// TIA Portal V17 export
// export: Created 2025-03-12T15:33:37.1839538Z, ExportSetting WithDefaults, DisplayName Totally Integrated Automation Portal, DisplayVersion V17 Update 8, DisplayName TIA Portal Openness, DisplayVersion V17 Update 8, DisplayName TIA Portal Version Control Interface, DisplayVersion V17, DisplayName SINAMICS Startdrive Advanced, DisplayVersion V17 SP2, DisplayName SINAMICS Startdrive G110M, G120, G120C, G120D, G120P, G115D, DisplayVersion V17 SP2, DisplayName SINAMICS Startdrive G130, G150, S120, S150, SINAMICS MV, S210, DisplayVersion V17 SP2, DisplayName STEP 7 Professional, DisplayVersion V17 Update 8, DisplayName SINUMERIK ONE STEP 7 Toolbox, DisplayVersion V17 Update 12, DisplayName SINUMERIK 840D sl STEP 7 Toolbox, DisplayVersion V17 Update 12, DisplayName STEP 7 Safety, DisplayVersion V17 Update 6, DisplayName WinCC Advanced, DisplayVersion V17 Update 8
FUNCTION "FC440_MACHINE_ALARM_DECODING" : Void   // FC440, LAD
{ S7_Optimized_Access := 'FALSE' }
AUTHOR : ETXETAR
VERSION : 1.0
// stored: AutoNumber false, IsIECCheckEnabled false, SetENOAutomatically false, UDAEnableTagReadback false
   VAR_TEMP
      RST_ALARMS_1 : Bool;   // RESET ALARMS 1
      RST_ALARMS_2 : Bool;   // RESET ALARMS 2
      ZERO : Int;   // ZERO
      RET_VAL_1 : Int;   // RET VALUE
   END_VAR
   VAR CONSTANT
      FC_CONSTANT : Int := 440;
   END_VAR
   VAR_TEMP   // added for the SCL form of the ladder/FBD networks
      _w1 : Bool;
      _w2 : Bool;
      _w3 : Bool;
      _w4 : Bool;
      _w5 : Bool;
      _w6 : Bool;
      _w7 : Bool;
      _w8 : Bool;
      _w9 : Bool;
      _w10 : Bool;
      _w11 : Bool;
   END_VAR
BEGIN

REGION Network 1: ZERO
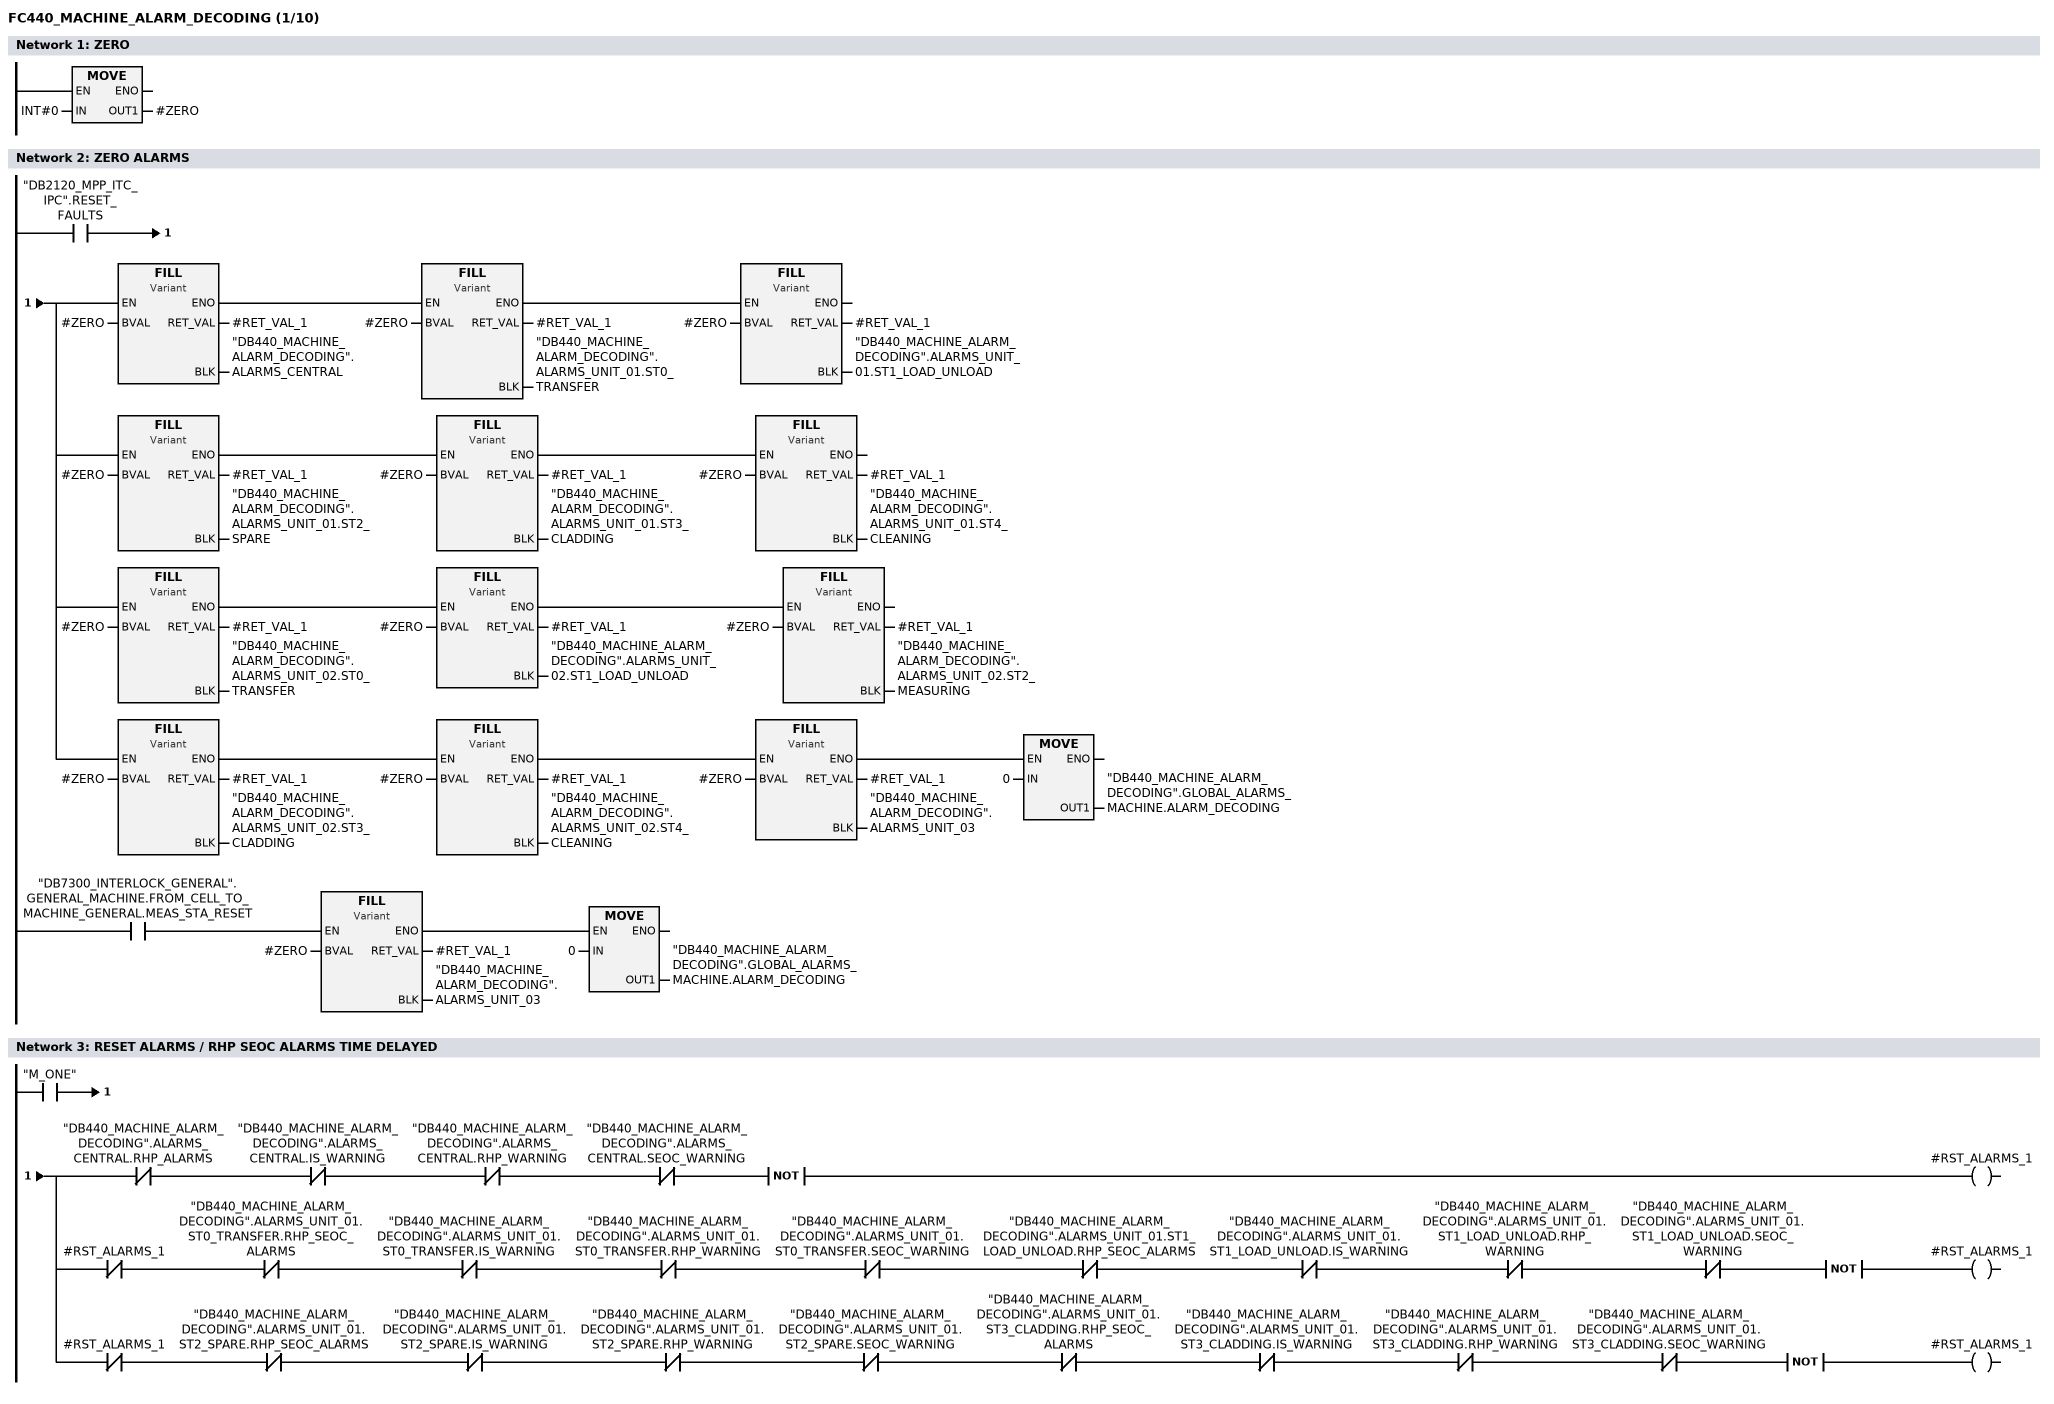
   RUNG wire#powerrail
      { S7_GenerateENO := "TRUE" } Move(in := INT#0, out1 => #ZERO)
   END_RUNG
   // the same network as SCL:
   #ZERO := INT#0;
END_REGION

REGION Network 2: ZERO ALARMS
   RUNG wire#powerrail
      Contact( "DB2120_MPP_ITC_IPC".RESET_FAULTS )
      wire#w1
      { S7_Templates := "ptr_type := Variant" } FILL(BVAL := #ZERO, RET_VAL => #RET_VAL_1, BLK => "DB440_MACHINE_ALARM_DECODING".ALARMS_CENTRAL)
      { S7_Templates := "ptr_type := Variant" } FILL(BVAL := #ZERO, RET_VAL => #RET_VAL_1, BLK => "DB440_MACHINE_ALARM_DECODING".ALARMS_UNIT_01.ST0_TRANSFER)
      { S7_Templates := "ptr_type := Variant" } FILL(BVAL := #ZERO, RET_VAL => #RET_VAL_1, BLK => "DB440_MACHINE_ALARM_DECODING".ALARMS_UNIT_01.ST1_LOAD_UNLOAD)
   END_RUNG
   RUNG wire#w1
      { S7_Templates := "ptr_type := Variant" } FILL(BVAL := #ZERO, RET_VAL => #RET_VAL_1, BLK => "DB440_MACHINE_ALARM_DECODING".ALARMS_UNIT_01.ST2_SPARE)
      { S7_Templates := "ptr_type := Variant" } FILL(BVAL := #ZERO, RET_VAL => #RET_VAL_1, BLK => "DB440_MACHINE_ALARM_DECODING".ALARMS_UNIT_01.ST3_CLADDING)
      { S7_Templates := "ptr_type := Variant" } FILL(BVAL := #ZERO, RET_VAL => #RET_VAL_1, BLK => "DB440_MACHINE_ALARM_DECODING".ALARMS_UNIT_01.ST4_CLEANING)
   END_RUNG
   RUNG wire#w1
      { S7_Templates := "ptr_type := Variant" } FILL(BVAL := #ZERO, RET_VAL => #RET_VAL_1, BLK => "DB440_MACHINE_ALARM_DECODING".ALARMS_UNIT_02.ST0_TRANSFER)
      { S7_Templates := "ptr_type := Variant" } FILL(BVAL := #ZERO, RET_VAL => #RET_VAL_1, BLK => "DB440_MACHINE_ALARM_DECODING".ALARMS_UNIT_02.ST1_LOAD_UNLOAD)
      { S7_Templates := "ptr_type := Variant" } FILL(BVAL := #ZERO, RET_VAL => #RET_VAL_1, BLK => "DB440_MACHINE_ALARM_DECODING".ALARMS_UNIT_02.ST2_MEASURING)
   END_RUNG
   RUNG wire#w1
      { S7_Templates := "ptr_type := Variant" } FILL(BVAL := #ZERO, RET_VAL => #RET_VAL_1, BLK => "DB440_MACHINE_ALARM_DECODING".ALARMS_UNIT_02.ST3_CLADDING)
      { S7_Templates := "ptr_type := Variant" } FILL(BVAL := #ZERO, RET_VAL => #RET_VAL_1, BLK => "DB440_MACHINE_ALARM_DECODING".ALARMS_UNIT_02.ST4_CLEANING)
      { S7_Templates := "ptr_type := Variant" } FILL(BVAL := #ZERO, RET_VAL => #RET_VAL_1, BLK => "DB440_MACHINE_ALARM_DECODING".ALARMS_UNIT_03)
      { S7_GenerateENO := "TRUE" } Move(in := 0, out1 => "DB440_MACHINE_ALARM_DECODING".GLOBAL_ALARMS_MACHINE.ALARM_DECODING)
   END_RUNG
   RUNG wire#powerrail
      Contact( "DB7300_INTERLOCK_GENERAL".GENERAL_MACHINE.FROM_CELL_TO_MACHINE_GENERAL.MEAS_STA_RESET )
      { S7_Templates := "ptr_type := Variant" } FILL(BVAL := #ZERO, RET_VAL => #RET_VAL_1, BLK => "DB440_MACHINE_ALARM_DECODING".ALARMS_UNIT_03)
      { S7_GenerateENO := "TRUE" } Move(in := 0, out1 => "DB440_MACHINE_ALARM_DECODING".GLOBAL_ALARMS_MACHINE.ALARM_DECODING)
   END_RUNG
   // the same network as SCL:
   #_w2 := "DB2120_MPP_ITC_IPC".RESET_FAULTS;
   #RET_VAL_1 := FILL(EN := "DB2120_MPP_ITC_IPC".RESET_FAULTS,
                      BVAL := #ZERO,
                      BLK => "DB440_MACHINE_ALARM_DECODING".ALARMS_CENTRAL,
                      ENO => #_w1);
   #RET_VAL_1 := FILL(EN := #_w1,
                      BVAL := #ZERO,
                      BLK => "DB440_MACHINE_ALARM_DECODING".ALARMS_UNIT_01.ST0_TRANSFER,
                      ENO => #_w3);
   IF #_w3 THEN
       #RET_VAL_1 := FILL(BVAL := #ZERO, BLK => "DB440_MACHINE_ALARM_DECODING".ALARMS_UNIT_01.ST1_LOAD_UNLOAD);
   END_IF;
   #RET_VAL_1 := FILL(EN := #_w2,
                      BVAL := #ZERO,
                      BLK => "DB440_MACHINE_ALARM_DECODING".ALARMS_UNIT_01.ST2_SPARE,
                      ENO => #_w4);
   #RET_VAL_1 := FILL(EN := #_w4,
                      BVAL := #ZERO,
                      BLK => "DB440_MACHINE_ALARM_DECODING".ALARMS_UNIT_01.ST3_CLADDING,
                      ENO => #_w5);
   IF #_w5 THEN
       #RET_VAL_1 := FILL(BVAL := #ZERO, BLK => "DB440_MACHINE_ALARM_DECODING".ALARMS_UNIT_01.ST4_CLEANING);
   END_IF;
   #RET_VAL_1 := FILL(EN := #_w2,
                      BVAL := #ZERO,
                      BLK => "DB440_MACHINE_ALARM_DECODING".ALARMS_UNIT_02.ST0_TRANSFER,
                      ENO => #_w6);
   #RET_VAL_1 := FILL(EN := #_w6,
                      BVAL := #ZERO,
                      BLK => "DB440_MACHINE_ALARM_DECODING".ALARMS_UNIT_02.ST1_LOAD_UNLOAD,
                      ENO => #_w7);
   IF #_w7 THEN
       #RET_VAL_1 := FILL(BVAL := #ZERO, BLK => "DB440_MACHINE_ALARM_DECODING".ALARMS_UNIT_02.ST2_MEASURING);
   END_IF;
   #RET_VAL_1 := FILL(EN := #_w2,
                      BVAL := #ZERO,
                      BLK => "DB440_MACHINE_ALARM_DECODING".ALARMS_UNIT_02.ST3_CLADDING,
                      ENO => #_w8);
   #RET_VAL_1 := FILL(EN := #_w8,
                      BVAL := #ZERO,
                      BLK => "DB440_MACHINE_ALARM_DECODING".ALARMS_UNIT_02.ST4_CLEANING,
                      ENO => #_w9);
   #RET_VAL_1 := FILL(EN := #_w9,
                      BVAL := #ZERO,
                      BLK => "DB440_MACHINE_ALARM_DECODING".ALARMS_UNIT_03,
                      ENO => #_w10);
   IF #_w10 THEN "DB440_MACHINE_ALARM_DECODING".GLOBAL_ALARMS_MACHINE.ALARM_DECODING := 0; END_IF;
   #RET_VAL_1 := FILL(EN := "DB7300_INTERLOCK_GENERAL".GENERAL_MACHINE.FROM_CELL_TO_MACHINE_GENERAL.MEAS_STA_RESET,
                      BVAL := #ZERO,
                      BLK => "DB440_MACHINE_ALARM_DECODING".ALARMS_UNIT_03,
                      ENO => #_w11);
   IF #_w11 THEN "DB440_MACHINE_ALARM_DECODING".GLOBAL_ALARMS_MACHINE.ALARM_DECODING := 0; END_IF;
END_REGION

REGION Network 3: RESET ALARMS / RHP SEOC ALARMS TIME DELAYED
   RUNG wire#powerrail
      Contact( "M_ONE" )
      wire#w1
      I_Contact( "DB440_MACHINE_ALARM_DECODING".ALARMS_CENTRAL.RHP_ALARMS )
      I_Contact( "DB440_MACHINE_ALARM_DECODING".ALARMS_CENTRAL.IS_WARNING )
      I_Contact( "DB440_MACHINE_ALARM_DECODING".ALARMS_CENTRAL.RHP_WARNING )
      I_Contact( "DB440_MACHINE_ALARM_DECODING".ALARMS_CENTRAL.SEOC_WARNING )
      Not()
      Coil( #RST_ALARMS_1 )
   END_RUNG
   RUNG wire#w1
      I_Contact( #RST_ALARMS_1 )
      I_Contact( "DB440_MACHINE_ALARM_DECODING".ALARMS_UNIT_01.ST0_TRANSFER.RHP_SEOC_ALARMS )
      I_Contact( "DB440_MACHINE_ALARM_DECODING".ALARMS_UNIT_01.ST0_TRANSFER.IS_WARNING )
      I_Contact( "DB440_MACHINE_ALARM_DECODING".ALARMS_UNIT_01.ST0_TRANSFER.RHP_WARNING )
      I_Contact( "DB440_MACHINE_ALARM_DECODING".ALARMS_UNIT_01.ST0_TRANSFER.SEOC_WARNING )
      I_Contact( "DB440_MACHINE_ALARM_DECODING".ALARMS_UNIT_01.ST1_LOAD_UNLOAD.RHP_SEOC_ALARMS )
      I_Contact( "DB440_MACHINE_ALARM_DECODING".ALARMS_UNIT_01.ST1_LOAD_UNLOAD.IS_WARNING )
      I_Contact( "DB440_MACHINE_ALARM_DECODING".ALARMS_UNIT_01.ST1_LOAD_UNLOAD.RHP_WARNING )
      I_Contact( "DB440_MACHINE_ALARM_DECODING".ALARMS_UNIT_01.ST1_LOAD_UNLOAD.SEOC_WARNING )
      Not()
      Coil( #RST_ALARMS_1 )
   END_RUNG
   RUNG wire#w1
      I_Contact( #RST_ALARMS_1 )
      I_Contact( "DB440_MACHINE_ALARM_DECODING".ALARMS_UNIT_01.ST2_SPARE.RHP_SEOC_ALARMS )
      I_Contact( "DB440_MACHINE_ALARM_DECODING".ALARMS_UNIT_01.ST2_SPARE.IS_WARNING )
      I_Contact( "DB440_MACHINE_ALARM_DECODING".ALARMS_UNIT_01.ST2_SPARE.RHP_WARNING )
      I_Contact( "DB440_MACHINE_ALARM_DECODING".ALARMS_UNIT_01.ST2_SPARE.SEOC_WARNING )
      I_Contact( "DB440_MACHINE_ALARM_DECODING".ALARMS_UNIT_01.ST3_CLADDING.RHP_SEOC_ALARMS )
      I_Contact( "DB440_MACHINE_ALARM_DECODING".ALARMS_UNIT_01.ST3_CLADDING.IS_WARNING )
      I_Contact( "DB440_MACHINE_ALARM_DECODING".ALARMS_UNIT_01.ST3_CLADDING.RHP_WARNING )
      I_Contact( "DB440_MACHINE_ALARM_DECODING".ALARMS_UNIT_01.ST3_CLADDING.SEOC_WARNING )
      Not()
      Coil( #RST_ALARMS_1 )
   END_RUNG
   // the same network as SCL:
   #RST_ALARMS_1 := NOT ("M_ONE" AND NOT "DB440_MACHINE_ALARM_DECODING".ALARMS_CENTRAL.RHP_ALARMS AND NOT "DB440_MACHINE_ALARM_DECODING".ALARMS_CENTRAL.IS_WARNING AND NOT "DB440_MACHINE_ALARM_DECODING".ALARMS_CENTRAL.RHP_WARNING AND NOT "DB440_MACHINE_ALARM_DECODING".ALARMS_CENTRAL.SEOC_WARNING);
   #RST_ALARMS_1 := NOT ("M_ONE" AND NOT #RST_ALARMS_1 AND NOT "DB440_MACHINE_ALARM_DECODING".ALARMS_UNIT_01.ST0_TRANSFER.RHP_SEOC_ALARMS AND NOT "DB440_MACHINE_ALARM_DECODING".ALARMS_UNIT_01.ST0_TRANSFER.IS_WARNING AND NOT "DB440_MACHINE_ALARM_DECODING".ALARMS_UNIT_01.ST0_TRANSFER.RHP_WARNING AND NOT "DB440_MACHINE_ALARM_DECODING".ALARMS_UNIT_01.ST0_TRANSFER.SEOC_WARNING AND NOT "DB440_MACHINE_ALARM_DECODING".ALARMS_UNIT_01.ST1_LOAD_UNLOAD.RHP_SEOC_ALARMS AND NOT "DB440_MACHINE_ALARM_DECODING".ALARMS_UNIT_01.ST1_LOAD_UNLOAD.IS_WARNING AND NOT "DB440_MACHINE_ALARM_DECODING".ALARMS_UNIT_01.ST1_LOAD_UNLOAD.RHP_WARNING AND NOT "DB440_MACHINE_ALARM_DECODING".ALARMS_UNIT_01.ST1_LOAD_UNLOAD.SEOC_WARNING);
   #RST_ALARMS_1 := NOT ("M_ONE" AND NOT #RST_ALARMS_1 AND NOT "DB440_MACHINE_ALARM_DECODING".ALARMS_UNIT_01.ST2_SPARE.RHP_SEOC_ALARMS AND NOT "DB440_MACHINE_ALARM_DECODING".ALARMS_UNIT_01.ST2_SPARE.IS_WARNING AND NOT "DB440_MACHINE_ALARM_DECODING".ALARMS_UNIT_01.ST2_SPARE.RHP_WARNING AND NOT "DB440_MACHINE_ALARM_DECODING".ALARMS_UNIT_01.ST2_SPARE.SEOC_WARNING AND NOT "DB440_MACHINE_ALARM_DECODING".ALARMS_UNIT_01.ST3_CLADDING.RHP_SEOC_ALARMS AND NOT "DB440_MACHINE_ALARM_DECODING".ALARMS_UNIT_01.ST3_CLADDING.IS_WARNING AND NOT "DB440_MACHINE_ALARM_DECODING".ALARMS_UNIT_01.ST3_CLADDING.RHP_WARNING AND NOT "DB440_MACHINE_ALARM_DECODING".ALARMS_UNIT_01.ST3_CLADDING.SEOC_WARNING);
END_REGION

REGION Network 4: RESET ALARMS / RHP SEOC ALARMS TIME DELAYED
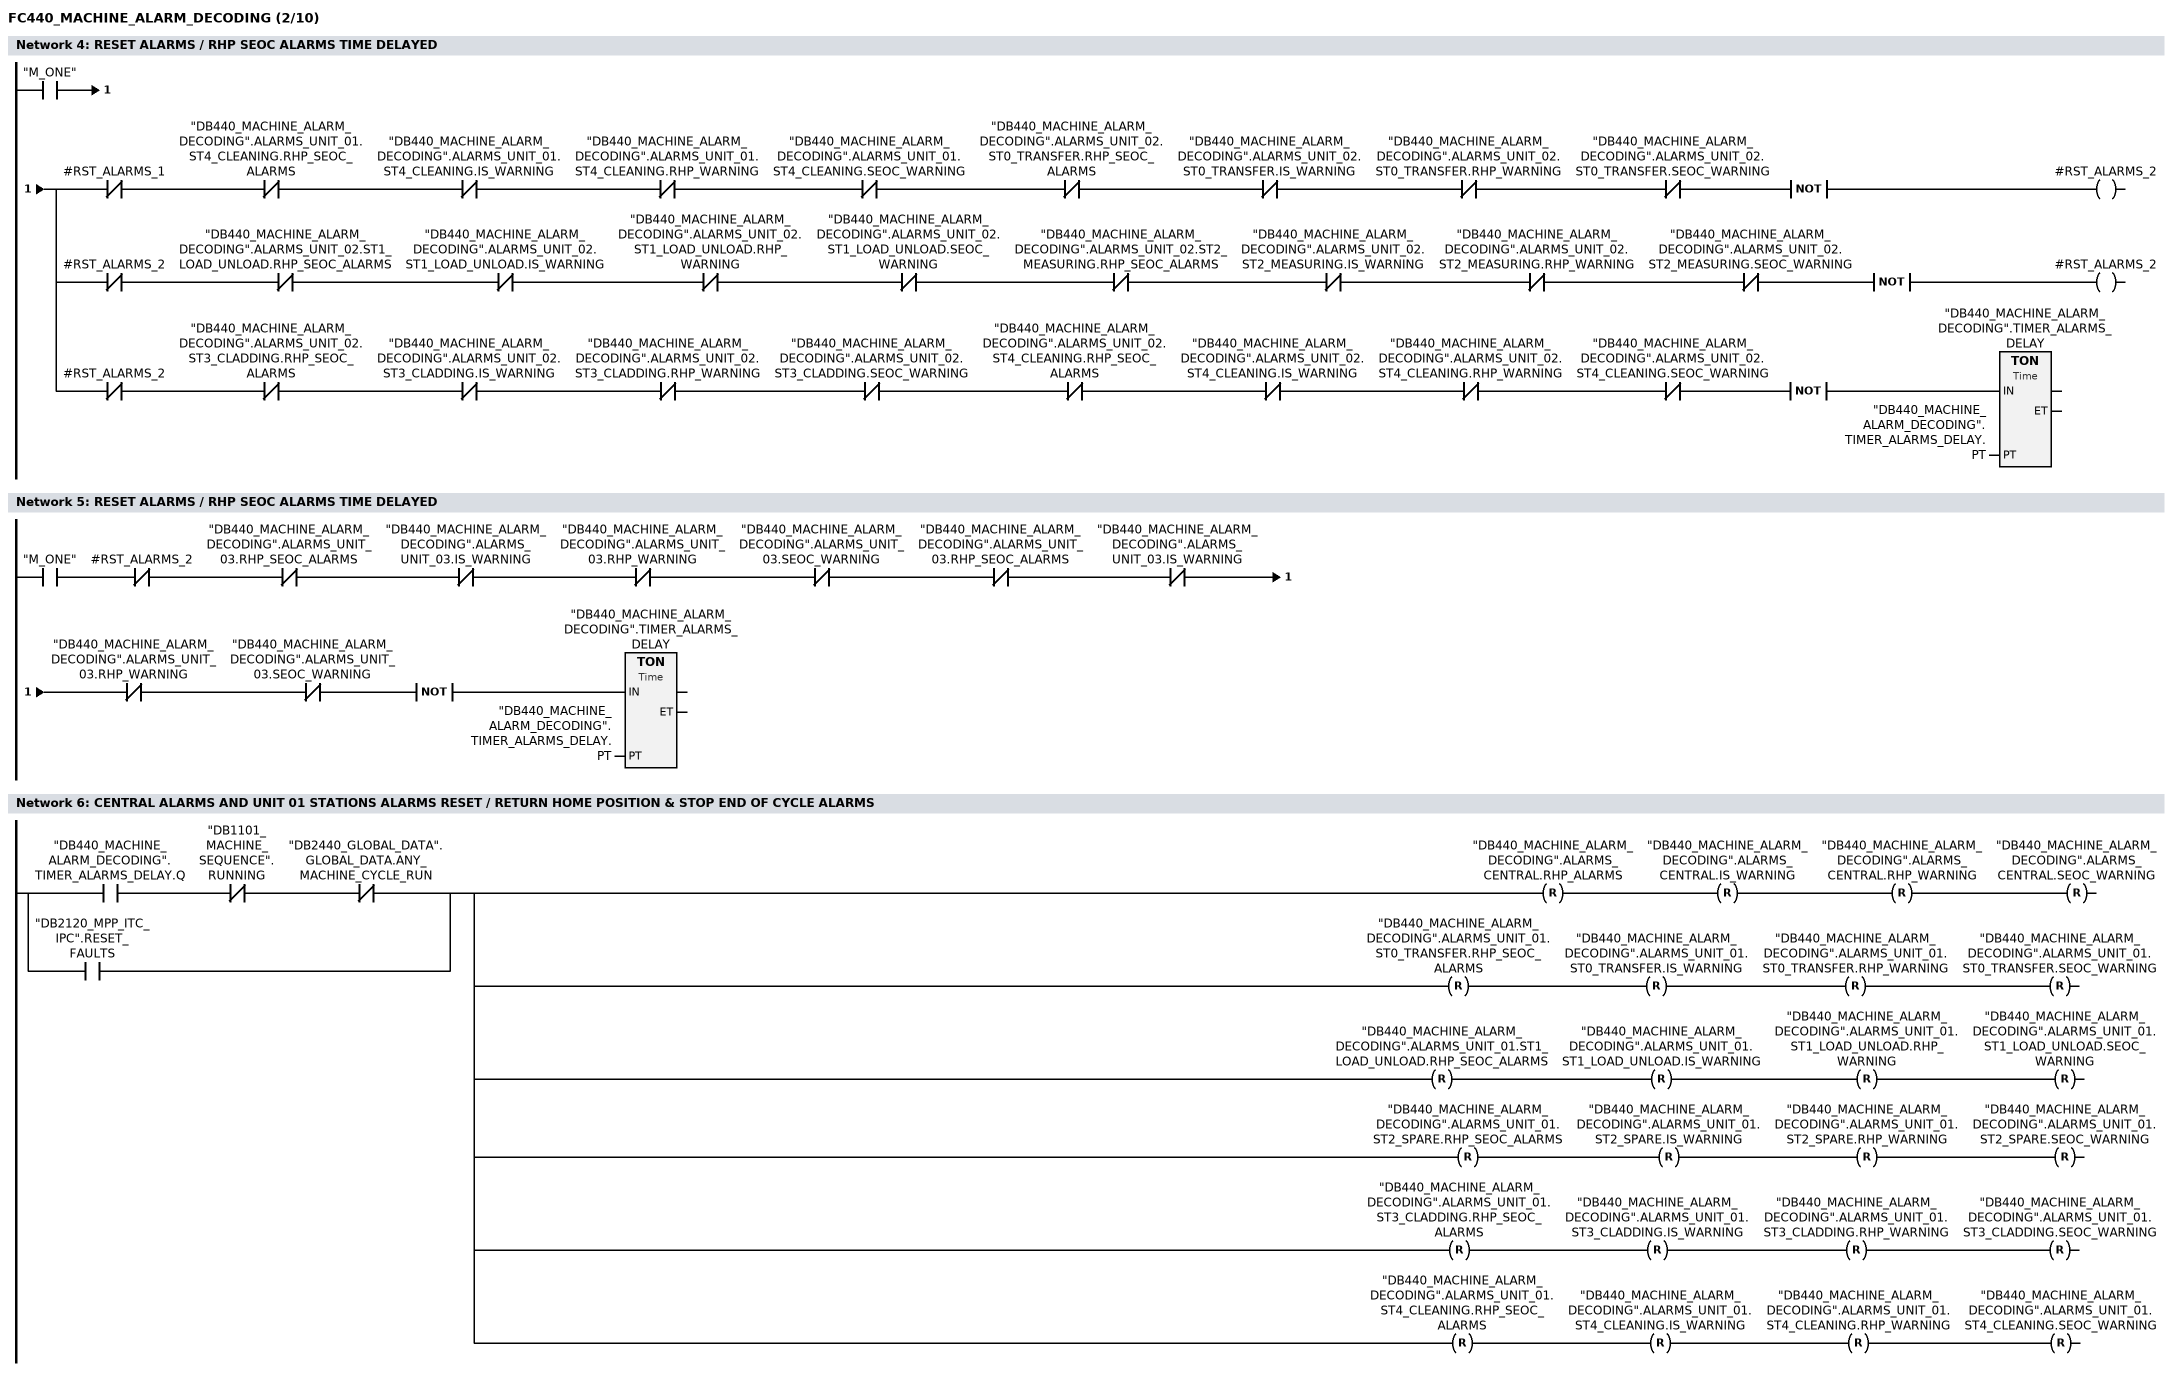
   RUNG wire#powerrail
      Contact( "M_ONE" )
      wire#w1
      I_Contact( #RST_ALARMS_1 )
      I_Contact( "DB440_MACHINE_ALARM_DECODING".ALARMS_UNIT_01.ST4_CLEANING.RHP_SEOC_ALARMS )
      I_Contact( "DB440_MACHINE_ALARM_DECODING".ALARMS_UNIT_01.ST4_CLEANING.IS_WARNING )
      I_Contact( "DB440_MACHINE_ALARM_DECODING".ALARMS_UNIT_01.ST4_CLEANING.RHP_WARNING )
      I_Contact( "DB440_MACHINE_ALARM_DECODING".ALARMS_UNIT_01.ST4_CLEANING.SEOC_WARNING )
      I_Contact( "DB440_MACHINE_ALARM_DECODING".ALARMS_UNIT_02.ST0_TRANSFER.RHP_SEOC_ALARMS )
      I_Contact( "DB440_MACHINE_ALARM_DECODING".ALARMS_UNIT_02.ST0_TRANSFER.IS_WARNING )
      I_Contact( "DB440_MACHINE_ALARM_DECODING".ALARMS_UNIT_02.ST0_TRANSFER.RHP_WARNING )
      I_Contact( "DB440_MACHINE_ALARM_DECODING".ALARMS_UNIT_02.ST0_TRANSFER.SEOC_WARNING )
      Not()
      Coil( #RST_ALARMS_2 )
   END_RUNG
   RUNG wire#w1
      I_Contact( #RST_ALARMS_2 )
      I_Contact( "DB440_MACHINE_ALARM_DECODING".ALARMS_UNIT_02.ST1_LOAD_UNLOAD.RHP_SEOC_ALARMS )
      I_Contact( "DB440_MACHINE_ALARM_DECODING".ALARMS_UNIT_02.ST1_LOAD_UNLOAD.IS_WARNING )
      I_Contact( "DB440_MACHINE_ALARM_DECODING".ALARMS_UNIT_02.ST1_LOAD_UNLOAD.RHP_WARNING )
      I_Contact( "DB440_MACHINE_ALARM_DECODING".ALARMS_UNIT_02.ST1_LOAD_UNLOAD.SEOC_WARNING )
      I_Contact( "DB440_MACHINE_ALARM_DECODING".ALARMS_UNIT_02.ST2_MEASURING.RHP_SEOC_ALARMS )
      I_Contact( "DB440_MACHINE_ALARM_DECODING".ALARMS_UNIT_02.ST2_MEASURING.IS_WARNING )
      I_Contact( "DB440_MACHINE_ALARM_DECODING".ALARMS_UNIT_02.ST2_MEASURING.RHP_WARNING )
      I_Contact( "DB440_MACHINE_ALARM_DECODING".ALARMS_UNIT_02.ST2_MEASURING.SEOC_WARNING )
      Not()
      Coil( #RST_ALARMS_2 )
   END_RUNG
   RUNG wire#w1
      I_Contact( #RST_ALARMS_2 )
      I_Contact( "DB440_MACHINE_ALARM_DECODING".ALARMS_UNIT_02.ST3_CLADDING.RHP_SEOC_ALARMS )
      I_Contact( "DB440_MACHINE_ALARM_DECODING".ALARMS_UNIT_02.ST3_CLADDING.IS_WARNING )
      I_Contact( "DB440_MACHINE_ALARM_DECODING".ALARMS_UNIT_02.ST3_CLADDING.RHP_WARNING )
      I_Contact( "DB440_MACHINE_ALARM_DECODING".ALARMS_UNIT_02.ST3_CLADDING.SEOC_WARNING )
      I_Contact( "DB440_MACHINE_ALARM_DECODING".ALARMS_UNIT_02.ST4_CLEANING.RHP_SEOC_ALARMS )
      I_Contact( "DB440_MACHINE_ALARM_DECODING".ALARMS_UNIT_02.ST4_CLEANING.IS_WARNING )
      I_Contact( "DB440_MACHINE_ALARM_DECODING".ALARMS_UNIT_02.ST4_CLEANING.RHP_WARNING )
      I_Contact( "DB440_MACHINE_ALARM_DECODING".ALARMS_UNIT_02.ST4_CLEANING.SEOC_WARNING )
      Not()
      { S7_Templates := "time_type := Time" } "DB440_MACHINE_ALARM_DECODING".TIMER_ALARMS_DELAY.TON(pt := "DB440_MACHINE_ALARM_DECODING".TIMER_ALARMS_DELAY.PT, et =>)
   END_RUNG
   // the same network as SCL:
   #RST_ALARMS_2 := NOT ("M_ONE" AND NOT #RST_ALARMS_1 AND NOT "DB440_MACHINE_ALARM_DECODING".ALARMS_UNIT_01.ST4_CLEANING.RHP_SEOC_ALARMS AND NOT "DB440_MACHINE_ALARM_DECODING".ALARMS_UNIT_01.ST4_CLEANING.IS_WARNING AND NOT "DB440_MACHINE_ALARM_DECODING".ALARMS_UNIT_01.ST4_CLEANING.RHP_WARNING AND NOT "DB440_MACHINE_ALARM_DECODING".ALARMS_UNIT_01.ST4_CLEANING.SEOC_WARNING AND NOT "DB440_MACHINE_ALARM_DECODING".ALARMS_UNIT_02.ST0_TRANSFER.RHP_SEOC_ALARMS AND NOT "DB440_MACHINE_ALARM_DECODING".ALARMS_UNIT_02.ST0_TRANSFER.IS_WARNING AND NOT "DB440_MACHINE_ALARM_DECODING".ALARMS_UNIT_02.ST0_TRANSFER.RHP_WARNING AND NOT "DB440_MACHINE_ALARM_DECODING".ALARMS_UNIT_02.ST0_TRANSFER.SEOC_WARNING);
   #RST_ALARMS_2 := NOT ("M_ONE" AND NOT #RST_ALARMS_2 AND NOT "DB440_MACHINE_ALARM_DECODING".ALARMS_UNIT_02.ST1_LOAD_UNLOAD.RHP_SEOC_ALARMS AND NOT "DB440_MACHINE_ALARM_DECODING".ALARMS_UNIT_02.ST1_LOAD_UNLOAD.IS_WARNING AND NOT "DB440_MACHINE_ALARM_DECODING".ALARMS_UNIT_02.ST1_LOAD_UNLOAD.RHP_WARNING AND NOT "DB440_MACHINE_ALARM_DECODING".ALARMS_UNIT_02.ST1_LOAD_UNLOAD.SEOC_WARNING AND NOT "DB440_MACHINE_ALARM_DECODING".ALARMS_UNIT_02.ST2_MEASURING.RHP_SEOC_ALARMS AND NOT "DB440_MACHINE_ALARM_DECODING".ALARMS_UNIT_02.ST2_MEASURING.IS_WARNING AND NOT "DB440_MACHINE_ALARM_DECODING".ALARMS_UNIT_02.ST2_MEASURING.RHP_WARNING AND NOT "DB440_MACHINE_ALARM_DECODING".ALARMS_UNIT_02.ST2_MEASURING.SEOC_WARNING);
   "DB440_MACHINE_ALARM_DECODING".TIMER_ALARMS_DELAY.TON(IN := NOT ("M_ONE" AND NOT #RST_ALARMS_2 AND NOT "DB440_MACHINE_ALARM_DECODING".ALARMS_UNIT_02.ST3_CLADDING.RHP_SEOC_ALARMS AND NOT "DB440_MACHINE_ALARM_DECODING".ALARMS_UNIT_02.ST3_CLADDING.IS_WARNING AND NOT "DB440_MACHINE_ALARM_DECODING".ALARMS_UNIT_02.ST3_CLADDING.RHP_WARNING AND NOT "DB440_MACHINE_ALARM_DECODING".ALARMS_UNIT_02.ST3_CLADDING.SEOC_WARNING AND NOT "DB440_MACHINE_ALARM_DECODING".ALARMS_UNIT_02.ST4_CLEANING.RHP_SEOC_ALARMS AND NOT "DB440_MACHINE_ALARM_DECODING".ALARMS_UNIT_02.ST4_CLEANING.IS_WARNING AND NOT "DB440_MACHINE_ALARM_DECODING".ALARMS_UNIT_02.ST4_CLEANING.RHP_WARNING AND NOT "DB440_MACHINE_ALARM_DECODING".ALARMS_UNIT_02.ST4_CLEANING.SEOC_WARNING),
                           PT := "DB440_MACHINE_ALARM_DECODING".TIMER_ALARMS_DELAY.PT);
END_REGION

REGION Network 5: RESET ALARMS / RHP SEOC ALARMS TIME DELAYED
   RUNG wire#powerrail
      Contact( "M_ONE" )
      I_Contact( #RST_ALARMS_2 )
      I_Contact( "DB440_MACHINE_ALARM_DECODING".ALARMS_UNIT_03.RHP_SEOC_ALARMS )
      I_Contact( "DB440_MACHINE_ALARM_DECODING".ALARMS_UNIT_03.IS_WARNING )
      I_Contact( "DB440_MACHINE_ALARM_DECODING".ALARMS_UNIT_03.RHP_WARNING )
      I_Contact( "DB440_MACHINE_ALARM_DECODING".ALARMS_UNIT_03.SEOC_WARNING )
      I_Contact( "DB440_MACHINE_ALARM_DECODING".ALARMS_UNIT_03.RHP_SEOC_ALARMS )
      I_Contact( "DB440_MACHINE_ALARM_DECODING".ALARMS_UNIT_03.IS_WARNING )
      I_Contact( "DB440_MACHINE_ALARM_DECODING".ALARMS_UNIT_03.RHP_WARNING )
      I_Contact( "DB440_MACHINE_ALARM_DECODING".ALARMS_UNIT_03.SEOC_WARNING )
      Not()
      { S7_Templates := "time_type := Time" } "DB440_MACHINE_ALARM_DECODING".TIMER_ALARMS_DELAY.TON(pt := "DB440_MACHINE_ALARM_DECODING".TIMER_ALARMS_DELAY.PT, et =>)
   END_RUNG
   // the same network as SCL:
   "DB440_MACHINE_ALARM_DECODING".TIMER_ALARMS_DELAY.TON(IN := NOT ("M_ONE" AND NOT #RST_ALARMS_2 AND NOT "DB440_MACHINE_ALARM_DECODING".ALARMS_UNIT_03.RHP_SEOC_ALARMS AND NOT "DB440_MACHINE_ALARM_DECODING".ALARMS_UNIT_03.IS_WARNING AND NOT "DB440_MACHINE_ALARM_DECODING".ALARMS_UNIT_03.RHP_WARNING AND NOT "DB440_MACHINE_ALARM_DECODING".ALARMS_UNIT_03.SEOC_WARNING AND NOT "DB440_MACHINE_ALARM_DECODING".ALARMS_UNIT_03.RHP_SEOC_ALARMS AND NOT "DB440_MACHINE_ALARM_DECODING".ALARMS_UNIT_03.IS_WARNING AND NOT "DB440_MACHINE_ALARM_DECODING".ALARMS_UNIT_03.RHP_WARNING AND NOT "DB440_MACHINE_ALARM_DECODING".ALARMS_UNIT_03.SEOC_WARNING),
                           PT := "DB440_MACHINE_ALARM_DECODING".TIMER_ALARMS_DELAY.PT);
END_REGION

REGION Network 6: CENTRAL ALARMS AND UNIT 01 STATIONS ALARMS RESET / RETURN HOME POSITION & STOP END OF CYCLE ALARMS
   RUNG wire#powerrail
      Contact( "DB440_MACHINE_ALARM_DECODING".TIMER_ALARMS_DELAY.Q )
      I_Contact( "DB1101_MACHINE_SEQUENCE".RUNNING )
      I_Contact( "DB2440_GLOBAL_DATA".GLOBAL_DATA.ANY_MACHINE_CYCLE_RUN )
      wire#w1
      R_Coil( "DB440_MACHINE_ALARM_DECODING".ALARMS_CENTRAL.RHP_ALARMS )
      R_Coil( "DB440_MACHINE_ALARM_DECODING".ALARMS_CENTRAL.IS_WARNING )
      R_Coil( "DB440_MACHINE_ALARM_DECODING".ALARMS_CENTRAL.RHP_WARNING )
      R_Coil( "DB440_MACHINE_ALARM_DECODING".ALARMS_CENTRAL.SEOC_WARNING )
   END_RUNG
   RUNG wire#powerrail
      Contact( "DB2120_MPP_ITC_IPC".RESET_FAULTS )
   END_RUNG wire#w1
   RUNG wire#w1
      R_Coil( "DB440_MACHINE_ALARM_DECODING".ALARMS_UNIT_01.ST0_TRANSFER.RHP_SEOC_ALARMS )
      R_Coil( "DB440_MACHINE_ALARM_DECODING".ALARMS_UNIT_01.ST0_TRANSFER.IS_WARNING )
      R_Coil( "DB440_MACHINE_ALARM_DECODING".ALARMS_UNIT_01.ST0_TRANSFER.RHP_WARNING )
      R_Coil( "DB440_MACHINE_ALARM_DECODING".ALARMS_UNIT_01.ST0_TRANSFER.SEOC_WARNING )
   END_RUNG
   RUNG wire#w1
      R_Coil( "DB440_MACHINE_ALARM_DECODING".ALARMS_UNIT_01.ST1_LOAD_UNLOAD.RHP_SEOC_ALARMS )
      R_Coil( "DB440_MACHINE_ALARM_DECODING".ALARMS_UNIT_01.ST1_LOAD_UNLOAD.IS_WARNING )
      R_Coil( "DB440_MACHINE_ALARM_DECODING".ALARMS_UNIT_01.ST1_LOAD_UNLOAD.RHP_WARNING )
      R_Coil( "DB440_MACHINE_ALARM_DECODING".ALARMS_UNIT_01.ST1_LOAD_UNLOAD.SEOC_WARNING )
   END_RUNG
   RUNG wire#w1
      R_Coil( "DB440_MACHINE_ALARM_DECODING".ALARMS_UNIT_01.ST2_SPARE.RHP_SEOC_ALARMS )
      R_Coil( "DB440_MACHINE_ALARM_DECODING".ALARMS_UNIT_01.ST2_SPARE.IS_WARNING )
      R_Coil( "DB440_MACHINE_ALARM_DECODING".ALARMS_UNIT_01.ST2_SPARE.RHP_WARNING )
      R_Coil( "DB440_MACHINE_ALARM_DECODING".ALARMS_UNIT_01.ST2_SPARE.SEOC_WARNING )
   END_RUNG
   RUNG wire#w1
      R_Coil( "DB440_MACHINE_ALARM_DECODING".ALARMS_UNIT_01.ST3_CLADDING.RHP_SEOC_ALARMS )
      R_Coil( "DB440_MACHINE_ALARM_DECODING".ALARMS_UNIT_01.ST3_CLADDING.IS_WARNING )
      R_Coil( "DB440_MACHINE_ALARM_DECODING".ALARMS_UNIT_01.ST3_CLADDING.RHP_WARNING )
      R_Coil( "DB440_MACHINE_ALARM_DECODING".ALARMS_UNIT_01.ST3_CLADDING.SEOC_WARNING )
   END_RUNG
   RUNG wire#w1
      R_Coil( "DB440_MACHINE_ALARM_DECODING".ALARMS_UNIT_01.ST4_CLEANING.RHP_SEOC_ALARMS )
      R_Coil( "DB440_MACHINE_ALARM_DECODING".ALARMS_UNIT_01.ST4_CLEANING.IS_WARNING )
      R_Coil( "DB440_MACHINE_ALARM_DECODING".ALARMS_UNIT_01.ST4_CLEANING.RHP_WARNING )
      R_Coil( "DB440_MACHINE_ALARM_DECODING".ALARMS_UNIT_01.ST4_CLEANING.SEOC_WARNING )
   END_RUNG
   // the same network as SCL:
   IF ("DB440_MACHINE_ALARM_DECODING".TIMER_ALARMS_DELAY.Q AND NOT "DB1101_MACHINE_SEQUENCE".RUNNING AND NOT "DB2440_GLOBAL_DATA".GLOBAL_DATA.ANY_MACHINE_CYCLE_RUN) OR "DB2120_MPP_ITC_IPC".RESET_FAULTS THEN
       "DB440_MACHINE_ALARM_DECODING".ALARMS_CENTRAL.RHP_ALARMS := FALSE;
       "DB440_MACHINE_ALARM_DECODING".ALARMS_CENTRAL.IS_WARNING := FALSE;
       "DB440_MACHINE_ALARM_DECODING".ALARMS_CENTRAL.RHP_WARNING := FALSE;
       "DB440_MACHINE_ALARM_DECODING".ALARMS_CENTRAL.SEOC_WARNING := FALSE;
       "DB440_MACHINE_ALARM_DECODING".ALARMS_UNIT_01.ST0_TRANSFER.RHP_SEOC_ALARMS := FALSE;
       "DB440_MACHINE_ALARM_DECODING".ALARMS_UNIT_01.ST0_TRANSFER.IS_WARNING := FALSE;
       "DB440_MACHINE_ALARM_DECODING".ALARMS_UNIT_01.ST0_TRANSFER.RHP_WARNING := FALSE;
       "DB440_MACHINE_ALARM_DECODING".ALARMS_UNIT_01.ST0_TRANSFER.SEOC_WARNING := FALSE;
       "DB440_MACHINE_ALARM_DECODING".ALARMS_UNIT_01.ST1_LOAD_UNLOAD.RHP_SEOC_ALARMS := FALSE;
       "DB440_MACHINE_ALARM_DECODING".ALARMS_UNIT_01.ST1_LOAD_UNLOAD.IS_WARNING := FALSE;
       "DB440_MACHINE_ALARM_DECODING".ALARMS_UNIT_01.ST1_LOAD_UNLOAD.RHP_WARNING := FALSE;
       "DB440_MACHINE_ALARM_DECODING".ALARMS_UNIT_01.ST1_LOAD_UNLOAD.SEOC_WARNING := FALSE;
       "DB440_MACHINE_ALARM_DECODING".ALARMS_UNIT_01.ST2_SPARE.RHP_SEOC_ALARMS := FALSE;
       "DB440_MACHINE_ALARM_DECODING".ALARMS_UNIT_01.ST2_SPARE.IS_WARNING := FALSE;
       "DB440_MACHINE_ALARM_DECODING".ALARMS_UNIT_01.ST2_SPARE.RHP_WARNING := FALSE;
       "DB440_MACHINE_ALARM_DECODING".ALARMS_UNIT_01.ST2_SPARE.SEOC_WARNING := FALSE;
       "DB440_MACHINE_ALARM_DECODING".ALARMS_UNIT_01.ST3_CLADDING.RHP_SEOC_ALARMS := FALSE;
       "DB440_MACHINE_ALARM_DECODING".ALARMS_UNIT_01.ST3_CLADDING.IS_WARNING := FALSE;
       "DB440_MACHINE_ALARM_DECODING".ALARMS_UNIT_01.ST3_CLADDING.RHP_WARNING := FALSE;
       "DB440_MACHINE_ALARM_DECODING".ALARMS_UNIT_01.ST3_CLADDING.SEOC_WARNING := FALSE;
       "DB440_MACHINE_ALARM_DECODING".ALARMS_UNIT_01.ST4_CLEANING.RHP_SEOC_ALARMS := FALSE;
       "DB440_MACHINE_ALARM_DECODING".ALARMS_UNIT_01.ST4_CLEANING.IS_WARNING := FALSE;
       "DB440_MACHINE_ALARM_DECODING".ALARMS_UNIT_01.ST4_CLEANING.RHP_WARNING := FALSE;
       "DB440_MACHINE_ALARM_DECODING".ALARMS_UNIT_01.ST4_CLEANING.SEOC_WARNING := FALSE;
   END_IF;
END_REGION

REGION Network 7: UNIT 02 STATIONS ALARMS AND UNIT 03 ALARMS RESET / RHP SEOC ALARMS TIME DELAYED
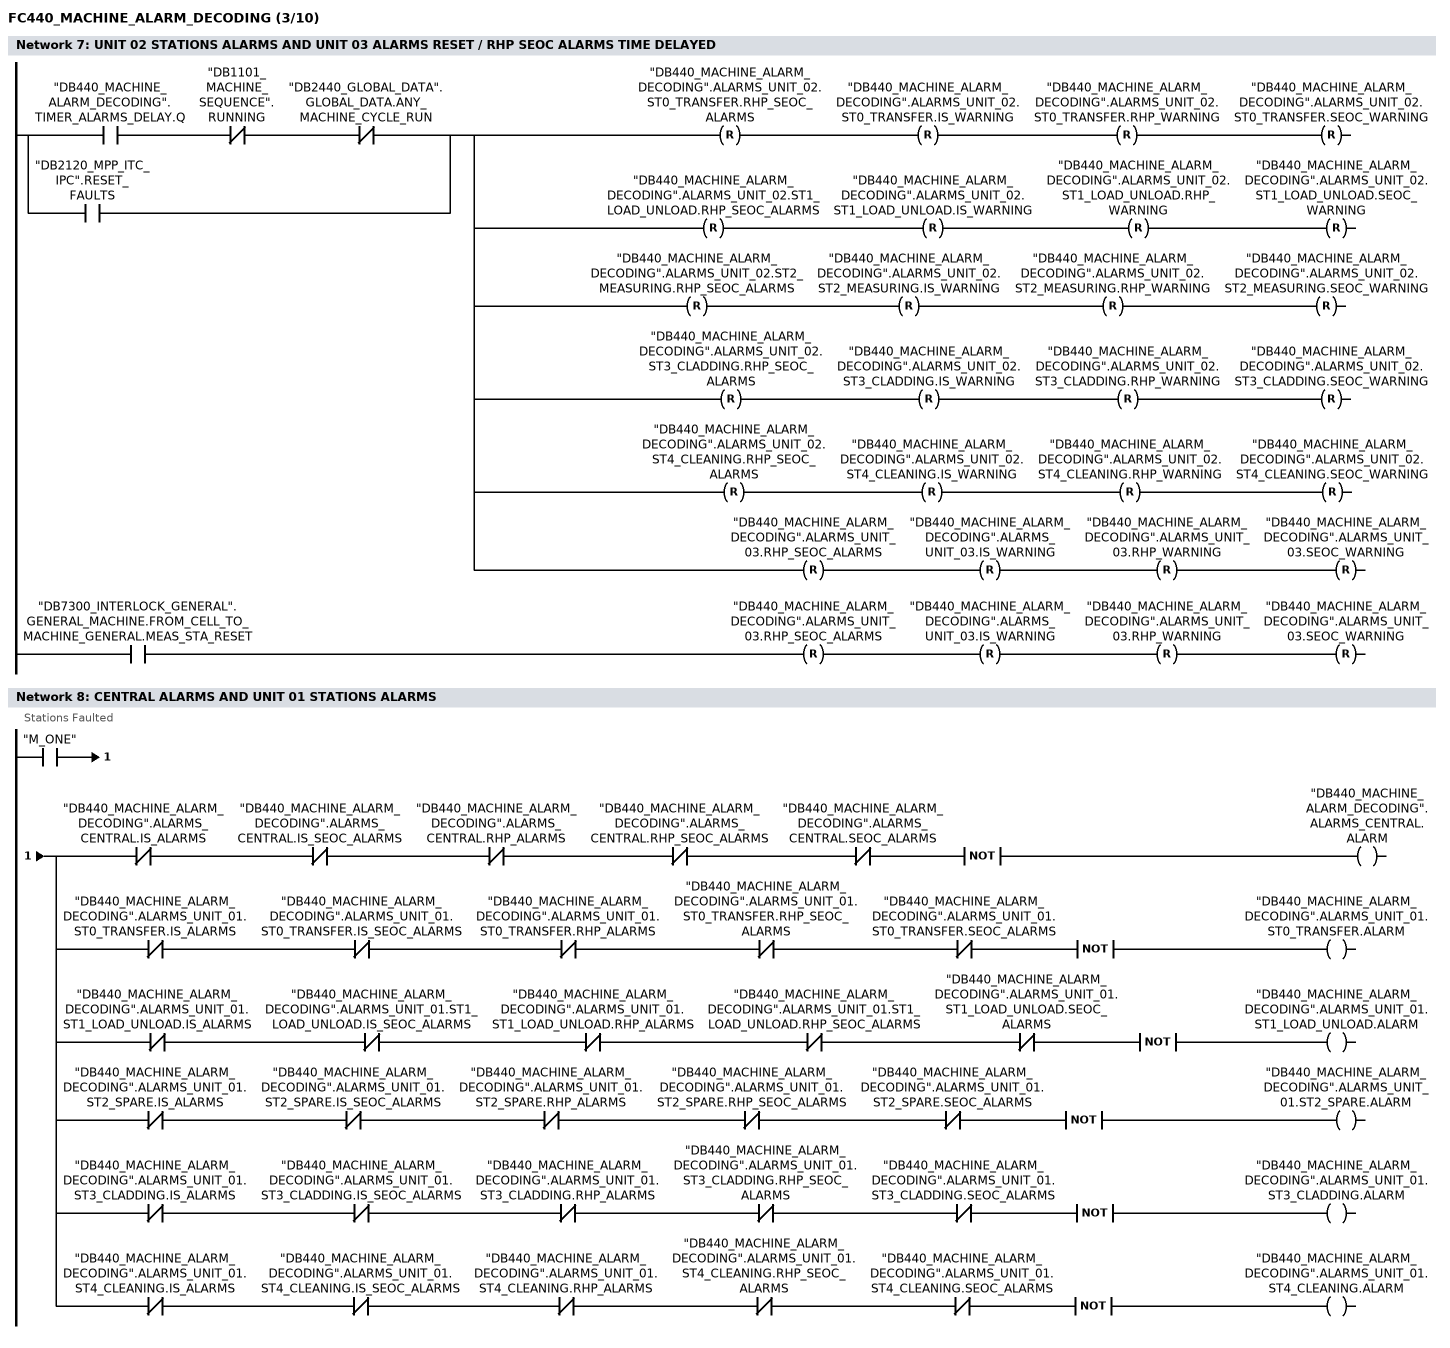
   RUNG wire#powerrail
      Contact( "DB440_MACHINE_ALARM_DECODING".TIMER_ALARMS_DELAY.Q )
      I_Contact( "DB1101_MACHINE_SEQUENCE".RUNNING )
      I_Contact( "DB2440_GLOBAL_DATA".GLOBAL_DATA.ANY_MACHINE_CYCLE_RUN )
      wire#w1
      R_Coil( "DB440_MACHINE_ALARM_DECODING".ALARMS_UNIT_02.ST0_TRANSFER.RHP_SEOC_ALARMS )
      R_Coil( "DB440_MACHINE_ALARM_DECODING".ALARMS_UNIT_02.ST0_TRANSFER.IS_WARNING )
      R_Coil( "DB440_MACHINE_ALARM_DECODING".ALARMS_UNIT_02.ST0_TRANSFER.RHP_WARNING )
      R_Coil( "DB440_MACHINE_ALARM_DECODING".ALARMS_UNIT_02.ST0_TRANSFER.SEOC_WARNING )
   END_RUNG
   RUNG wire#powerrail
      Contact( "DB2120_MPP_ITC_IPC".RESET_FAULTS )
   END_RUNG wire#w1
   RUNG wire#w1
      R_Coil( "DB440_MACHINE_ALARM_DECODING".ALARMS_UNIT_02.ST1_LOAD_UNLOAD.RHP_SEOC_ALARMS )
      R_Coil( "DB440_MACHINE_ALARM_DECODING".ALARMS_UNIT_02.ST1_LOAD_UNLOAD.IS_WARNING )
      R_Coil( "DB440_MACHINE_ALARM_DECODING".ALARMS_UNIT_02.ST1_LOAD_UNLOAD.RHP_WARNING )
      R_Coil( "DB440_MACHINE_ALARM_DECODING".ALARMS_UNIT_02.ST1_LOAD_UNLOAD.SEOC_WARNING )
   END_RUNG
   RUNG wire#w1
      R_Coil( "DB440_MACHINE_ALARM_DECODING".ALARMS_UNIT_02.ST2_MEASURING.RHP_SEOC_ALARMS )
      R_Coil( "DB440_MACHINE_ALARM_DECODING".ALARMS_UNIT_02.ST2_MEASURING.IS_WARNING )
      R_Coil( "DB440_MACHINE_ALARM_DECODING".ALARMS_UNIT_02.ST2_MEASURING.RHP_WARNING )
      R_Coil( "DB440_MACHINE_ALARM_DECODING".ALARMS_UNIT_02.ST2_MEASURING.SEOC_WARNING )
   END_RUNG
   RUNG wire#w1
      R_Coil( "DB440_MACHINE_ALARM_DECODING".ALARMS_UNIT_02.ST3_CLADDING.RHP_SEOC_ALARMS )
      R_Coil( "DB440_MACHINE_ALARM_DECODING".ALARMS_UNIT_02.ST3_CLADDING.IS_WARNING )
      R_Coil( "DB440_MACHINE_ALARM_DECODING".ALARMS_UNIT_02.ST3_CLADDING.RHP_WARNING )
      R_Coil( "DB440_MACHINE_ALARM_DECODING".ALARMS_UNIT_02.ST3_CLADDING.SEOC_WARNING )
   END_RUNG
   RUNG wire#w1
      R_Coil( "DB440_MACHINE_ALARM_DECODING".ALARMS_UNIT_02.ST4_CLEANING.RHP_SEOC_ALARMS )
      R_Coil( "DB440_MACHINE_ALARM_DECODING".ALARMS_UNIT_02.ST4_CLEANING.IS_WARNING )
      R_Coil( "DB440_MACHINE_ALARM_DECODING".ALARMS_UNIT_02.ST4_CLEANING.RHP_WARNING )
      R_Coil( "DB440_MACHINE_ALARM_DECODING".ALARMS_UNIT_02.ST4_CLEANING.SEOC_WARNING )
   END_RUNG
   RUNG wire#w1
      R_Coil( "DB440_MACHINE_ALARM_DECODING".ALARMS_UNIT_03.RHP_SEOC_ALARMS )
      R_Coil( "DB440_MACHINE_ALARM_DECODING".ALARMS_UNIT_03.IS_WARNING )
      R_Coil( "DB440_MACHINE_ALARM_DECODING".ALARMS_UNIT_03.RHP_WARNING )
      R_Coil( "DB440_MACHINE_ALARM_DECODING".ALARMS_UNIT_03.SEOC_WARNING )
   END_RUNG
   RUNG wire#powerrail
      Contact( "DB7300_INTERLOCK_GENERAL".GENERAL_MACHINE.FROM_CELL_TO_MACHINE_GENERAL.MEAS_STA_RESET )
      R_Coil( "DB440_MACHINE_ALARM_DECODING".ALARMS_UNIT_03.RHP_SEOC_ALARMS )
      R_Coil( "DB440_MACHINE_ALARM_DECODING".ALARMS_UNIT_03.IS_WARNING )
      R_Coil( "DB440_MACHINE_ALARM_DECODING".ALARMS_UNIT_03.RHP_WARNING )
      R_Coil( "DB440_MACHINE_ALARM_DECODING".ALARMS_UNIT_03.SEOC_WARNING )
   END_RUNG
   // the same network as SCL:
   IF ("DB440_MACHINE_ALARM_DECODING".TIMER_ALARMS_DELAY.Q AND NOT "DB1101_MACHINE_SEQUENCE".RUNNING AND NOT "DB2440_GLOBAL_DATA".GLOBAL_DATA.ANY_MACHINE_CYCLE_RUN) OR "DB2120_MPP_ITC_IPC".RESET_FAULTS THEN
       "DB440_MACHINE_ALARM_DECODING".ALARMS_UNIT_02.ST0_TRANSFER.RHP_SEOC_ALARMS := FALSE;
       "DB440_MACHINE_ALARM_DECODING".ALARMS_UNIT_02.ST0_TRANSFER.IS_WARNING := FALSE;
       "DB440_MACHINE_ALARM_DECODING".ALARMS_UNIT_02.ST0_TRANSFER.RHP_WARNING := FALSE;
       "DB440_MACHINE_ALARM_DECODING".ALARMS_UNIT_02.ST0_TRANSFER.SEOC_WARNING := FALSE;
       "DB440_MACHINE_ALARM_DECODING".ALARMS_UNIT_02.ST1_LOAD_UNLOAD.RHP_SEOC_ALARMS := FALSE;
       "DB440_MACHINE_ALARM_DECODING".ALARMS_UNIT_02.ST1_LOAD_UNLOAD.IS_WARNING := FALSE;
       "DB440_MACHINE_ALARM_DECODING".ALARMS_UNIT_02.ST1_LOAD_UNLOAD.RHP_WARNING := FALSE;
       "DB440_MACHINE_ALARM_DECODING".ALARMS_UNIT_02.ST1_LOAD_UNLOAD.SEOC_WARNING := FALSE;
       "DB440_MACHINE_ALARM_DECODING".ALARMS_UNIT_02.ST2_MEASURING.RHP_SEOC_ALARMS := FALSE;
       "DB440_MACHINE_ALARM_DECODING".ALARMS_UNIT_02.ST2_MEASURING.IS_WARNING := FALSE;
       "DB440_MACHINE_ALARM_DECODING".ALARMS_UNIT_02.ST2_MEASURING.RHP_WARNING := FALSE;
       "DB440_MACHINE_ALARM_DECODING".ALARMS_UNIT_02.ST2_MEASURING.SEOC_WARNING := FALSE;
       "DB440_MACHINE_ALARM_DECODING".ALARMS_UNIT_02.ST3_CLADDING.RHP_SEOC_ALARMS := FALSE;
       "DB440_MACHINE_ALARM_DECODING".ALARMS_UNIT_02.ST3_CLADDING.IS_WARNING := FALSE;
       "DB440_MACHINE_ALARM_DECODING".ALARMS_UNIT_02.ST3_CLADDING.RHP_WARNING := FALSE;
       "DB440_MACHINE_ALARM_DECODING".ALARMS_UNIT_02.ST3_CLADDING.SEOC_WARNING := FALSE;
       "DB440_MACHINE_ALARM_DECODING".ALARMS_UNIT_02.ST4_CLEANING.RHP_SEOC_ALARMS := FALSE;
       "DB440_MACHINE_ALARM_DECODING".ALARMS_UNIT_02.ST4_CLEANING.IS_WARNING := FALSE;
       "DB440_MACHINE_ALARM_DECODING".ALARMS_UNIT_02.ST4_CLEANING.RHP_WARNING := FALSE;
       "DB440_MACHINE_ALARM_DECODING".ALARMS_UNIT_02.ST4_CLEANING.SEOC_WARNING := FALSE;
       "DB440_MACHINE_ALARM_DECODING".ALARMS_UNIT_03.RHP_SEOC_ALARMS := FALSE;
       "DB440_MACHINE_ALARM_DECODING".ALARMS_UNIT_03.IS_WARNING := FALSE;
       "DB440_MACHINE_ALARM_DECODING".ALARMS_UNIT_03.RHP_WARNING := FALSE;
       "DB440_MACHINE_ALARM_DECODING".ALARMS_UNIT_03.SEOC_WARNING := FALSE;
   END_IF;
   IF "DB7300_INTERLOCK_GENERAL".GENERAL_MACHINE.FROM_CELL_TO_MACHINE_GENERAL.MEAS_STA_RESET THEN
       "DB440_MACHINE_ALARM_DECODING".ALARMS_UNIT_03.RHP_SEOC_ALARMS := FALSE;
       "DB440_MACHINE_ALARM_DECODING".ALARMS_UNIT_03.IS_WARNING := FALSE;
       "DB440_MACHINE_ALARM_DECODING".ALARMS_UNIT_03.RHP_WARNING := FALSE;
       "DB440_MACHINE_ALARM_DECODING".ALARMS_UNIT_03.SEOC_WARNING := FALSE;
   END_IF;
END_REGION

REGION Network 8: CENTRAL ALARMS AND UNIT 01 STATIONS ALARMS
   // Stations Faulted
   RUNG wire#powerrail
      Contact( "M_ONE" )
      wire#w1
      I_Contact( "DB440_MACHINE_ALARM_DECODING".ALARMS_CENTRAL.IS_ALARMS )
      I_Contact( "DB440_MACHINE_ALARM_DECODING".ALARMS_CENTRAL.IS_SEOC_ALARMS )
      I_Contact( "DB440_MACHINE_ALARM_DECODING".ALARMS_CENTRAL.RHP_ALARMS )
      I_Contact( "DB440_MACHINE_ALARM_DECODING".ALARMS_CENTRAL.RHP_SEOC_ALARMS )
      I_Contact( "DB440_MACHINE_ALARM_DECODING".ALARMS_CENTRAL.SEOC_ALARMS )
      Not()
      Coil( "DB440_MACHINE_ALARM_DECODING".ALARMS_CENTRAL.ALARM )
   END_RUNG
   RUNG wire#w1
      I_Contact( "DB440_MACHINE_ALARM_DECODING".ALARMS_UNIT_01.ST0_TRANSFER.IS_ALARMS )
      I_Contact( "DB440_MACHINE_ALARM_DECODING".ALARMS_UNIT_01.ST0_TRANSFER.IS_SEOC_ALARMS )
      I_Contact( "DB440_MACHINE_ALARM_DECODING".ALARMS_UNIT_01.ST0_TRANSFER.RHP_ALARMS )
      I_Contact( "DB440_MACHINE_ALARM_DECODING".ALARMS_UNIT_01.ST0_TRANSFER.RHP_SEOC_ALARMS )
      I_Contact( "DB440_MACHINE_ALARM_DECODING".ALARMS_UNIT_01.ST0_TRANSFER.SEOC_ALARMS )
      Not()
      Coil( "DB440_MACHINE_ALARM_DECODING".ALARMS_UNIT_01.ST0_TRANSFER.ALARM )
   END_RUNG
   RUNG wire#w1
      I_Contact( "DB440_MACHINE_ALARM_DECODING".ALARMS_UNIT_01.ST1_LOAD_UNLOAD.IS_ALARMS )
      I_Contact( "DB440_MACHINE_ALARM_DECODING".ALARMS_UNIT_01.ST1_LOAD_UNLOAD.IS_SEOC_ALARMS )
      I_Contact( "DB440_MACHINE_ALARM_DECODING".ALARMS_UNIT_01.ST1_LOAD_UNLOAD.RHP_ALARMS )
      I_Contact( "DB440_MACHINE_ALARM_DECODING".ALARMS_UNIT_01.ST1_LOAD_UNLOAD.RHP_SEOC_ALARMS )
      I_Contact( "DB440_MACHINE_ALARM_DECODING".ALARMS_UNIT_01.ST1_LOAD_UNLOAD.SEOC_ALARMS )
      Not()
      Coil( "DB440_MACHINE_ALARM_DECODING".ALARMS_UNIT_01.ST1_LOAD_UNLOAD.ALARM )
   END_RUNG
   RUNG wire#w1
      I_Contact( "DB440_MACHINE_ALARM_DECODING".ALARMS_UNIT_01.ST2_SPARE.IS_ALARMS )
      I_Contact( "DB440_MACHINE_ALARM_DECODING".ALARMS_UNIT_01.ST2_SPARE.IS_SEOC_ALARMS )
      I_Contact( "DB440_MACHINE_ALARM_DECODING".ALARMS_UNIT_01.ST2_SPARE.RHP_ALARMS )
      I_Contact( "DB440_MACHINE_ALARM_DECODING".ALARMS_UNIT_01.ST2_SPARE.RHP_SEOC_ALARMS )
      I_Contact( "DB440_MACHINE_ALARM_DECODING".ALARMS_UNIT_01.ST2_SPARE.SEOC_ALARMS )
      Not()
      Coil( "DB440_MACHINE_ALARM_DECODING".ALARMS_UNIT_01.ST2_SPARE.ALARM )
   END_RUNG
   RUNG wire#w1
      I_Contact( "DB440_MACHINE_ALARM_DECODING".ALARMS_UNIT_01.ST3_CLADDING.IS_ALARMS )
      I_Contact( "DB440_MACHINE_ALARM_DECODING".ALARMS_UNIT_01.ST3_CLADDING.IS_SEOC_ALARMS )
      I_Contact( "DB440_MACHINE_ALARM_DECODING".ALARMS_UNIT_01.ST3_CLADDING.RHP_ALARMS )
      I_Contact( "DB440_MACHINE_ALARM_DECODING".ALARMS_UNIT_01.ST3_CLADDING.RHP_SEOC_ALARMS )
      I_Contact( "DB440_MACHINE_ALARM_DECODING".ALARMS_UNIT_01.ST3_CLADDING.SEOC_ALARMS )
      Not()
      Coil( "DB440_MACHINE_ALARM_DECODING".ALARMS_UNIT_01.ST3_CLADDING.ALARM )
   END_RUNG
   RUNG wire#w1
      I_Contact( "DB440_MACHINE_ALARM_DECODING".ALARMS_UNIT_01.ST4_CLEANING.IS_ALARMS )
      I_Contact( "DB440_MACHINE_ALARM_DECODING".ALARMS_UNIT_01.ST4_CLEANING.IS_SEOC_ALARMS )
      I_Contact( "DB440_MACHINE_ALARM_DECODING".ALARMS_UNIT_01.ST4_CLEANING.RHP_ALARMS )
      I_Contact( "DB440_MACHINE_ALARM_DECODING".ALARMS_UNIT_01.ST4_CLEANING.RHP_SEOC_ALARMS )
      I_Contact( "DB440_MACHINE_ALARM_DECODING".ALARMS_UNIT_01.ST4_CLEANING.SEOC_ALARMS )
      Not()
      Coil( "DB440_MACHINE_ALARM_DECODING".ALARMS_UNIT_01.ST4_CLEANING.ALARM )
   END_RUNG
   // the same network as SCL:
   "DB440_MACHINE_ALARM_DECODING".ALARMS_CENTRAL.ALARM := NOT ("M_ONE" AND NOT "DB440_MACHINE_ALARM_DECODING".ALARMS_CENTRAL.IS_ALARMS AND NOT "DB440_MACHINE_ALARM_DECODING".ALARMS_CENTRAL.IS_SEOC_ALARMS AND NOT "DB440_MACHINE_ALARM_DECODING".ALARMS_CENTRAL.RHP_ALARMS AND NOT "DB440_MACHINE_ALARM_DECODING".ALARMS_CENTRAL.RHP_SEOC_ALARMS AND NOT "DB440_MACHINE_ALARM_DECODING".ALARMS_CENTRAL.SEOC_ALARMS);
   "DB440_MACHINE_ALARM_DECODING".ALARMS_UNIT_01.ST0_TRANSFER.ALARM := NOT ("M_ONE" AND NOT "DB440_MACHINE_ALARM_DECODING".ALARMS_UNIT_01.ST0_TRANSFER.IS_ALARMS AND NOT "DB440_MACHINE_ALARM_DECODING".ALARMS_UNIT_01.ST0_TRANSFER.IS_SEOC_ALARMS AND NOT "DB440_MACHINE_ALARM_DECODING".ALARMS_UNIT_01.ST0_TRANSFER.RHP_ALARMS AND NOT "DB440_MACHINE_ALARM_DECODING".ALARMS_UNIT_01.ST0_TRANSFER.RHP_SEOC_ALARMS AND NOT "DB440_MACHINE_ALARM_DECODING".ALARMS_UNIT_01.ST0_TRANSFER.SEOC_ALARMS);
   "DB440_MACHINE_ALARM_DECODING".ALARMS_UNIT_01.ST1_LOAD_UNLOAD.ALARM := NOT ("M_ONE" AND NOT "DB440_MACHINE_ALARM_DECODING".ALARMS_UNIT_01.ST1_LOAD_UNLOAD.IS_ALARMS AND NOT "DB440_MACHINE_ALARM_DECODING".ALARMS_UNIT_01.ST1_LOAD_UNLOAD.IS_SEOC_ALARMS AND NOT "DB440_MACHINE_ALARM_DECODING".ALARMS_UNIT_01.ST1_LOAD_UNLOAD.RHP_ALARMS AND NOT "DB440_MACHINE_ALARM_DECODING".ALARMS_UNIT_01.ST1_LOAD_UNLOAD.RHP_SEOC_ALARMS AND NOT "DB440_MACHINE_ALARM_DECODING".ALARMS_UNIT_01.ST1_LOAD_UNLOAD.SEOC_ALARMS);
   "DB440_MACHINE_ALARM_DECODING".ALARMS_UNIT_01.ST2_SPARE.ALARM := NOT ("M_ONE" AND NOT "DB440_MACHINE_ALARM_DECODING".ALARMS_UNIT_01.ST2_SPARE.IS_ALARMS AND NOT "DB440_MACHINE_ALARM_DECODING".ALARMS_UNIT_01.ST2_SPARE.IS_SEOC_ALARMS AND NOT "DB440_MACHINE_ALARM_DECODING".ALARMS_UNIT_01.ST2_SPARE.RHP_ALARMS AND NOT "DB440_MACHINE_ALARM_DECODING".ALARMS_UNIT_01.ST2_SPARE.RHP_SEOC_ALARMS AND NOT "DB440_MACHINE_ALARM_DECODING".ALARMS_UNIT_01.ST2_SPARE.SEOC_ALARMS);
   "DB440_MACHINE_ALARM_DECODING".ALARMS_UNIT_01.ST3_CLADDING.ALARM := NOT ("M_ONE" AND NOT "DB440_MACHINE_ALARM_DECODING".ALARMS_UNIT_01.ST3_CLADDING.IS_ALARMS AND NOT "DB440_MACHINE_ALARM_DECODING".ALARMS_UNIT_01.ST3_CLADDING.IS_SEOC_ALARMS AND NOT "DB440_MACHINE_ALARM_DECODING".ALARMS_UNIT_01.ST3_CLADDING.RHP_ALARMS AND NOT "DB440_MACHINE_ALARM_DECODING".ALARMS_UNIT_01.ST3_CLADDING.RHP_SEOC_ALARMS AND NOT "DB440_MACHINE_ALARM_DECODING".ALARMS_UNIT_01.ST3_CLADDING.SEOC_ALARMS);
   "DB440_MACHINE_ALARM_DECODING".ALARMS_UNIT_01.ST4_CLEANING.ALARM := NOT ("M_ONE" AND NOT "DB440_MACHINE_ALARM_DECODING".ALARMS_UNIT_01.ST4_CLEANING.IS_ALARMS AND NOT "DB440_MACHINE_ALARM_DECODING".ALARMS_UNIT_01.ST4_CLEANING.IS_SEOC_ALARMS AND NOT "DB440_MACHINE_ALARM_DECODING".ALARMS_UNIT_01.ST4_CLEANING.RHP_ALARMS AND NOT "DB440_MACHINE_ALARM_DECODING".ALARMS_UNIT_01.ST4_CLEANING.RHP_SEOC_ALARMS AND NOT "DB440_MACHINE_ALARM_DECODING".ALARMS_UNIT_01.ST4_CLEANING.SEOC_ALARMS);
END_REGION

REGION Network 9: UNIT 02 STATIONS ALARMS AND UNIT 03 ALARMS
   // Stations Faulted
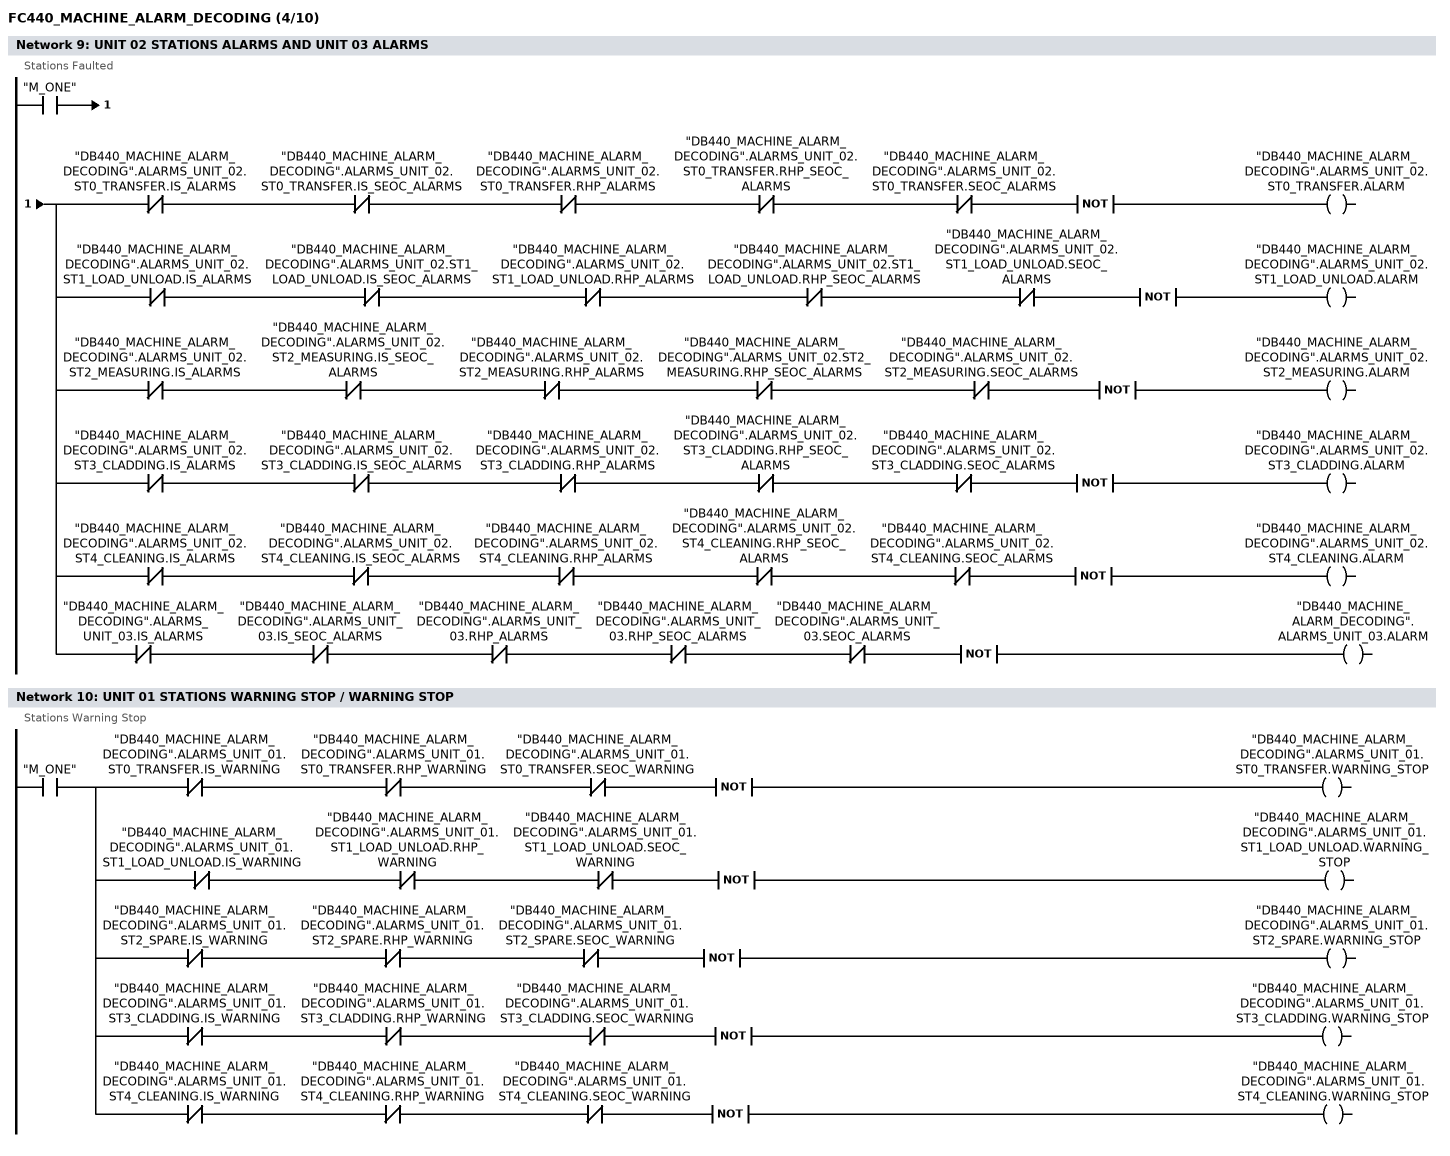
   RUNG wire#powerrail
      Contact( "M_ONE" )
      wire#w1
      I_Contact( "DB440_MACHINE_ALARM_DECODING".ALARMS_UNIT_02.ST0_TRANSFER.IS_ALARMS )
      I_Contact( "DB440_MACHINE_ALARM_DECODING".ALARMS_UNIT_02.ST0_TRANSFER.IS_SEOC_ALARMS )
      I_Contact( "DB440_MACHINE_ALARM_DECODING".ALARMS_UNIT_02.ST0_TRANSFER.RHP_ALARMS )
      I_Contact( "DB440_MACHINE_ALARM_DECODING".ALARMS_UNIT_02.ST0_TRANSFER.RHP_SEOC_ALARMS )
      I_Contact( "DB440_MACHINE_ALARM_DECODING".ALARMS_UNIT_02.ST0_TRANSFER.SEOC_ALARMS )
      Not()
      Coil( "DB440_MACHINE_ALARM_DECODING".ALARMS_UNIT_02.ST0_TRANSFER.ALARM )
   END_RUNG
   RUNG wire#w1
      I_Contact( "DB440_MACHINE_ALARM_DECODING".ALARMS_UNIT_02.ST1_LOAD_UNLOAD.IS_ALARMS )
      I_Contact( "DB440_MACHINE_ALARM_DECODING".ALARMS_UNIT_02.ST1_LOAD_UNLOAD.IS_SEOC_ALARMS )
      I_Contact( "DB440_MACHINE_ALARM_DECODING".ALARMS_UNIT_02.ST1_LOAD_UNLOAD.RHP_ALARMS )
      I_Contact( "DB440_MACHINE_ALARM_DECODING".ALARMS_UNIT_02.ST1_LOAD_UNLOAD.RHP_SEOC_ALARMS )
      I_Contact( "DB440_MACHINE_ALARM_DECODING".ALARMS_UNIT_02.ST1_LOAD_UNLOAD.SEOC_ALARMS )
      Not()
      Coil( "DB440_MACHINE_ALARM_DECODING".ALARMS_UNIT_02.ST1_LOAD_UNLOAD.ALARM )
   END_RUNG
   RUNG wire#w1
      I_Contact( "DB440_MACHINE_ALARM_DECODING".ALARMS_UNIT_02.ST2_MEASURING.IS_ALARMS )
      I_Contact( "DB440_MACHINE_ALARM_DECODING".ALARMS_UNIT_02.ST2_MEASURING.IS_SEOC_ALARMS )
      I_Contact( "DB440_MACHINE_ALARM_DECODING".ALARMS_UNIT_02.ST2_MEASURING.RHP_ALARMS )
      I_Contact( "DB440_MACHINE_ALARM_DECODING".ALARMS_UNIT_02.ST2_MEASURING.RHP_SEOC_ALARMS )
      I_Contact( "DB440_MACHINE_ALARM_DECODING".ALARMS_UNIT_02.ST2_MEASURING.SEOC_ALARMS )
      Not()
      Coil( "DB440_MACHINE_ALARM_DECODING".ALARMS_UNIT_02.ST2_MEASURING.ALARM )
   END_RUNG
   RUNG wire#w1
      I_Contact( "DB440_MACHINE_ALARM_DECODING".ALARMS_UNIT_02.ST3_CLADDING.IS_ALARMS )
      I_Contact( "DB440_MACHINE_ALARM_DECODING".ALARMS_UNIT_02.ST3_CLADDING.IS_SEOC_ALARMS )
      I_Contact( "DB440_MACHINE_ALARM_DECODING".ALARMS_UNIT_02.ST3_CLADDING.RHP_ALARMS )
      I_Contact( "DB440_MACHINE_ALARM_DECODING".ALARMS_UNIT_02.ST3_CLADDING.RHP_SEOC_ALARMS )
      I_Contact( "DB440_MACHINE_ALARM_DECODING".ALARMS_UNIT_02.ST3_CLADDING.SEOC_ALARMS )
      Not()
      Coil( "DB440_MACHINE_ALARM_DECODING".ALARMS_UNIT_02.ST3_CLADDING.ALARM )
   END_RUNG
   RUNG wire#w1
      I_Contact( "DB440_MACHINE_ALARM_DECODING".ALARMS_UNIT_02.ST4_CLEANING.IS_ALARMS )
      I_Contact( "DB440_MACHINE_ALARM_DECODING".ALARMS_UNIT_02.ST4_CLEANING.IS_SEOC_ALARMS )
      I_Contact( "DB440_MACHINE_ALARM_DECODING".ALARMS_UNIT_02.ST4_CLEANING.RHP_ALARMS )
      I_Contact( "DB440_MACHINE_ALARM_DECODING".ALARMS_UNIT_02.ST4_CLEANING.RHP_SEOC_ALARMS )
      I_Contact( "DB440_MACHINE_ALARM_DECODING".ALARMS_UNIT_02.ST4_CLEANING.SEOC_ALARMS )
      Not()
      Coil( "DB440_MACHINE_ALARM_DECODING".ALARMS_UNIT_02.ST4_CLEANING.ALARM )
   END_RUNG
   RUNG wire#w1
      I_Contact( "DB440_MACHINE_ALARM_DECODING".ALARMS_UNIT_03.IS_ALARMS )
      I_Contact( "DB440_MACHINE_ALARM_DECODING".ALARMS_UNIT_03.IS_SEOC_ALARMS )
      I_Contact( "DB440_MACHINE_ALARM_DECODING".ALARMS_UNIT_03.RHP_ALARMS )
      I_Contact( "DB440_MACHINE_ALARM_DECODING".ALARMS_UNIT_03.RHP_SEOC_ALARMS )
      I_Contact( "DB440_MACHINE_ALARM_DECODING".ALARMS_UNIT_03.SEOC_ALARMS )
      Not()
      Coil( "DB440_MACHINE_ALARM_DECODING".ALARMS_UNIT_03.ALARM )
   END_RUNG
   // the same network as SCL:
   "DB440_MACHINE_ALARM_DECODING".ALARMS_UNIT_02.ST0_TRANSFER.ALARM := NOT ("M_ONE" AND NOT "DB440_MACHINE_ALARM_DECODING".ALARMS_UNIT_02.ST0_TRANSFER.IS_ALARMS AND NOT "DB440_MACHINE_ALARM_DECODING".ALARMS_UNIT_02.ST0_TRANSFER.IS_SEOC_ALARMS AND NOT "DB440_MACHINE_ALARM_DECODING".ALARMS_UNIT_02.ST0_TRANSFER.RHP_ALARMS AND NOT "DB440_MACHINE_ALARM_DECODING".ALARMS_UNIT_02.ST0_TRANSFER.RHP_SEOC_ALARMS AND NOT "DB440_MACHINE_ALARM_DECODING".ALARMS_UNIT_02.ST0_TRANSFER.SEOC_ALARMS);
   "DB440_MACHINE_ALARM_DECODING".ALARMS_UNIT_02.ST1_LOAD_UNLOAD.ALARM := NOT ("M_ONE" AND NOT "DB440_MACHINE_ALARM_DECODING".ALARMS_UNIT_02.ST1_LOAD_UNLOAD.IS_ALARMS AND NOT "DB440_MACHINE_ALARM_DECODING".ALARMS_UNIT_02.ST1_LOAD_UNLOAD.IS_SEOC_ALARMS AND NOT "DB440_MACHINE_ALARM_DECODING".ALARMS_UNIT_02.ST1_LOAD_UNLOAD.RHP_ALARMS AND NOT "DB440_MACHINE_ALARM_DECODING".ALARMS_UNIT_02.ST1_LOAD_UNLOAD.RHP_SEOC_ALARMS AND NOT "DB440_MACHINE_ALARM_DECODING".ALARMS_UNIT_02.ST1_LOAD_UNLOAD.SEOC_ALARMS);
   "DB440_MACHINE_ALARM_DECODING".ALARMS_UNIT_02.ST2_MEASURING.ALARM := NOT ("M_ONE" AND NOT "DB440_MACHINE_ALARM_DECODING".ALARMS_UNIT_02.ST2_MEASURING.IS_ALARMS AND NOT "DB440_MACHINE_ALARM_DECODING".ALARMS_UNIT_02.ST2_MEASURING.IS_SEOC_ALARMS AND NOT "DB440_MACHINE_ALARM_DECODING".ALARMS_UNIT_02.ST2_MEASURING.RHP_ALARMS AND NOT "DB440_MACHINE_ALARM_DECODING".ALARMS_UNIT_02.ST2_MEASURING.RHP_SEOC_ALARMS AND NOT "DB440_MACHINE_ALARM_DECODING".ALARMS_UNIT_02.ST2_MEASURING.SEOC_ALARMS);
   "DB440_MACHINE_ALARM_DECODING".ALARMS_UNIT_02.ST3_CLADDING.ALARM := NOT ("M_ONE" AND NOT "DB440_MACHINE_ALARM_DECODING".ALARMS_UNIT_02.ST3_CLADDING.IS_ALARMS AND NOT "DB440_MACHINE_ALARM_DECODING".ALARMS_UNIT_02.ST3_CLADDING.IS_SEOC_ALARMS AND NOT "DB440_MACHINE_ALARM_DECODING".ALARMS_UNIT_02.ST3_CLADDING.RHP_ALARMS AND NOT "DB440_MACHINE_ALARM_DECODING".ALARMS_UNIT_02.ST3_CLADDING.RHP_SEOC_ALARMS AND NOT "DB440_MACHINE_ALARM_DECODING".ALARMS_UNIT_02.ST3_CLADDING.SEOC_ALARMS);
   "DB440_MACHINE_ALARM_DECODING".ALARMS_UNIT_02.ST4_CLEANING.ALARM := NOT ("M_ONE" AND NOT "DB440_MACHINE_ALARM_DECODING".ALARMS_UNIT_02.ST4_CLEANING.IS_ALARMS AND NOT "DB440_MACHINE_ALARM_DECODING".ALARMS_UNIT_02.ST4_CLEANING.IS_SEOC_ALARMS AND NOT "DB440_MACHINE_ALARM_DECODING".ALARMS_UNIT_02.ST4_CLEANING.RHP_ALARMS AND NOT "DB440_MACHINE_ALARM_DECODING".ALARMS_UNIT_02.ST4_CLEANING.RHP_SEOC_ALARMS AND NOT "DB440_MACHINE_ALARM_DECODING".ALARMS_UNIT_02.ST4_CLEANING.SEOC_ALARMS);
   "DB440_MACHINE_ALARM_DECODING".ALARMS_UNIT_03.ALARM := NOT ("M_ONE" AND NOT "DB440_MACHINE_ALARM_DECODING".ALARMS_UNIT_03.IS_ALARMS AND NOT "DB440_MACHINE_ALARM_DECODING".ALARMS_UNIT_03.IS_SEOC_ALARMS AND NOT "DB440_MACHINE_ALARM_DECODING".ALARMS_UNIT_03.RHP_ALARMS AND NOT "DB440_MACHINE_ALARM_DECODING".ALARMS_UNIT_03.RHP_SEOC_ALARMS AND NOT "DB440_MACHINE_ALARM_DECODING".ALARMS_UNIT_03.SEOC_ALARMS);
END_REGION

REGION Network 10: UNIT 01 STATIONS WARNING STOP / WARNING STOP
   // Stations Warning Stop
   RUNG wire#powerrail
      Contact( "M_ONE" )
      wire#w1
      I_Contact( "DB440_MACHINE_ALARM_DECODING".ALARMS_UNIT_01.ST0_TRANSFER.IS_WARNING )
      I_Contact( "DB440_MACHINE_ALARM_DECODING".ALARMS_UNIT_01.ST0_TRANSFER.RHP_WARNING )
      I_Contact( "DB440_MACHINE_ALARM_DECODING".ALARMS_UNIT_01.ST0_TRANSFER.SEOC_WARNING )
      Not()
      Coil( "DB440_MACHINE_ALARM_DECODING".ALARMS_UNIT_01.ST0_TRANSFER.WARNING_STOP )
   END_RUNG
   RUNG wire#w1
      I_Contact( "DB440_MACHINE_ALARM_DECODING".ALARMS_UNIT_01.ST1_LOAD_UNLOAD.IS_WARNING )
      I_Contact( "DB440_MACHINE_ALARM_DECODING".ALARMS_UNIT_01.ST1_LOAD_UNLOAD.RHP_WARNING )
      I_Contact( "DB440_MACHINE_ALARM_DECODING".ALARMS_UNIT_01.ST1_LOAD_UNLOAD.SEOC_WARNING )
      Not()
      Coil( "DB440_MACHINE_ALARM_DECODING".ALARMS_UNIT_01.ST1_LOAD_UNLOAD.WARNING_STOP )
   END_RUNG
   RUNG wire#w1
      I_Contact( "DB440_MACHINE_ALARM_DECODING".ALARMS_UNIT_01.ST2_SPARE.IS_WARNING )
      I_Contact( "DB440_MACHINE_ALARM_DECODING".ALARMS_UNIT_01.ST2_SPARE.RHP_WARNING )
      I_Contact( "DB440_MACHINE_ALARM_DECODING".ALARMS_UNIT_01.ST2_SPARE.SEOC_WARNING )
      Not()
      Coil( "DB440_MACHINE_ALARM_DECODING".ALARMS_UNIT_01.ST2_SPARE.WARNING_STOP )
   END_RUNG
   RUNG wire#w1
      I_Contact( "DB440_MACHINE_ALARM_DECODING".ALARMS_UNIT_01.ST3_CLADDING.IS_WARNING )
      I_Contact( "DB440_MACHINE_ALARM_DECODING".ALARMS_UNIT_01.ST3_CLADDING.RHP_WARNING )
      I_Contact( "DB440_MACHINE_ALARM_DECODING".ALARMS_UNIT_01.ST3_CLADDING.SEOC_WARNING )
      Not()
      Coil( "DB440_MACHINE_ALARM_DECODING".ALARMS_UNIT_01.ST3_CLADDING.WARNING_STOP )
   END_RUNG
   RUNG wire#w1
      I_Contact( "DB440_MACHINE_ALARM_DECODING".ALARMS_UNIT_01.ST4_CLEANING.IS_WARNING )
      I_Contact( "DB440_MACHINE_ALARM_DECODING".ALARMS_UNIT_01.ST4_CLEANING.RHP_WARNING )
      I_Contact( "DB440_MACHINE_ALARM_DECODING".ALARMS_UNIT_01.ST4_CLEANING.SEOC_WARNING )
      Not()
      Coil( "DB440_MACHINE_ALARM_DECODING".ALARMS_UNIT_01.ST4_CLEANING.WARNING_STOP )
   END_RUNG
   // the same network as SCL:
   "DB440_MACHINE_ALARM_DECODING".ALARMS_UNIT_01.ST0_TRANSFER.WARNING_STOP := NOT ("M_ONE" AND NOT "DB440_MACHINE_ALARM_DECODING".ALARMS_UNIT_01.ST0_TRANSFER.IS_WARNING AND NOT "DB440_MACHINE_ALARM_DECODING".ALARMS_UNIT_01.ST0_TRANSFER.RHP_WARNING AND NOT "DB440_MACHINE_ALARM_DECODING".ALARMS_UNIT_01.ST0_TRANSFER.SEOC_WARNING);
   "DB440_MACHINE_ALARM_DECODING".ALARMS_UNIT_01.ST1_LOAD_UNLOAD.WARNING_STOP := NOT ("M_ONE" AND NOT "DB440_MACHINE_ALARM_DECODING".ALARMS_UNIT_01.ST1_LOAD_UNLOAD.IS_WARNING AND NOT "DB440_MACHINE_ALARM_DECODING".ALARMS_UNIT_01.ST1_LOAD_UNLOAD.RHP_WARNING AND NOT "DB440_MACHINE_ALARM_DECODING".ALARMS_UNIT_01.ST1_LOAD_UNLOAD.SEOC_WARNING);
   "DB440_MACHINE_ALARM_DECODING".ALARMS_UNIT_01.ST2_SPARE.WARNING_STOP := NOT ("M_ONE" AND NOT "DB440_MACHINE_ALARM_DECODING".ALARMS_UNIT_01.ST2_SPARE.IS_WARNING AND NOT "DB440_MACHINE_ALARM_DECODING".ALARMS_UNIT_01.ST2_SPARE.RHP_WARNING AND NOT "DB440_MACHINE_ALARM_DECODING".ALARMS_UNIT_01.ST2_SPARE.SEOC_WARNING);
   "DB440_MACHINE_ALARM_DECODING".ALARMS_UNIT_01.ST3_CLADDING.WARNING_STOP := NOT ("M_ONE" AND NOT "DB440_MACHINE_ALARM_DECODING".ALARMS_UNIT_01.ST3_CLADDING.IS_WARNING AND NOT "DB440_MACHINE_ALARM_DECODING".ALARMS_UNIT_01.ST3_CLADDING.RHP_WARNING AND NOT "DB440_MACHINE_ALARM_DECODING".ALARMS_UNIT_01.ST3_CLADDING.SEOC_WARNING);
   "DB440_MACHINE_ALARM_DECODING".ALARMS_UNIT_01.ST4_CLEANING.WARNING_STOP := NOT ("M_ONE" AND NOT "DB440_MACHINE_ALARM_DECODING".ALARMS_UNIT_01.ST4_CLEANING.IS_WARNING AND NOT "DB440_MACHINE_ALARM_DECODING".ALARMS_UNIT_01.ST4_CLEANING.RHP_WARNING AND NOT "DB440_MACHINE_ALARM_DECODING".ALARMS_UNIT_01.ST4_CLEANING.SEOC_WARNING);
END_REGION

REGION Network 11: UNIT 02 STATIONS WARNING AND UNIT 03 WARNINGS STOP / WARNING STOP
   // Stations Warning Stop
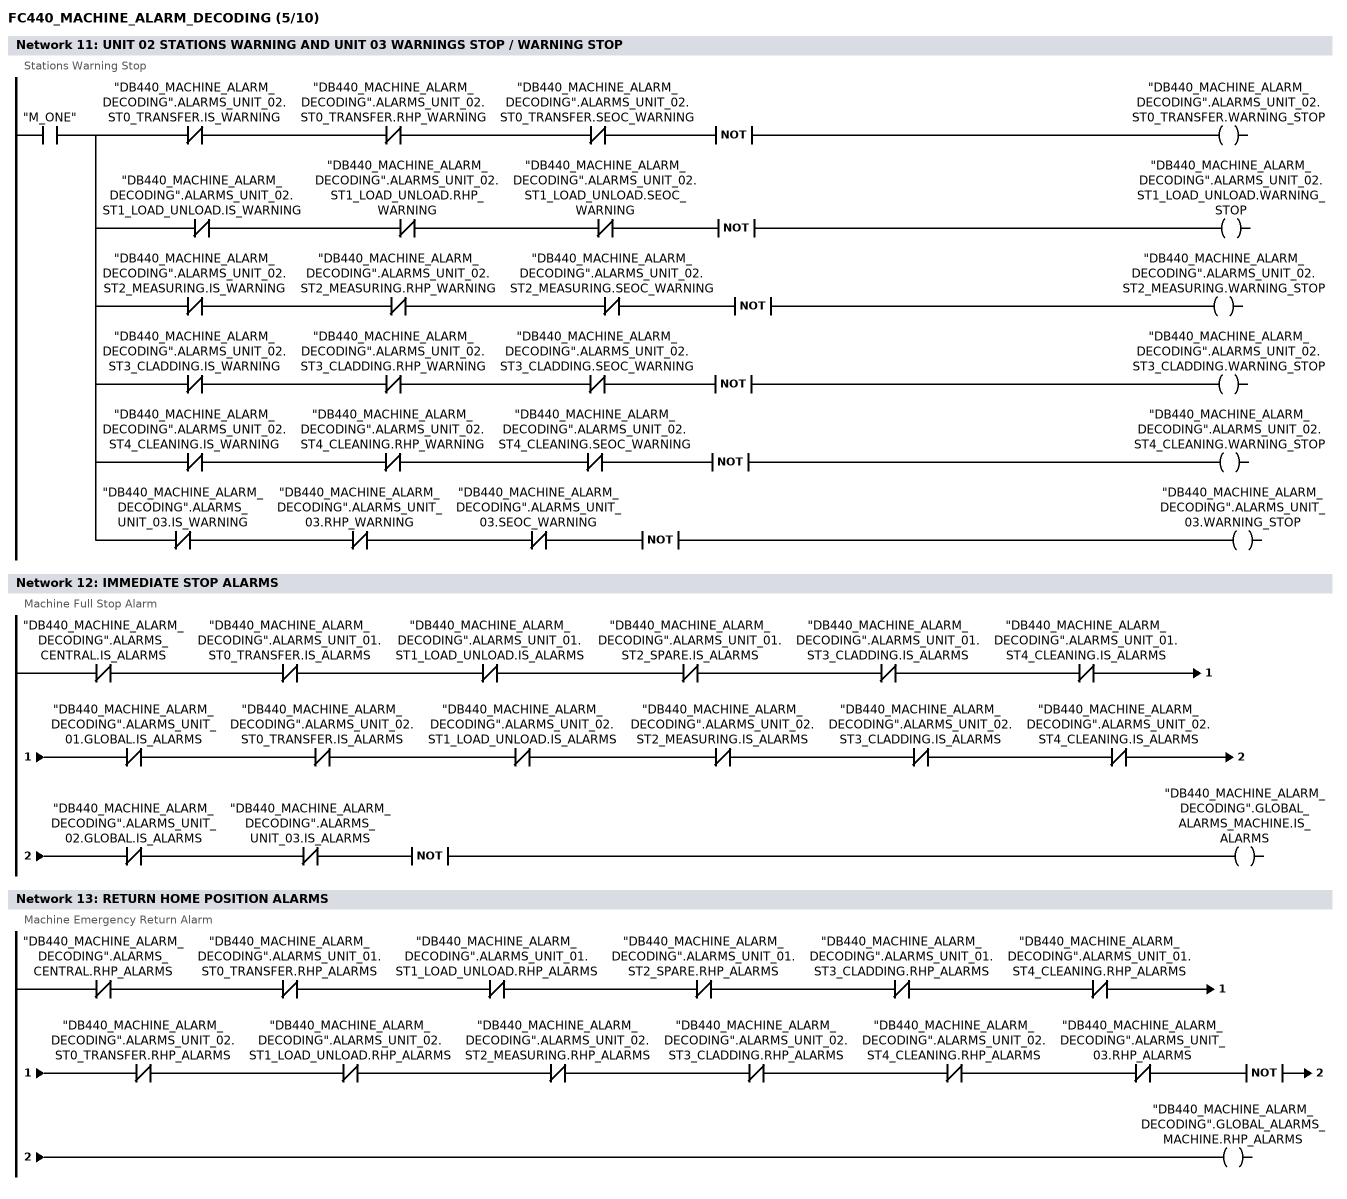
   RUNG wire#powerrail
      Contact( "M_ONE" )
      wire#w1
      I_Contact( "DB440_MACHINE_ALARM_DECODING".ALARMS_UNIT_02.ST0_TRANSFER.IS_WARNING )
      I_Contact( "DB440_MACHINE_ALARM_DECODING".ALARMS_UNIT_02.ST0_TRANSFER.RHP_WARNING )
      I_Contact( "DB440_MACHINE_ALARM_DECODING".ALARMS_UNIT_02.ST0_TRANSFER.SEOC_WARNING )
      Not()
      Coil( "DB440_MACHINE_ALARM_DECODING".ALARMS_UNIT_02.ST0_TRANSFER.WARNING_STOP )
   END_RUNG
   RUNG wire#w1
      I_Contact( "DB440_MACHINE_ALARM_DECODING".ALARMS_UNIT_02.ST1_LOAD_UNLOAD.IS_WARNING )
      I_Contact( "DB440_MACHINE_ALARM_DECODING".ALARMS_UNIT_02.ST1_LOAD_UNLOAD.RHP_WARNING )
      I_Contact( "DB440_MACHINE_ALARM_DECODING".ALARMS_UNIT_02.ST1_LOAD_UNLOAD.SEOC_WARNING )
      Not()
      Coil( "DB440_MACHINE_ALARM_DECODING".ALARMS_UNIT_02.ST1_LOAD_UNLOAD.WARNING_STOP )
   END_RUNG
   RUNG wire#w1
      I_Contact( "DB440_MACHINE_ALARM_DECODING".ALARMS_UNIT_02.ST2_MEASURING.IS_WARNING )
      I_Contact( "DB440_MACHINE_ALARM_DECODING".ALARMS_UNIT_02.ST2_MEASURING.RHP_WARNING )
      I_Contact( "DB440_MACHINE_ALARM_DECODING".ALARMS_UNIT_02.ST2_MEASURING.SEOC_WARNING )
      Not()
      Coil( "DB440_MACHINE_ALARM_DECODING".ALARMS_UNIT_02.ST2_MEASURING.WARNING_STOP )
   END_RUNG
   RUNG wire#w1
      I_Contact( "DB440_MACHINE_ALARM_DECODING".ALARMS_UNIT_02.ST3_CLADDING.IS_WARNING )
      I_Contact( "DB440_MACHINE_ALARM_DECODING".ALARMS_UNIT_02.ST3_CLADDING.RHP_WARNING )
      I_Contact( "DB440_MACHINE_ALARM_DECODING".ALARMS_UNIT_02.ST3_CLADDING.SEOC_WARNING )
      Not()
      Coil( "DB440_MACHINE_ALARM_DECODING".ALARMS_UNIT_02.ST3_CLADDING.WARNING_STOP )
   END_RUNG
   RUNG wire#w1
      I_Contact( "DB440_MACHINE_ALARM_DECODING".ALARMS_UNIT_02.ST4_CLEANING.IS_WARNING )
      I_Contact( "DB440_MACHINE_ALARM_DECODING".ALARMS_UNIT_02.ST4_CLEANING.RHP_WARNING )
      I_Contact( "DB440_MACHINE_ALARM_DECODING".ALARMS_UNIT_02.ST4_CLEANING.SEOC_WARNING )
      Not()
      Coil( "DB440_MACHINE_ALARM_DECODING".ALARMS_UNIT_02.ST4_CLEANING.WARNING_STOP )
   END_RUNG
   RUNG wire#w1
      I_Contact( "DB440_MACHINE_ALARM_DECODING".ALARMS_UNIT_03.IS_WARNING )
      I_Contact( "DB440_MACHINE_ALARM_DECODING".ALARMS_UNIT_03.RHP_WARNING )
      I_Contact( "DB440_MACHINE_ALARM_DECODING".ALARMS_UNIT_03.SEOC_WARNING )
      Not()
      Coil( "DB440_MACHINE_ALARM_DECODING".ALARMS_UNIT_03.WARNING_STOP )
   END_RUNG
   // the same network as SCL:
   "DB440_MACHINE_ALARM_DECODING".ALARMS_UNIT_02.ST0_TRANSFER.WARNING_STOP := NOT ("M_ONE" AND NOT "DB440_MACHINE_ALARM_DECODING".ALARMS_UNIT_02.ST0_TRANSFER.IS_WARNING AND NOT "DB440_MACHINE_ALARM_DECODING".ALARMS_UNIT_02.ST0_TRANSFER.RHP_WARNING AND NOT "DB440_MACHINE_ALARM_DECODING".ALARMS_UNIT_02.ST0_TRANSFER.SEOC_WARNING);
   "DB440_MACHINE_ALARM_DECODING".ALARMS_UNIT_02.ST1_LOAD_UNLOAD.WARNING_STOP := NOT ("M_ONE" AND NOT "DB440_MACHINE_ALARM_DECODING".ALARMS_UNIT_02.ST1_LOAD_UNLOAD.IS_WARNING AND NOT "DB440_MACHINE_ALARM_DECODING".ALARMS_UNIT_02.ST1_LOAD_UNLOAD.RHP_WARNING AND NOT "DB440_MACHINE_ALARM_DECODING".ALARMS_UNIT_02.ST1_LOAD_UNLOAD.SEOC_WARNING);
   "DB440_MACHINE_ALARM_DECODING".ALARMS_UNIT_02.ST2_MEASURING.WARNING_STOP := NOT ("M_ONE" AND NOT "DB440_MACHINE_ALARM_DECODING".ALARMS_UNIT_02.ST2_MEASURING.IS_WARNING AND NOT "DB440_MACHINE_ALARM_DECODING".ALARMS_UNIT_02.ST2_MEASURING.RHP_WARNING AND NOT "DB440_MACHINE_ALARM_DECODING".ALARMS_UNIT_02.ST2_MEASURING.SEOC_WARNING);
   "DB440_MACHINE_ALARM_DECODING".ALARMS_UNIT_02.ST3_CLADDING.WARNING_STOP := NOT ("M_ONE" AND NOT "DB440_MACHINE_ALARM_DECODING".ALARMS_UNIT_02.ST3_CLADDING.IS_WARNING AND NOT "DB440_MACHINE_ALARM_DECODING".ALARMS_UNIT_02.ST3_CLADDING.RHP_WARNING AND NOT "DB440_MACHINE_ALARM_DECODING".ALARMS_UNIT_02.ST3_CLADDING.SEOC_WARNING);
   "DB440_MACHINE_ALARM_DECODING".ALARMS_UNIT_02.ST4_CLEANING.WARNING_STOP := NOT ("M_ONE" AND NOT "DB440_MACHINE_ALARM_DECODING".ALARMS_UNIT_02.ST4_CLEANING.IS_WARNING AND NOT "DB440_MACHINE_ALARM_DECODING".ALARMS_UNIT_02.ST4_CLEANING.RHP_WARNING AND NOT "DB440_MACHINE_ALARM_DECODING".ALARMS_UNIT_02.ST4_CLEANING.SEOC_WARNING);
   "DB440_MACHINE_ALARM_DECODING".ALARMS_UNIT_03.WARNING_STOP := NOT ("M_ONE" AND NOT "DB440_MACHINE_ALARM_DECODING".ALARMS_UNIT_03.IS_WARNING AND NOT "DB440_MACHINE_ALARM_DECODING".ALARMS_UNIT_03.RHP_WARNING AND NOT "DB440_MACHINE_ALARM_DECODING".ALARMS_UNIT_03.SEOC_WARNING);
END_REGION

REGION Network 12: IMMEDIATE STOP ALARMS
   // Machine Full Stop Alarm
   RUNG wire#powerrail
      I_Contact( "DB440_MACHINE_ALARM_DECODING".ALARMS_CENTRAL.IS_ALARMS )
      I_Contact( "DB440_MACHINE_ALARM_DECODING".ALARMS_UNIT_01.ST0_TRANSFER.IS_ALARMS )
      I_Contact( "DB440_MACHINE_ALARM_DECODING".ALARMS_UNIT_01.ST1_LOAD_UNLOAD.IS_ALARMS )
      I_Contact( "DB440_MACHINE_ALARM_DECODING".ALARMS_UNIT_01.ST2_SPARE.IS_ALARMS )
      I_Contact( "DB440_MACHINE_ALARM_DECODING".ALARMS_UNIT_01.ST3_CLADDING.IS_ALARMS )
      I_Contact( "DB440_MACHINE_ALARM_DECODING".ALARMS_UNIT_01.ST4_CLEANING.IS_ALARMS )
      I_Contact( "DB440_MACHINE_ALARM_DECODING".ALARMS_UNIT_01.GLOBAL.IS_ALARMS )
      I_Contact( "DB440_MACHINE_ALARM_DECODING".ALARMS_UNIT_02.ST0_TRANSFER.IS_ALARMS )
      I_Contact( "DB440_MACHINE_ALARM_DECODING".ALARMS_UNIT_02.ST1_LOAD_UNLOAD.IS_ALARMS )
      I_Contact( "DB440_MACHINE_ALARM_DECODING".ALARMS_UNIT_02.ST2_MEASURING.IS_ALARMS )
      I_Contact( "DB440_MACHINE_ALARM_DECODING".ALARMS_UNIT_02.ST3_CLADDING.IS_ALARMS )
      I_Contact( "DB440_MACHINE_ALARM_DECODING".ALARMS_UNIT_02.ST4_CLEANING.IS_ALARMS )
      I_Contact( "DB440_MACHINE_ALARM_DECODING".ALARMS_UNIT_02.GLOBAL.IS_ALARMS )
      I_Contact( "DB440_MACHINE_ALARM_DECODING".ALARMS_UNIT_03.IS_ALARMS )
      Not()
      Coil( "DB440_MACHINE_ALARM_DECODING".GLOBAL_ALARMS_MACHINE.IS_ALARMS )
   END_RUNG
   // the same network as SCL:
   "DB440_MACHINE_ALARM_DECODING".GLOBAL_ALARMS_MACHINE.IS_ALARMS := NOT (NOT "DB440_MACHINE_ALARM_DECODING".ALARMS_CENTRAL.IS_ALARMS AND NOT "DB440_MACHINE_ALARM_DECODING".ALARMS_UNIT_01.ST0_TRANSFER.IS_ALARMS AND NOT "DB440_MACHINE_ALARM_DECODING".ALARMS_UNIT_01.ST1_LOAD_UNLOAD.IS_ALARMS AND NOT "DB440_MACHINE_ALARM_DECODING".ALARMS_UNIT_01.ST2_SPARE.IS_ALARMS AND NOT "DB440_MACHINE_ALARM_DECODING".ALARMS_UNIT_01.ST3_CLADDING.IS_ALARMS AND NOT "DB440_MACHINE_ALARM_DECODING".ALARMS_UNIT_01.ST4_CLEANING.IS_ALARMS AND NOT "DB440_MACHINE_ALARM_DECODING".ALARMS_UNIT_01.GLOBAL.IS_ALARMS AND NOT "DB440_MACHINE_ALARM_DECODING".ALARMS_UNIT_02.ST0_TRANSFER.IS_ALARMS AND NOT "DB440_MACHINE_ALARM_DECODING".ALARMS_UNIT_02.ST1_LOAD_UNLOAD.IS_ALARMS AND NOT "DB440_MACHINE_ALARM_DECODING".ALARMS_UNIT_02.ST2_MEASURING.IS_ALARMS AND NOT "DB440_MACHINE_ALARM_DECODING".ALARMS_UNIT_02.ST3_CLADDING.IS_ALARMS AND NOT "DB440_MACHINE_ALARM_DECODING".ALARMS_UNIT_02.ST4_CLEANING.IS_ALARMS AND NOT "DB440_MACHINE_ALARM_DECODING".ALARMS_UNIT_02.GLOBAL.IS_ALARMS AND NOT "DB440_MACHINE_ALARM_DECODING".ALARMS_UNIT_03.IS_ALARMS);
END_REGION

REGION Network 13: RETURN HOME POSITION ALARMS
   // Machine Emergency Return Alarm
   RUNG wire#powerrail
      I_Contact( "DB440_MACHINE_ALARM_DECODING".ALARMS_CENTRAL.RHP_ALARMS )
      I_Contact( "DB440_MACHINE_ALARM_DECODING".ALARMS_UNIT_01.ST0_TRANSFER.RHP_ALARMS )
      I_Contact( "DB440_MACHINE_ALARM_DECODING".ALARMS_UNIT_01.ST1_LOAD_UNLOAD.RHP_ALARMS )
      I_Contact( "DB440_MACHINE_ALARM_DECODING".ALARMS_UNIT_01.ST2_SPARE.RHP_ALARMS )
      I_Contact( "DB440_MACHINE_ALARM_DECODING".ALARMS_UNIT_01.ST3_CLADDING.RHP_ALARMS )
      I_Contact( "DB440_MACHINE_ALARM_DECODING".ALARMS_UNIT_01.ST4_CLEANING.RHP_ALARMS )
      I_Contact( "DB440_MACHINE_ALARM_DECODING".ALARMS_UNIT_02.ST0_TRANSFER.RHP_ALARMS )
      I_Contact( "DB440_MACHINE_ALARM_DECODING".ALARMS_UNIT_02.ST1_LOAD_UNLOAD.RHP_ALARMS )
      I_Contact( "DB440_MACHINE_ALARM_DECODING".ALARMS_UNIT_02.ST2_MEASURING.RHP_ALARMS )
      I_Contact( "DB440_MACHINE_ALARM_DECODING".ALARMS_UNIT_02.ST3_CLADDING.RHP_ALARMS )
      I_Contact( "DB440_MACHINE_ALARM_DECODING".ALARMS_UNIT_02.ST4_CLEANING.RHP_ALARMS )
      I_Contact( "DB440_MACHINE_ALARM_DECODING".ALARMS_UNIT_03.RHP_ALARMS )
      Not()
      Coil( "DB440_MACHINE_ALARM_DECODING".GLOBAL_ALARMS_MACHINE.RHP_ALARMS )
   END_RUNG
   // the same network as SCL:
   "DB440_MACHINE_ALARM_DECODING".GLOBAL_ALARMS_MACHINE.RHP_ALARMS := NOT (NOT "DB440_MACHINE_ALARM_DECODING".ALARMS_CENTRAL.RHP_ALARMS AND NOT "DB440_MACHINE_ALARM_DECODING".ALARMS_UNIT_01.ST0_TRANSFER.RHP_ALARMS AND NOT "DB440_MACHINE_ALARM_DECODING".ALARMS_UNIT_01.ST1_LOAD_UNLOAD.RHP_ALARMS AND NOT "DB440_MACHINE_ALARM_DECODING".ALARMS_UNIT_01.ST2_SPARE.RHP_ALARMS AND NOT "DB440_MACHINE_ALARM_DECODING".ALARMS_UNIT_01.ST3_CLADDING.RHP_ALARMS AND NOT "DB440_MACHINE_ALARM_DECODING".ALARMS_UNIT_01.ST4_CLEANING.RHP_ALARMS AND NOT "DB440_MACHINE_ALARM_DECODING".ALARMS_UNIT_02.ST0_TRANSFER.RHP_ALARMS AND NOT "DB440_MACHINE_ALARM_DECODING".ALARMS_UNIT_02.ST1_LOAD_UNLOAD.RHP_ALARMS AND NOT "DB440_MACHINE_ALARM_DECODING".ALARMS_UNIT_02.ST2_MEASURING.RHP_ALARMS AND NOT "DB440_MACHINE_ALARM_DECODING".ALARMS_UNIT_02.ST3_CLADDING.RHP_ALARMS AND NOT "DB440_MACHINE_ALARM_DECODING".ALARMS_UNIT_02.ST4_CLEANING.RHP_ALARMS AND NOT "DB440_MACHINE_ALARM_DECODING".ALARMS_UNIT_03.RHP_ALARMS);
END_REGION

REGION Network 14: STOP END OF CYCLE ALARMS
   // Machine End Of Cycle Alarm
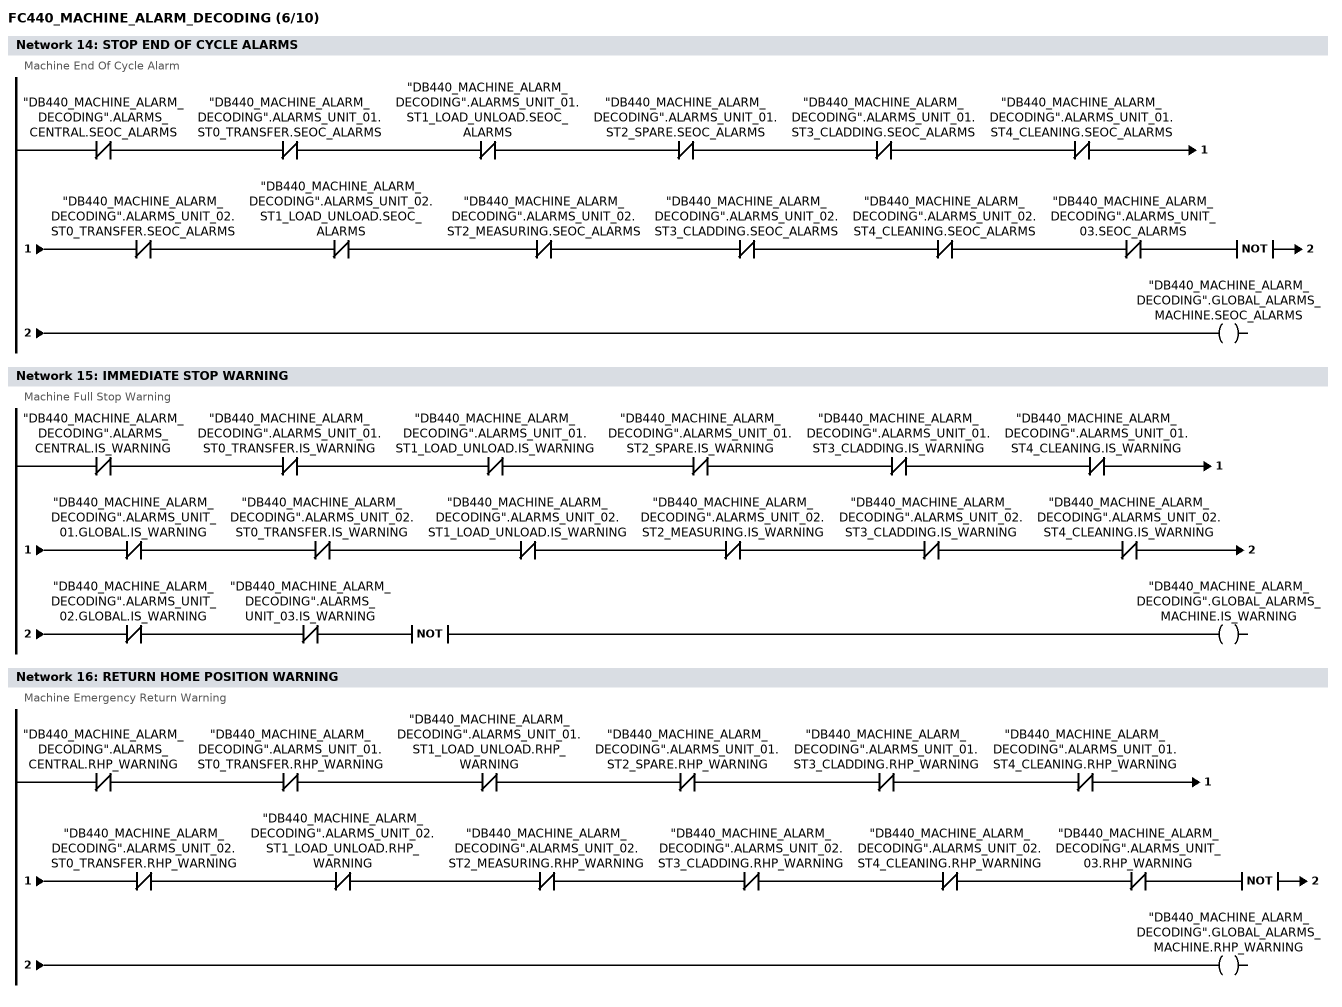
   RUNG wire#powerrail
      I_Contact( "DB440_MACHINE_ALARM_DECODING".ALARMS_CENTRAL.SEOC_ALARMS )
      I_Contact( "DB440_MACHINE_ALARM_DECODING".ALARMS_UNIT_01.ST0_TRANSFER.SEOC_ALARMS )
      I_Contact( "DB440_MACHINE_ALARM_DECODING".ALARMS_UNIT_01.ST1_LOAD_UNLOAD.SEOC_ALARMS )
      I_Contact( "DB440_MACHINE_ALARM_DECODING".ALARMS_UNIT_01.ST2_SPARE.SEOC_ALARMS )
      I_Contact( "DB440_MACHINE_ALARM_DECODING".ALARMS_UNIT_01.ST3_CLADDING.SEOC_ALARMS )
      I_Contact( "DB440_MACHINE_ALARM_DECODING".ALARMS_UNIT_01.ST4_CLEANING.SEOC_ALARMS )
      I_Contact( "DB440_MACHINE_ALARM_DECODING".ALARMS_UNIT_02.ST0_TRANSFER.SEOC_ALARMS )
      I_Contact( "DB440_MACHINE_ALARM_DECODING".ALARMS_UNIT_02.ST1_LOAD_UNLOAD.SEOC_ALARMS )
      I_Contact( "DB440_MACHINE_ALARM_DECODING".ALARMS_UNIT_02.ST2_MEASURING.SEOC_ALARMS )
      I_Contact( "DB440_MACHINE_ALARM_DECODING".ALARMS_UNIT_02.ST3_CLADDING.SEOC_ALARMS )
      I_Contact( "DB440_MACHINE_ALARM_DECODING".ALARMS_UNIT_02.ST4_CLEANING.SEOC_ALARMS )
      I_Contact( "DB440_MACHINE_ALARM_DECODING".ALARMS_UNIT_03.SEOC_ALARMS )
      Not()
      Coil( "DB440_MACHINE_ALARM_DECODING".GLOBAL_ALARMS_MACHINE.SEOC_ALARMS )
   END_RUNG
   // the same network as SCL:
   "DB440_MACHINE_ALARM_DECODING".GLOBAL_ALARMS_MACHINE.SEOC_ALARMS := NOT (NOT "DB440_MACHINE_ALARM_DECODING".ALARMS_CENTRAL.SEOC_ALARMS AND NOT "DB440_MACHINE_ALARM_DECODING".ALARMS_UNIT_01.ST0_TRANSFER.SEOC_ALARMS AND NOT "DB440_MACHINE_ALARM_DECODING".ALARMS_UNIT_01.ST1_LOAD_UNLOAD.SEOC_ALARMS AND NOT "DB440_MACHINE_ALARM_DECODING".ALARMS_UNIT_01.ST2_SPARE.SEOC_ALARMS AND NOT "DB440_MACHINE_ALARM_DECODING".ALARMS_UNIT_01.ST3_CLADDING.SEOC_ALARMS AND NOT "DB440_MACHINE_ALARM_DECODING".ALARMS_UNIT_01.ST4_CLEANING.SEOC_ALARMS AND NOT "DB440_MACHINE_ALARM_DECODING".ALARMS_UNIT_02.ST0_TRANSFER.SEOC_ALARMS AND NOT "DB440_MACHINE_ALARM_DECODING".ALARMS_UNIT_02.ST1_LOAD_UNLOAD.SEOC_ALARMS AND NOT "DB440_MACHINE_ALARM_DECODING".ALARMS_UNIT_02.ST2_MEASURING.SEOC_ALARMS AND NOT "DB440_MACHINE_ALARM_DECODING".ALARMS_UNIT_02.ST3_CLADDING.SEOC_ALARMS AND NOT "DB440_MACHINE_ALARM_DECODING".ALARMS_UNIT_02.ST4_CLEANING.SEOC_ALARMS AND NOT "DB440_MACHINE_ALARM_DECODING".ALARMS_UNIT_03.SEOC_ALARMS);
END_REGION

REGION Network 15: IMMEDIATE STOP WARNING
   // Machine Full Stop Warning
   RUNG wire#powerrail
      I_Contact( "DB440_MACHINE_ALARM_DECODING".ALARMS_CENTRAL.IS_WARNING )
      I_Contact( "DB440_MACHINE_ALARM_DECODING".ALARMS_UNIT_01.ST0_TRANSFER.IS_WARNING )
      I_Contact( "DB440_MACHINE_ALARM_DECODING".ALARMS_UNIT_01.ST1_LOAD_UNLOAD.IS_WARNING )
      I_Contact( "DB440_MACHINE_ALARM_DECODING".ALARMS_UNIT_01.ST2_SPARE.IS_WARNING )
      I_Contact( "DB440_MACHINE_ALARM_DECODING".ALARMS_UNIT_01.ST3_CLADDING.IS_WARNING )
      I_Contact( "DB440_MACHINE_ALARM_DECODING".ALARMS_UNIT_01.ST4_CLEANING.IS_WARNING )
      I_Contact( "DB440_MACHINE_ALARM_DECODING".ALARMS_UNIT_01.GLOBAL.IS_WARNING )
      I_Contact( "DB440_MACHINE_ALARM_DECODING".ALARMS_UNIT_02.ST0_TRANSFER.IS_WARNING )
      I_Contact( "DB440_MACHINE_ALARM_DECODING".ALARMS_UNIT_02.ST1_LOAD_UNLOAD.IS_WARNING )
      I_Contact( "DB440_MACHINE_ALARM_DECODING".ALARMS_UNIT_02.ST2_MEASURING.IS_WARNING )
      I_Contact( "DB440_MACHINE_ALARM_DECODING".ALARMS_UNIT_02.ST3_CLADDING.IS_WARNING )
      I_Contact( "DB440_MACHINE_ALARM_DECODING".ALARMS_UNIT_02.ST4_CLEANING.IS_WARNING )
      I_Contact( "DB440_MACHINE_ALARM_DECODING".ALARMS_UNIT_02.GLOBAL.IS_WARNING )
      I_Contact( "DB440_MACHINE_ALARM_DECODING".ALARMS_UNIT_03.IS_WARNING )
      Not()
      Coil( "DB440_MACHINE_ALARM_DECODING".GLOBAL_ALARMS_MACHINE.IS_WARNING )
   END_RUNG
   // the same network as SCL:
   "DB440_MACHINE_ALARM_DECODING".GLOBAL_ALARMS_MACHINE.IS_WARNING := NOT (NOT "DB440_MACHINE_ALARM_DECODING".ALARMS_CENTRAL.IS_WARNING AND NOT "DB440_MACHINE_ALARM_DECODING".ALARMS_UNIT_01.ST0_TRANSFER.IS_WARNING AND NOT "DB440_MACHINE_ALARM_DECODING".ALARMS_UNIT_01.ST1_LOAD_UNLOAD.IS_WARNING AND NOT "DB440_MACHINE_ALARM_DECODING".ALARMS_UNIT_01.ST2_SPARE.IS_WARNING AND NOT "DB440_MACHINE_ALARM_DECODING".ALARMS_UNIT_01.ST3_CLADDING.IS_WARNING AND NOT "DB440_MACHINE_ALARM_DECODING".ALARMS_UNIT_01.ST4_CLEANING.IS_WARNING AND NOT "DB440_MACHINE_ALARM_DECODING".ALARMS_UNIT_01.GLOBAL.IS_WARNING AND NOT "DB440_MACHINE_ALARM_DECODING".ALARMS_UNIT_02.ST0_TRANSFER.IS_WARNING AND NOT "DB440_MACHINE_ALARM_DECODING".ALARMS_UNIT_02.ST1_LOAD_UNLOAD.IS_WARNING AND NOT "DB440_MACHINE_ALARM_DECODING".ALARMS_UNIT_02.ST2_MEASURING.IS_WARNING AND NOT "DB440_MACHINE_ALARM_DECODING".ALARMS_UNIT_02.ST3_CLADDING.IS_WARNING AND NOT "DB440_MACHINE_ALARM_DECODING".ALARMS_UNIT_02.ST4_CLEANING.IS_WARNING AND NOT "DB440_MACHINE_ALARM_DECODING".ALARMS_UNIT_02.GLOBAL.IS_WARNING AND NOT "DB440_MACHINE_ALARM_DECODING".ALARMS_UNIT_03.IS_WARNING);
END_REGION

REGION Network 16: RETURN HOME POSITION WARNING
   // Machine Emergency Return Warning
   RUNG wire#powerrail
      I_Contact( "DB440_MACHINE_ALARM_DECODING".ALARMS_CENTRAL.RHP_WARNING )
      I_Contact( "DB440_MACHINE_ALARM_DECODING".ALARMS_UNIT_01.ST0_TRANSFER.RHP_WARNING )
      I_Contact( "DB440_MACHINE_ALARM_DECODING".ALARMS_UNIT_01.ST1_LOAD_UNLOAD.RHP_WARNING )
      I_Contact( "DB440_MACHINE_ALARM_DECODING".ALARMS_UNIT_01.ST2_SPARE.RHP_WARNING )
      I_Contact( "DB440_MACHINE_ALARM_DECODING".ALARMS_UNIT_01.ST3_CLADDING.RHP_WARNING )
      I_Contact( "DB440_MACHINE_ALARM_DECODING".ALARMS_UNIT_01.ST4_CLEANING.RHP_WARNING )
      I_Contact( "DB440_MACHINE_ALARM_DECODING".ALARMS_UNIT_02.ST0_TRANSFER.RHP_WARNING )
      I_Contact( "DB440_MACHINE_ALARM_DECODING".ALARMS_UNIT_02.ST1_LOAD_UNLOAD.RHP_WARNING )
      I_Contact( "DB440_MACHINE_ALARM_DECODING".ALARMS_UNIT_02.ST2_MEASURING.RHP_WARNING )
      I_Contact( "DB440_MACHINE_ALARM_DECODING".ALARMS_UNIT_02.ST3_CLADDING.RHP_WARNING )
      I_Contact( "DB440_MACHINE_ALARM_DECODING".ALARMS_UNIT_02.ST4_CLEANING.RHP_WARNING )
      I_Contact( "DB440_MACHINE_ALARM_DECODING".ALARMS_UNIT_03.RHP_WARNING )
      Not()
      Coil( "DB440_MACHINE_ALARM_DECODING".GLOBAL_ALARMS_MACHINE.RHP_WARNING )
   END_RUNG
   // the same network as SCL:
   "DB440_MACHINE_ALARM_DECODING".GLOBAL_ALARMS_MACHINE.RHP_WARNING := NOT (NOT "DB440_MACHINE_ALARM_DECODING".ALARMS_CENTRAL.RHP_WARNING AND NOT "DB440_MACHINE_ALARM_DECODING".ALARMS_UNIT_01.ST0_TRANSFER.RHP_WARNING AND NOT "DB440_MACHINE_ALARM_DECODING".ALARMS_UNIT_01.ST1_LOAD_UNLOAD.RHP_WARNING AND NOT "DB440_MACHINE_ALARM_DECODING".ALARMS_UNIT_01.ST2_SPARE.RHP_WARNING AND NOT "DB440_MACHINE_ALARM_DECODING".ALARMS_UNIT_01.ST3_CLADDING.RHP_WARNING AND NOT "DB440_MACHINE_ALARM_DECODING".ALARMS_UNIT_01.ST4_CLEANING.RHP_WARNING AND NOT "DB440_MACHINE_ALARM_DECODING".ALARMS_UNIT_02.ST0_TRANSFER.RHP_WARNING AND NOT "DB440_MACHINE_ALARM_DECODING".ALARMS_UNIT_02.ST1_LOAD_UNLOAD.RHP_WARNING AND NOT "DB440_MACHINE_ALARM_DECODING".ALARMS_UNIT_02.ST2_MEASURING.RHP_WARNING AND NOT "DB440_MACHINE_ALARM_DECODING".ALARMS_UNIT_02.ST3_CLADDING.RHP_WARNING AND NOT "DB440_MACHINE_ALARM_DECODING".ALARMS_UNIT_02.ST4_CLEANING.RHP_WARNING AND NOT "DB440_MACHINE_ALARM_DECODING".ALARMS_UNIT_03.RHP_WARNING);
END_REGION

REGION Network 17: STOP END OF CYCLE WARNING
   // Machine End of Cycle Warning
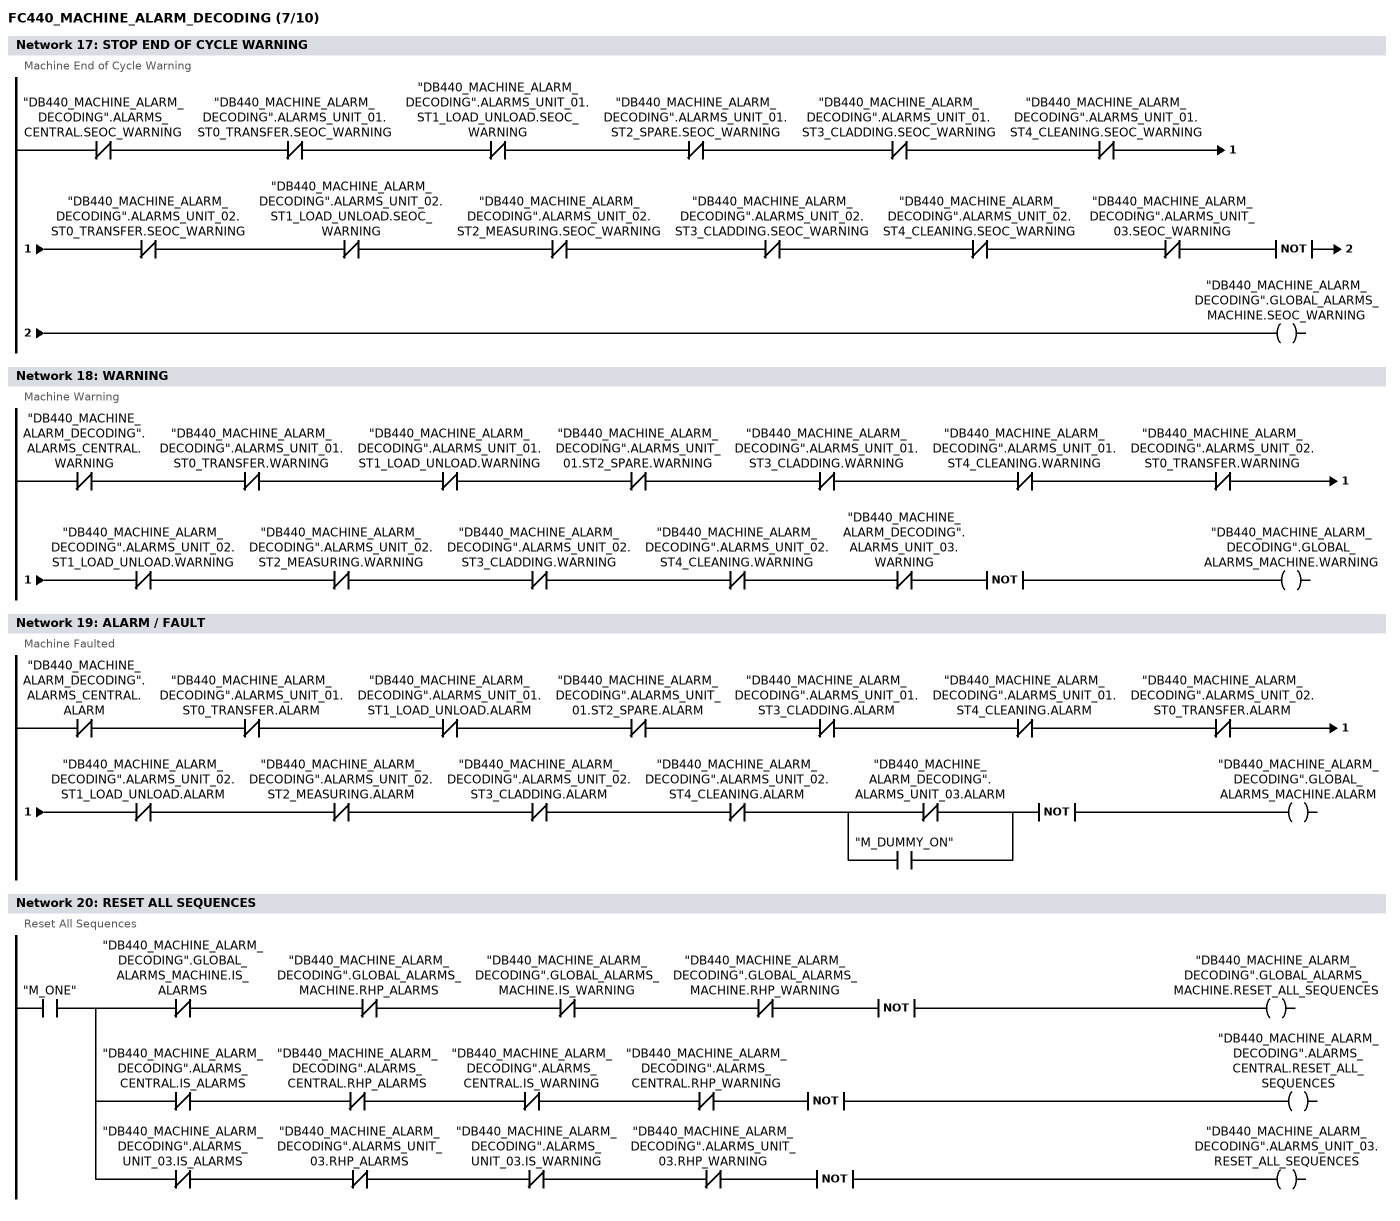
   RUNG wire#powerrail
      I_Contact( "DB440_MACHINE_ALARM_DECODING".ALARMS_CENTRAL.SEOC_WARNING )
      I_Contact( "DB440_MACHINE_ALARM_DECODING".ALARMS_UNIT_01.ST0_TRANSFER.SEOC_WARNING )
      I_Contact( "DB440_MACHINE_ALARM_DECODING".ALARMS_UNIT_01.ST1_LOAD_UNLOAD.SEOC_WARNING )
      I_Contact( "DB440_MACHINE_ALARM_DECODING".ALARMS_UNIT_01.ST2_SPARE.SEOC_WARNING )
      I_Contact( "DB440_MACHINE_ALARM_DECODING".ALARMS_UNIT_01.ST3_CLADDING.SEOC_WARNING )
      I_Contact( "DB440_MACHINE_ALARM_DECODING".ALARMS_UNIT_01.ST4_CLEANING.SEOC_WARNING )
      I_Contact( "DB440_MACHINE_ALARM_DECODING".ALARMS_UNIT_02.ST0_TRANSFER.SEOC_WARNING )
      I_Contact( "DB440_MACHINE_ALARM_DECODING".ALARMS_UNIT_02.ST1_LOAD_UNLOAD.SEOC_WARNING )
      I_Contact( "DB440_MACHINE_ALARM_DECODING".ALARMS_UNIT_02.ST2_MEASURING.SEOC_WARNING )
      I_Contact( "DB440_MACHINE_ALARM_DECODING".ALARMS_UNIT_02.ST3_CLADDING.SEOC_WARNING )
      I_Contact( "DB440_MACHINE_ALARM_DECODING".ALARMS_UNIT_02.ST4_CLEANING.SEOC_WARNING )
      I_Contact( "DB440_MACHINE_ALARM_DECODING".ALARMS_UNIT_03.SEOC_WARNING )
      Not()
      Coil( "DB440_MACHINE_ALARM_DECODING".GLOBAL_ALARMS_MACHINE.SEOC_WARNING )
   END_RUNG
   // the same network as SCL:
   "DB440_MACHINE_ALARM_DECODING".GLOBAL_ALARMS_MACHINE.SEOC_WARNING := NOT (NOT "DB440_MACHINE_ALARM_DECODING".ALARMS_CENTRAL.SEOC_WARNING AND NOT "DB440_MACHINE_ALARM_DECODING".ALARMS_UNIT_01.ST0_TRANSFER.SEOC_WARNING AND NOT "DB440_MACHINE_ALARM_DECODING".ALARMS_UNIT_01.ST1_LOAD_UNLOAD.SEOC_WARNING AND NOT "DB440_MACHINE_ALARM_DECODING".ALARMS_UNIT_01.ST2_SPARE.SEOC_WARNING AND NOT "DB440_MACHINE_ALARM_DECODING".ALARMS_UNIT_01.ST3_CLADDING.SEOC_WARNING AND NOT "DB440_MACHINE_ALARM_DECODING".ALARMS_UNIT_01.ST4_CLEANING.SEOC_WARNING AND NOT "DB440_MACHINE_ALARM_DECODING".ALARMS_UNIT_02.ST0_TRANSFER.SEOC_WARNING AND NOT "DB440_MACHINE_ALARM_DECODING".ALARMS_UNIT_02.ST1_LOAD_UNLOAD.SEOC_WARNING AND NOT "DB440_MACHINE_ALARM_DECODING".ALARMS_UNIT_02.ST2_MEASURING.SEOC_WARNING AND NOT "DB440_MACHINE_ALARM_DECODING".ALARMS_UNIT_02.ST3_CLADDING.SEOC_WARNING AND NOT "DB440_MACHINE_ALARM_DECODING".ALARMS_UNIT_02.ST4_CLEANING.SEOC_WARNING AND NOT "DB440_MACHINE_ALARM_DECODING".ALARMS_UNIT_03.SEOC_WARNING);
END_REGION

REGION Network 18: WARNING
   // Machine Warning
   RUNG wire#powerrail
      I_Contact( "DB440_MACHINE_ALARM_DECODING".ALARMS_CENTRAL.WARNING )
      I_Contact( "DB440_MACHINE_ALARM_DECODING".ALARMS_UNIT_01.ST0_TRANSFER.WARNING )
      I_Contact( "DB440_MACHINE_ALARM_DECODING".ALARMS_UNIT_01.ST1_LOAD_UNLOAD.WARNING )
      I_Contact( "DB440_MACHINE_ALARM_DECODING".ALARMS_UNIT_01.ST2_SPARE.WARNING )
      I_Contact( "DB440_MACHINE_ALARM_DECODING".ALARMS_UNIT_01.ST3_CLADDING.WARNING )
      I_Contact( "DB440_MACHINE_ALARM_DECODING".ALARMS_UNIT_01.ST4_CLEANING.WARNING )
      I_Contact( "DB440_MACHINE_ALARM_DECODING".ALARMS_UNIT_02.ST0_TRANSFER.WARNING )
      I_Contact( "DB440_MACHINE_ALARM_DECODING".ALARMS_UNIT_02.ST1_LOAD_UNLOAD.WARNING )
      I_Contact( "DB440_MACHINE_ALARM_DECODING".ALARMS_UNIT_02.ST2_MEASURING.WARNING )
      I_Contact( "DB440_MACHINE_ALARM_DECODING".ALARMS_UNIT_02.ST3_CLADDING.WARNING )
      I_Contact( "DB440_MACHINE_ALARM_DECODING".ALARMS_UNIT_02.ST4_CLEANING.WARNING )
      I_Contact( "DB440_MACHINE_ALARM_DECODING".ALARMS_UNIT_03.WARNING )
      Not()
      Coil( "DB440_MACHINE_ALARM_DECODING".GLOBAL_ALARMS_MACHINE.WARNING )
   END_RUNG
   // the same network as SCL:
   "DB440_MACHINE_ALARM_DECODING".GLOBAL_ALARMS_MACHINE.WARNING := NOT (NOT "DB440_MACHINE_ALARM_DECODING".ALARMS_CENTRAL.WARNING AND NOT "DB440_MACHINE_ALARM_DECODING".ALARMS_UNIT_01.ST0_TRANSFER.WARNING AND NOT "DB440_MACHINE_ALARM_DECODING".ALARMS_UNIT_01.ST1_LOAD_UNLOAD.WARNING AND NOT "DB440_MACHINE_ALARM_DECODING".ALARMS_UNIT_01.ST2_SPARE.WARNING AND NOT "DB440_MACHINE_ALARM_DECODING".ALARMS_UNIT_01.ST3_CLADDING.WARNING AND NOT "DB440_MACHINE_ALARM_DECODING".ALARMS_UNIT_01.ST4_CLEANING.WARNING AND NOT "DB440_MACHINE_ALARM_DECODING".ALARMS_UNIT_02.ST0_TRANSFER.WARNING AND NOT "DB440_MACHINE_ALARM_DECODING".ALARMS_UNIT_02.ST1_LOAD_UNLOAD.WARNING AND NOT "DB440_MACHINE_ALARM_DECODING".ALARMS_UNIT_02.ST2_MEASURING.WARNING AND NOT "DB440_MACHINE_ALARM_DECODING".ALARMS_UNIT_02.ST3_CLADDING.WARNING AND NOT "DB440_MACHINE_ALARM_DECODING".ALARMS_UNIT_02.ST4_CLEANING.WARNING AND NOT "DB440_MACHINE_ALARM_DECODING".ALARMS_UNIT_03.WARNING);
END_REGION

REGION Network 19: ALARM / FAULT
   // Machine Faulted
   RUNG wire#powerrail
      I_Contact( "DB440_MACHINE_ALARM_DECODING".ALARMS_CENTRAL.ALARM )
      I_Contact( "DB440_MACHINE_ALARM_DECODING".ALARMS_UNIT_01.ST0_TRANSFER.ALARM )
      I_Contact( "DB440_MACHINE_ALARM_DECODING".ALARMS_UNIT_01.ST1_LOAD_UNLOAD.ALARM )
      I_Contact( "DB440_MACHINE_ALARM_DECODING".ALARMS_UNIT_01.ST2_SPARE.ALARM )
      I_Contact( "DB440_MACHINE_ALARM_DECODING".ALARMS_UNIT_01.ST3_CLADDING.ALARM )
      I_Contact( "DB440_MACHINE_ALARM_DECODING".ALARMS_UNIT_01.ST4_CLEANING.ALARM )
      I_Contact( "DB440_MACHINE_ALARM_DECODING".ALARMS_UNIT_02.ST0_TRANSFER.ALARM )
      I_Contact( "DB440_MACHINE_ALARM_DECODING".ALARMS_UNIT_02.ST1_LOAD_UNLOAD.ALARM )
      I_Contact( "DB440_MACHINE_ALARM_DECODING".ALARMS_UNIT_02.ST2_MEASURING.ALARM )
      I_Contact( "DB440_MACHINE_ALARM_DECODING".ALARMS_UNIT_02.ST3_CLADDING.ALARM )
      I_Contact( "DB440_MACHINE_ALARM_DECODING".ALARMS_UNIT_02.ST4_CLEANING.ALARM )
      wire#w1
      I_Contact( "DB440_MACHINE_ALARM_DECODING".ALARMS_UNIT_03.ALARM )
      wire#w2
      Not()
      Coil( "DB440_MACHINE_ALARM_DECODING".GLOBAL_ALARMS_MACHINE.ALARM )
   END_RUNG
   RUNG wire#w1
      Contact( "M_DUMMY_ON" )
   END_RUNG wire#w2
   // the same network as SCL:
   "DB440_MACHINE_ALARM_DECODING".GLOBAL_ALARMS_MACHINE.ALARM := NOT (NOT "DB440_MACHINE_ALARM_DECODING".ALARMS_CENTRAL.ALARM AND NOT "DB440_MACHINE_ALARM_DECODING".ALARMS_UNIT_01.ST0_TRANSFER.ALARM AND NOT "DB440_MACHINE_ALARM_DECODING".ALARMS_UNIT_01.ST1_LOAD_UNLOAD.ALARM AND NOT "DB440_MACHINE_ALARM_DECODING".ALARMS_UNIT_01.ST2_SPARE.ALARM AND NOT "DB440_MACHINE_ALARM_DECODING".ALARMS_UNIT_01.ST3_CLADDING.ALARM AND NOT "DB440_MACHINE_ALARM_DECODING".ALARMS_UNIT_01.ST4_CLEANING.ALARM AND NOT "DB440_MACHINE_ALARM_DECODING".ALARMS_UNIT_02.ST0_TRANSFER.ALARM AND NOT "DB440_MACHINE_ALARM_DECODING".ALARMS_UNIT_02.ST1_LOAD_UNLOAD.ALARM AND NOT "DB440_MACHINE_ALARM_DECODING".ALARMS_UNIT_02.ST2_MEASURING.ALARM AND NOT "DB440_MACHINE_ALARM_DECODING".ALARMS_UNIT_02.ST3_CLADDING.ALARM AND NOT "DB440_MACHINE_ALARM_DECODING".ALARMS_UNIT_02.ST4_CLEANING.ALARM AND (NOT "DB440_MACHINE_ALARM_DECODING".ALARMS_UNIT_03.ALARM OR "M_DUMMY_ON"));
END_REGION

REGION Network 20: RESET ALL SEQUENCES
   // Reset All Sequences
   RUNG wire#powerrail
      Contact( "M_ONE" )
      wire#w1
      I_Contact( "DB440_MACHINE_ALARM_DECODING".GLOBAL_ALARMS_MACHINE.IS_ALARMS )
      I_Contact( "DB440_MACHINE_ALARM_DECODING".GLOBAL_ALARMS_MACHINE.RHP_ALARMS )
      I_Contact( "DB440_MACHINE_ALARM_DECODING".GLOBAL_ALARMS_MACHINE.IS_WARNING )
      I_Contact( "DB440_MACHINE_ALARM_DECODING".GLOBAL_ALARMS_MACHINE.RHP_WARNING )
      Not()
      Coil( "DB440_MACHINE_ALARM_DECODING".GLOBAL_ALARMS_MACHINE.RESET_ALL_SEQUENCES )
   END_RUNG
   RUNG wire#w1
      I_Contact( "DB440_MACHINE_ALARM_DECODING".ALARMS_CENTRAL.IS_ALARMS )
      I_Contact( "DB440_MACHINE_ALARM_DECODING".ALARMS_CENTRAL.RHP_ALARMS )
      I_Contact( "DB440_MACHINE_ALARM_DECODING".ALARMS_CENTRAL.IS_WARNING )
      I_Contact( "DB440_MACHINE_ALARM_DECODING".ALARMS_CENTRAL.RHP_WARNING )
      Not()
      Coil( "DB440_MACHINE_ALARM_DECODING".ALARMS_CENTRAL.RESET_ALL_SEQUENCES )
   END_RUNG
   RUNG wire#w1
      I_Contact( "DB440_MACHINE_ALARM_DECODING".ALARMS_UNIT_03.IS_ALARMS )
      I_Contact( "DB440_MACHINE_ALARM_DECODING".ALARMS_UNIT_03.RHP_ALARMS )
      I_Contact( "DB440_MACHINE_ALARM_DECODING".ALARMS_UNIT_03.IS_WARNING )
      I_Contact( "DB440_MACHINE_ALARM_DECODING".ALARMS_UNIT_03.RHP_WARNING )
      Not()
      Coil( "DB440_MACHINE_ALARM_DECODING".ALARMS_UNIT_03.RESET_ALL_SEQUENCES )
   END_RUNG
   // the same network as SCL:
   "DB440_MACHINE_ALARM_DECODING".GLOBAL_ALARMS_MACHINE.RESET_ALL_SEQUENCES := NOT ("M_ONE" AND NOT "DB440_MACHINE_ALARM_DECODING".GLOBAL_ALARMS_MACHINE.IS_ALARMS AND NOT "DB440_MACHINE_ALARM_DECODING".GLOBAL_ALARMS_MACHINE.RHP_ALARMS AND NOT "DB440_MACHINE_ALARM_DECODING".GLOBAL_ALARMS_MACHINE.IS_WARNING AND NOT "DB440_MACHINE_ALARM_DECODING".GLOBAL_ALARMS_MACHINE.RHP_WARNING);
   "DB440_MACHINE_ALARM_DECODING".ALARMS_CENTRAL.RESET_ALL_SEQUENCES := NOT ("M_ONE" AND NOT "DB440_MACHINE_ALARM_DECODING".ALARMS_CENTRAL.IS_ALARMS AND NOT "DB440_MACHINE_ALARM_DECODING".ALARMS_CENTRAL.RHP_ALARMS AND NOT "DB440_MACHINE_ALARM_DECODING".ALARMS_CENTRAL.IS_WARNING AND NOT "DB440_MACHINE_ALARM_DECODING".ALARMS_CENTRAL.RHP_WARNING);
   "DB440_MACHINE_ALARM_DECODING".ALARMS_UNIT_03.RESET_ALL_SEQUENCES := NOT ("M_ONE" AND NOT "DB440_MACHINE_ALARM_DECODING".ALARMS_UNIT_03.IS_ALARMS AND NOT "DB440_MACHINE_ALARM_DECODING".ALARMS_UNIT_03.RHP_ALARMS AND NOT "DB440_MACHINE_ALARM_DECODING".ALARMS_UNIT_03.IS_WARNING AND NOT "DB440_MACHINE_ALARM_DECODING".ALARMS_UNIT_03.RHP_WARNING);
END_REGION

REGION Network 21: CENTRAL ALARMS RESET LOCAL SEQUENCES AND UNIT 01 STATIONS ALARMS RESET LOCAL SEQUENCES / RESET LOCAL SEQUENCES
   // Central Reset Local Sequences
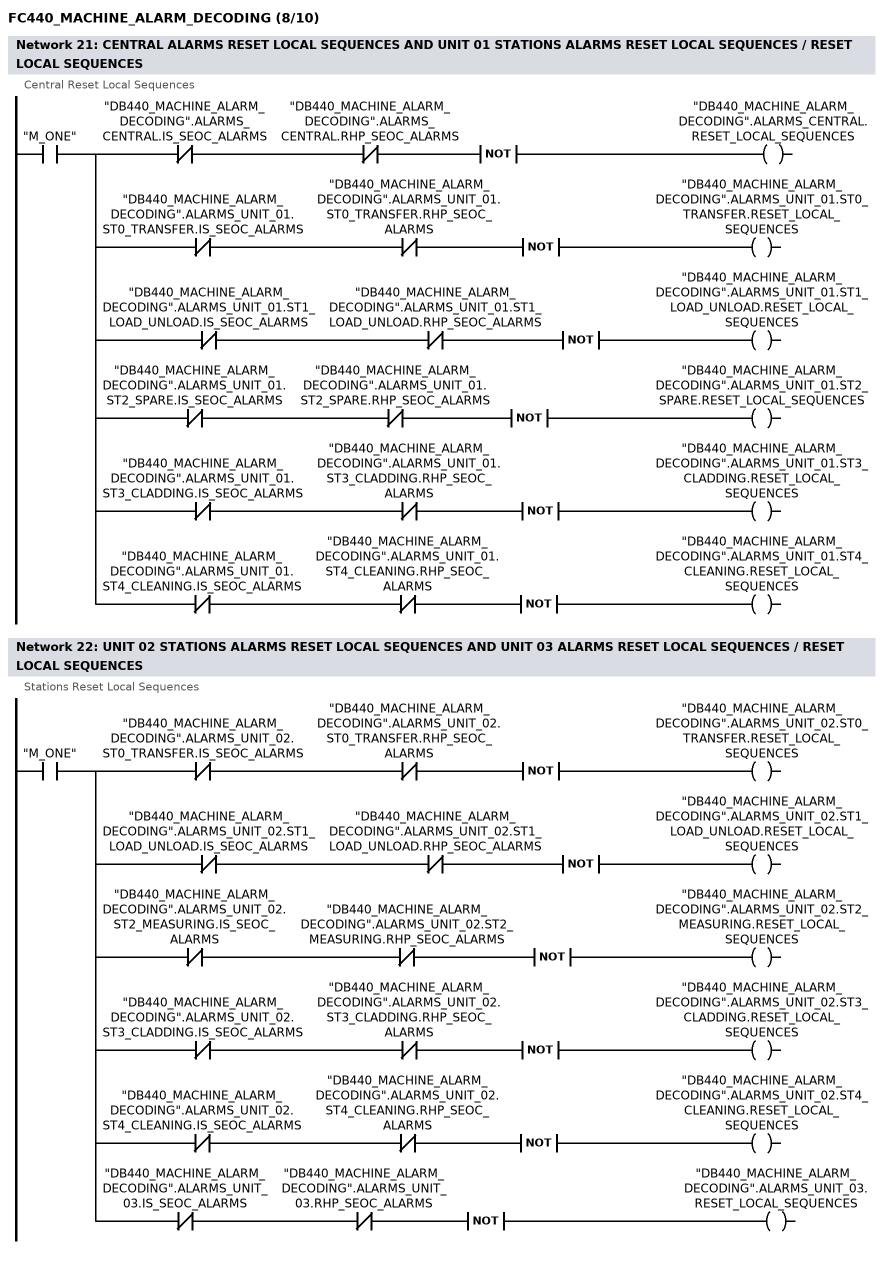
   RUNG wire#powerrail
      Contact( "M_ONE" )
      wire#w1
      I_Contact( "DB440_MACHINE_ALARM_DECODING".ALARMS_CENTRAL.IS_SEOC_ALARMS )
      I_Contact( "DB440_MACHINE_ALARM_DECODING".ALARMS_CENTRAL.RHP_SEOC_ALARMS )
      Not()
      Coil( "DB440_MACHINE_ALARM_DECODING".ALARMS_CENTRAL.RESET_LOCAL_SEQUENCES )
   END_RUNG
   RUNG wire#w1
      I_Contact( "DB440_MACHINE_ALARM_DECODING".ALARMS_UNIT_01.ST0_TRANSFER.IS_SEOC_ALARMS )
      I_Contact( "DB440_MACHINE_ALARM_DECODING".ALARMS_UNIT_01.ST0_TRANSFER.RHP_SEOC_ALARMS )
      Not()
      Coil( "DB440_MACHINE_ALARM_DECODING".ALARMS_UNIT_01.ST0_TRANSFER.RESET_LOCAL_SEQUENCES )
   END_RUNG
   RUNG wire#w1
      I_Contact( "DB440_MACHINE_ALARM_DECODING".ALARMS_UNIT_01.ST1_LOAD_UNLOAD.IS_SEOC_ALARMS )
      I_Contact( "DB440_MACHINE_ALARM_DECODING".ALARMS_UNIT_01.ST1_LOAD_UNLOAD.RHP_SEOC_ALARMS )
      Not()
      Coil( "DB440_MACHINE_ALARM_DECODING".ALARMS_UNIT_01.ST1_LOAD_UNLOAD.RESET_LOCAL_SEQUENCES )
   END_RUNG
   RUNG wire#w1
      I_Contact( "DB440_MACHINE_ALARM_DECODING".ALARMS_UNIT_01.ST2_SPARE.IS_SEOC_ALARMS )
      I_Contact( "DB440_MACHINE_ALARM_DECODING".ALARMS_UNIT_01.ST2_SPARE.RHP_SEOC_ALARMS )
      Not()
      Coil( "DB440_MACHINE_ALARM_DECODING".ALARMS_UNIT_01.ST2_SPARE.RESET_LOCAL_SEQUENCES )
   END_RUNG
   RUNG wire#w1
      I_Contact( "DB440_MACHINE_ALARM_DECODING".ALARMS_UNIT_01.ST3_CLADDING.IS_SEOC_ALARMS )
      I_Contact( "DB440_MACHINE_ALARM_DECODING".ALARMS_UNIT_01.ST3_CLADDING.RHP_SEOC_ALARMS )
      Not()
      Coil( "DB440_MACHINE_ALARM_DECODING".ALARMS_UNIT_01.ST3_CLADDING.RESET_LOCAL_SEQUENCES )
   END_RUNG
   RUNG wire#w1
      I_Contact( "DB440_MACHINE_ALARM_DECODING".ALARMS_UNIT_01.ST4_CLEANING.IS_SEOC_ALARMS )
      I_Contact( "DB440_MACHINE_ALARM_DECODING".ALARMS_UNIT_01.ST4_CLEANING.RHP_SEOC_ALARMS )
      Not()
      Coil( "DB440_MACHINE_ALARM_DECODING".ALARMS_UNIT_01.ST4_CLEANING.RESET_LOCAL_SEQUENCES )
   END_RUNG
   // the same network as SCL:
   "DB440_MACHINE_ALARM_DECODING".ALARMS_CENTRAL.RESET_LOCAL_SEQUENCES := NOT ("M_ONE" AND NOT "DB440_MACHINE_ALARM_DECODING".ALARMS_CENTRAL.IS_SEOC_ALARMS AND NOT "DB440_MACHINE_ALARM_DECODING".ALARMS_CENTRAL.RHP_SEOC_ALARMS);
   "DB440_MACHINE_ALARM_DECODING".ALARMS_UNIT_01.ST0_TRANSFER.RESET_LOCAL_SEQUENCES := NOT ("M_ONE" AND NOT "DB440_MACHINE_ALARM_DECODING".ALARMS_UNIT_01.ST0_TRANSFER.IS_SEOC_ALARMS AND NOT "DB440_MACHINE_ALARM_DECODING".ALARMS_UNIT_01.ST0_TRANSFER.RHP_SEOC_ALARMS);
   "DB440_MACHINE_ALARM_DECODING".ALARMS_UNIT_01.ST1_LOAD_UNLOAD.RESET_LOCAL_SEQUENCES := NOT ("M_ONE" AND NOT "DB440_MACHINE_ALARM_DECODING".ALARMS_UNIT_01.ST1_LOAD_UNLOAD.IS_SEOC_ALARMS AND NOT "DB440_MACHINE_ALARM_DECODING".ALARMS_UNIT_01.ST1_LOAD_UNLOAD.RHP_SEOC_ALARMS);
   "DB440_MACHINE_ALARM_DECODING".ALARMS_UNIT_01.ST2_SPARE.RESET_LOCAL_SEQUENCES := NOT ("M_ONE" AND NOT "DB440_MACHINE_ALARM_DECODING".ALARMS_UNIT_01.ST2_SPARE.IS_SEOC_ALARMS AND NOT "DB440_MACHINE_ALARM_DECODING".ALARMS_UNIT_01.ST2_SPARE.RHP_SEOC_ALARMS);
   "DB440_MACHINE_ALARM_DECODING".ALARMS_UNIT_01.ST3_CLADDING.RESET_LOCAL_SEQUENCES := NOT ("M_ONE" AND NOT "DB440_MACHINE_ALARM_DECODING".ALARMS_UNIT_01.ST3_CLADDING.IS_SEOC_ALARMS AND NOT "DB440_MACHINE_ALARM_DECODING".ALARMS_UNIT_01.ST3_CLADDING.RHP_SEOC_ALARMS);
   "DB440_MACHINE_ALARM_DECODING".ALARMS_UNIT_01.ST4_CLEANING.RESET_LOCAL_SEQUENCES := NOT ("M_ONE" AND NOT "DB440_MACHINE_ALARM_DECODING".ALARMS_UNIT_01.ST4_CLEANING.IS_SEOC_ALARMS AND NOT "DB440_MACHINE_ALARM_DECODING".ALARMS_UNIT_01.ST4_CLEANING.RHP_SEOC_ALARMS);
END_REGION

REGION Network 22: UNIT 02 STATIONS ALARMS RESET LOCAL SEQUENCES AND UNIT 03 ALARMS RESET LOCAL SEQUENCES / RESET LOCAL SEQUENCES
   // Stations Reset Local Sequences
   RUNG wire#powerrail
      Contact( "M_ONE" )
      wire#w1
      I_Contact( "DB440_MACHINE_ALARM_DECODING".ALARMS_UNIT_02.ST0_TRANSFER.IS_SEOC_ALARMS )
      I_Contact( "DB440_MACHINE_ALARM_DECODING".ALARMS_UNIT_02.ST0_TRANSFER.RHP_SEOC_ALARMS )
      Not()
      Coil( "DB440_MACHINE_ALARM_DECODING".ALARMS_UNIT_02.ST0_TRANSFER.RESET_LOCAL_SEQUENCES )
   END_RUNG
   RUNG wire#w1
      I_Contact( "DB440_MACHINE_ALARM_DECODING".ALARMS_UNIT_02.ST1_LOAD_UNLOAD.IS_SEOC_ALARMS )
      I_Contact( "DB440_MACHINE_ALARM_DECODING".ALARMS_UNIT_02.ST1_LOAD_UNLOAD.RHP_SEOC_ALARMS )
      Not()
      Coil( "DB440_MACHINE_ALARM_DECODING".ALARMS_UNIT_02.ST1_LOAD_UNLOAD.RESET_LOCAL_SEQUENCES )
   END_RUNG
   RUNG wire#w1
      I_Contact( "DB440_MACHINE_ALARM_DECODING".ALARMS_UNIT_02.ST2_MEASURING.IS_SEOC_ALARMS )
      I_Contact( "DB440_MACHINE_ALARM_DECODING".ALARMS_UNIT_02.ST2_MEASURING.RHP_SEOC_ALARMS )
      Not()
      Coil( "DB440_MACHINE_ALARM_DECODING".ALARMS_UNIT_02.ST2_MEASURING.RESET_LOCAL_SEQUENCES )
   END_RUNG
   RUNG wire#w1
      I_Contact( "DB440_MACHINE_ALARM_DECODING".ALARMS_UNIT_02.ST3_CLADDING.IS_SEOC_ALARMS )
      I_Contact( "DB440_MACHINE_ALARM_DECODING".ALARMS_UNIT_02.ST3_CLADDING.RHP_SEOC_ALARMS )
      Not()
      Coil( "DB440_MACHINE_ALARM_DECODING".ALARMS_UNIT_02.ST3_CLADDING.RESET_LOCAL_SEQUENCES )
   END_RUNG
   RUNG wire#w1
      I_Contact( "DB440_MACHINE_ALARM_DECODING".ALARMS_UNIT_02.ST4_CLEANING.IS_SEOC_ALARMS )
      I_Contact( "DB440_MACHINE_ALARM_DECODING".ALARMS_UNIT_02.ST4_CLEANING.RHP_SEOC_ALARMS )
      Not()
      Coil( "DB440_MACHINE_ALARM_DECODING".ALARMS_UNIT_02.ST4_CLEANING.RESET_LOCAL_SEQUENCES )
   END_RUNG
   RUNG wire#w1
      I_Contact( "DB440_MACHINE_ALARM_DECODING".ALARMS_UNIT_03.IS_SEOC_ALARMS )
      I_Contact( "DB440_MACHINE_ALARM_DECODING".ALARMS_UNIT_03.RHP_SEOC_ALARMS )
      Not()
      Coil( "DB440_MACHINE_ALARM_DECODING".ALARMS_UNIT_03.RESET_LOCAL_SEQUENCES )
   END_RUNG
   // the same network as SCL:
   "DB440_MACHINE_ALARM_DECODING".ALARMS_UNIT_02.ST0_TRANSFER.RESET_LOCAL_SEQUENCES := NOT ("M_ONE" AND NOT "DB440_MACHINE_ALARM_DECODING".ALARMS_UNIT_02.ST0_TRANSFER.IS_SEOC_ALARMS AND NOT "DB440_MACHINE_ALARM_DECODING".ALARMS_UNIT_02.ST0_TRANSFER.RHP_SEOC_ALARMS);
   "DB440_MACHINE_ALARM_DECODING".ALARMS_UNIT_02.ST1_LOAD_UNLOAD.RESET_LOCAL_SEQUENCES := NOT ("M_ONE" AND NOT "DB440_MACHINE_ALARM_DECODING".ALARMS_UNIT_02.ST1_LOAD_UNLOAD.IS_SEOC_ALARMS AND NOT "DB440_MACHINE_ALARM_DECODING".ALARMS_UNIT_02.ST1_LOAD_UNLOAD.RHP_SEOC_ALARMS);
   "DB440_MACHINE_ALARM_DECODING".ALARMS_UNIT_02.ST2_MEASURING.RESET_LOCAL_SEQUENCES := NOT ("M_ONE" AND NOT "DB440_MACHINE_ALARM_DECODING".ALARMS_UNIT_02.ST2_MEASURING.IS_SEOC_ALARMS AND NOT "DB440_MACHINE_ALARM_DECODING".ALARMS_UNIT_02.ST2_MEASURING.RHP_SEOC_ALARMS);
   "DB440_MACHINE_ALARM_DECODING".ALARMS_UNIT_02.ST3_CLADDING.RESET_LOCAL_SEQUENCES := NOT ("M_ONE" AND NOT "DB440_MACHINE_ALARM_DECODING".ALARMS_UNIT_02.ST3_CLADDING.IS_SEOC_ALARMS AND NOT "DB440_MACHINE_ALARM_DECODING".ALARMS_UNIT_02.ST3_CLADDING.RHP_SEOC_ALARMS);
   "DB440_MACHINE_ALARM_DECODING".ALARMS_UNIT_02.ST4_CLEANING.RESET_LOCAL_SEQUENCES := NOT ("M_ONE" AND NOT "DB440_MACHINE_ALARM_DECODING".ALARMS_UNIT_02.ST4_CLEANING.IS_SEOC_ALARMS AND NOT "DB440_MACHINE_ALARM_DECODING".ALARMS_UNIT_02.ST4_CLEANING.RHP_SEOC_ALARMS);
   "DB440_MACHINE_ALARM_DECODING".ALARMS_UNIT_03.RESET_LOCAL_SEQUENCES := NOT ("M_ONE" AND NOT "DB440_MACHINE_ALARM_DECODING".ALARMS_UNIT_03.IS_SEOC_ALARMS AND NOT "DB440_MACHINE_ALARM_DECODING".ALARMS_UNIT_03.RHP_SEOC_ALARMS);
END_REGION

REGION Network 23: <<<<<<<<<<<<<<<<<<<< ALARMS BY UNIT >>>>>>>>>>>>>>>>>>>>
END_REGION

REGION Network 24: <<<<<<<<<<<<<<<<<<<<<<<< UNIT 01 >>>>>>>>>>>>>>>>>>>>>>>>
END_REGION

REGION Network 25: UNIT 01 GLOBAL ALARMS AND WARNINGS
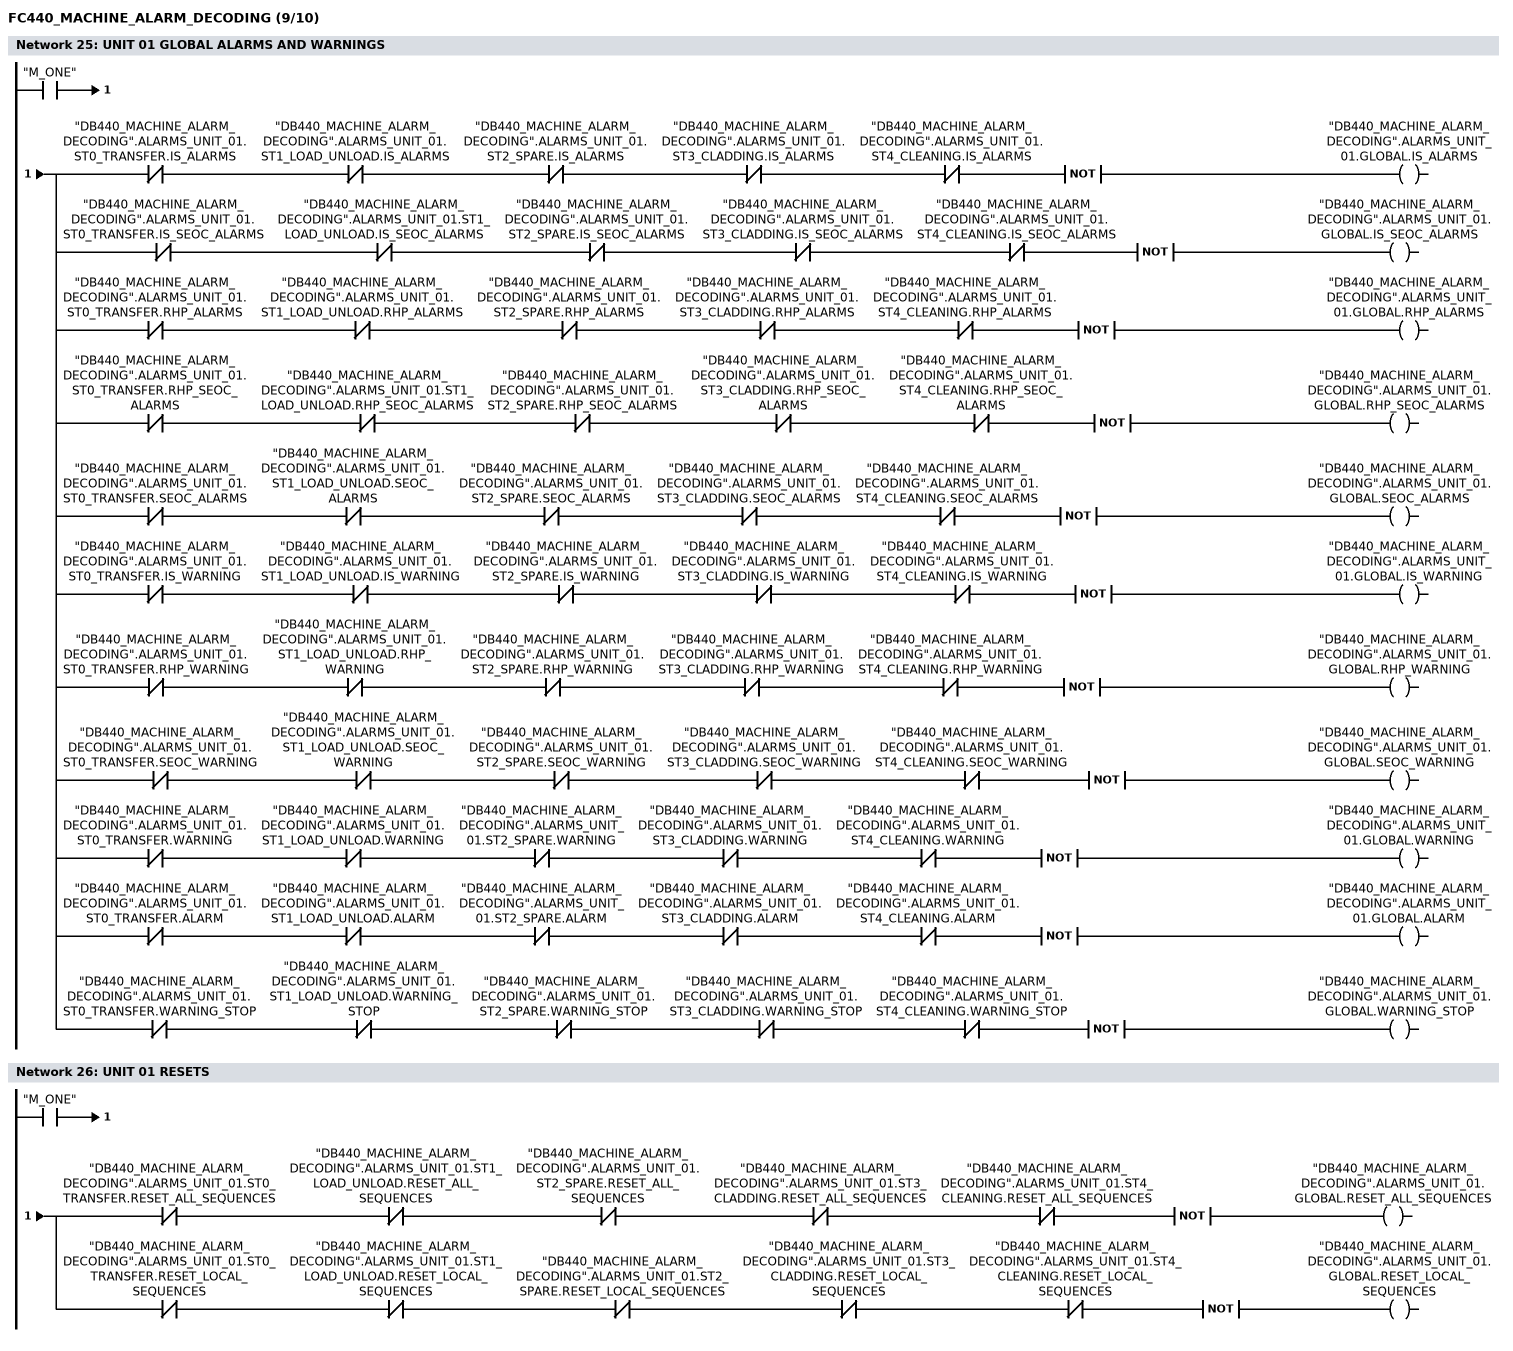
   RUNG wire#powerrail
      Contact( "M_ONE" )
      wire#w1
      I_Contact( "DB440_MACHINE_ALARM_DECODING".ALARMS_UNIT_01.ST0_TRANSFER.IS_ALARMS )
      I_Contact( "DB440_MACHINE_ALARM_DECODING".ALARMS_UNIT_01.ST1_LOAD_UNLOAD.IS_ALARMS )
      I_Contact( "DB440_MACHINE_ALARM_DECODING".ALARMS_UNIT_01.ST2_SPARE.IS_ALARMS )
      I_Contact( "DB440_MACHINE_ALARM_DECODING".ALARMS_UNIT_01.ST3_CLADDING.IS_ALARMS )
      I_Contact( "DB440_MACHINE_ALARM_DECODING".ALARMS_UNIT_01.ST4_CLEANING.IS_ALARMS )
      Not()
      Coil( "DB440_MACHINE_ALARM_DECODING".ALARMS_UNIT_01.GLOBAL.IS_ALARMS )
   END_RUNG
   RUNG wire#w1
      I_Contact( "DB440_MACHINE_ALARM_DECODING".ALARMS_UNIT_01.ST0_TRANSFER.IS_SEOC_ALARMS )
      I_Contact( "DB440_MACHINE_ALARM_DECODING".ALARMS_UNIT_01.ST1_LOAD_UNLOAD.IS_SEOC_ALARMS )
      I_Contact( "DB440_MACHINE_ALARM_DECODING".ALARMS_UNIT_01.ST2_SPARE.IS_SEOC_ALARMS )
      I_Contact( "DB440_MACHINE_ALARM_DECODING".ALARMS_UNIT_01.ST3_CLADDING.IS_SEOC_ALARMS )
      I_Contact( "DB440_MACHINE_ALARM_DECODING".ALARMS_UNIT_01.ST4_CLEANING.IS_SEOC_ALARMS )
      Not()
      Coil( "DB440_MACHINE_ALARM_DECODING".ALARMS_UNIT_01.GLOBAL.IS_SEOC_ALARMS )
   END_RUNG
   RUNG wire#w1
      I_Contact( "DB440_MACHINE_ALARM_DECODING".ALARMS_UNIT_01.ST0_TRANSFER.RHP_ALARMS )
      I_Contact( "DB440_MACHINE_ALARM_DECODING".ALARMS_UNIT_01.ST1_LOAD_UNLOAD.RHP_ALARMS )
      I_Contact( "DB440_MACHINE_ALARM_DECODING".ALARMS_UNIT_01.ST2_SPARE.RHP_ALARMS )
      I_Contact( "DB440_MACHINE_ALARM_DECODING".ALARMS_UNIT_01.ST3_CLADDING.RHP_ALARMS )
      I_Contact( "DB440_MACHINE_ALARM_DECODING".ALARMS_UNIT_01.ST4_CLEANING.RHP_ALARMS )
      Not()
      Coil( "DB440_MACHINE_ALARM_DECODING".ALARMS_UNIT_01.GLOBAL.RHP_ALARMS )
   END_RUNG
   RUNG wire#w1
      I_Contact( "DB440_MACHINE_ALARM_DECODING".ALARMS_UNIT_01.ST0_TRANSFER.RHP_SEOC_ALARMS )
      I_Contact( "DB440_MACHINE_ALARM_DECODING".ALARMS_UNIT_01.ST1_LOAD_UNLOAD.RHP_SEOC_ALARMS )
      I_Contact( "DB440_MACHINE_ALARM_DECODING".ALARMS_UNIT_01.ST2_SPARE.RHP_SEOC_ALARMS )
      I_Contact( "DB440_MACHINE_ALARM_DECODING".ALARMS_UNIT_01.ST3_CLADDING.RHP_SEOC_ALARMS )
      I_Contact( "DB440_MACHINE_ALARM_DECODING".ALARMS_UNIT_01.ST4_CLEANING.RHP_SEOC_ALARMS )
      Not()
      Coil( "DB440_MACHINE_ALARM_DECODING".ALARMS_UNIT_01.GLOBAL.RHP_SEOC_ALARMS )
   END_RUNG
   RUNG wire#w1
      I_Contact( "DB440_MACHINE_ALARM_DECODING".ALARMS_UNIT_01.ST0_TRANSFER.SEOC_ALARMS )
      I_Contact( "DB440_MACHINE_ALARM_DECODING".ALARMS_UNIT_01.ST1_LOAD_UNLOAD.SEOC_ALARMS )
      I_Contact( "DB440_MACHINE_ALARM_DECODING".ALARMS_UNIT_01.ST2_SPARE.SEOC_ALARMS )
      I_Contact( "DB440_MACHINE_ALARM_DECODING".ALARMS_UNIT_01.ST3_CLADDING.SEOC_ALARMS )
      I_Contact( "DB440_MACHINE_ALARM_DECODING".ALARMS_UNIT_01.ST4_CLEANING.SEOC_ALARMS )
      Not()
      Coil( "DB440_MACHINE_ALARM_DECODING".ALARMS_UNIT_01.GLOBAL.SEOC_ALARMS )
   END_RUNG
   RUNG wire#w1
      I_Contact( "DB440_MACHINE_ALARM_DECODING".ALARMS_UNIT_01.ST0_TRANSFER.IS_WARNING )
      I_Contact( "DB440_MACHINE_ALARM_DECODING".ALARMS_UNIT_01.ST1_LOAD_UNLOAD.IS_WARNING )
      I_Contact( "DB440_MACHINE_ALARM_DECODING".ALARMS_UNIT_01.ST2_SPARE.IS_WARNING )
      I_Contact( "DB440_MACHINE_ALARM_DECODING".ALARMS_UNIT_01.ST3_CLADDING.IS_WARNING )
      I_Contact( "DB440_MACHINE_ALARM_DECODING".ALARMS_UNIT_01.ST4_CLEANING.IS_WARNING )
      Not()
      Coil( "DB440_MACHINE_ALARM_DECODING".ALARMS_UNIT_01.GLOBAL.IS_WARNING )
   END_RUNG
   RUNG wire#w1
      I_Contact( "DB440_MACHINE_ALARM_DECODING".ALARMS_UNIT_01.ST0_TRANSFER.RHP_WARNING )
      I_Contact( "DB440_MACHINE_ALARM_DECODING".ALARMS_UNIT_01.ST1_LOAD_UNLOAD.RHP_WARNING )
      I_Contact( "DB440_MACHINE_ALARM_DECODING".ALARMS_UNIT_01.ST2_SPARE.RHP_WARNING )
      I_Contact( "DB440_MACHINE_ALARM_DECODING".ALARMS_UNIT_01.ST3_CLADDING.RHP_WARNING )
      I_Contact( "DB440_MACHINE_ALARM_DECODING".ALARMS_UNIT_01.ST4_CLEANING.RHP_WARNING )
      Not()
      Coil( "DB440_MACHINE_ALARM_DECODING".ALARMS_UNIT_01.GLOBAL.RHP_WARNING )
   END_RUNG
   RUNG wire#w1
      I_Contact( "DB440_MACHINE_ALARM_DECODING".ALARMS_UNIT_01.ST0_TRANSFER.SEOC_WARNING )
      I_Contact( "DB440_MACHINE_ALARM_DECODING".ALARMS_UNIT_01.ST1_LOAD_UNLOAD.SEOC_WARNING )
      I_Contact( "DB440_MACHINE_ALARM_DECODING".ALARMS_UNIT_01.ST2_SPARE.SEOC_WARNING )
      I_Contact( "DB440_MACHINE_ALARM_DECODING".ALARMS_UNIT_01.ST3_CLADDING.SEOC_WARNING )
      I_Contact( "DB440_MACHINE_ALARM_DECODING".ALARMS_UNIT_01.ST4_CLEANING.SEOC_WARNING )
      Not()
      Coil( "DB440_MACHINE_ALARM_DECODING".ALARMS_UNIT_01.GLOBAL.SEOC_WARNING )
   END_RUNG
   RUNG wire#w1
      I_Contact( "DB440_MACHINE_ALARM_DECODING".ALARMS_UNIT_01.ST0_TRANSFER.WARNING )
      I_Contact( "DB440_MACHINE_ALARM_DECODING".ALARMS_UNIT_01.ST1_LOAD_UNLOAD.WARNING )
      I_Contact( "DB440_MACHINE_ALARM_DECODING".ALARMS_UNIT_01.ST2_SPARE.WARNING )
      I_Contact( "DB440_MACHINE_ALARM_DECODING".ALARMS_UNIT_01.ST3_CLADDING.WARNING )
      I_Contact( "DB440_MACHINE_ALARM_DECODING".ALARMS_UNIT_01.ST4_CLEANING.WARNING )
      Not()
      Coil( "DB440_MACHINE_ALARM_DECODING".ALARMS_UNIT_01.GLOBAL.WARNING )
   END_RUNG
   RUNG wire#w1
      I_Contact( "DB440_MACHINE_ALARM_DECODING".ALARMS_UNIT_01.ST0_TRANSFER.ALARM )
      I_Contact( "DB440_MACHINE_ALARM_DECODING".ALARMS_UNIT_01.ST1_LOAD_UNLOAD.ALARM )
      I_Contact( "DB440_MACHINE_ALARM_DECODING".ALARMS_UNIT_01.ST2_SPARE.ALARM )
      I_Contact( "DB440_MACHINE_ALARM_DECODING".ALARMS_UNIT_01.ST3_CLADDING.ALARM )
      I_Contact( "DB440_MACHINE_ALARM_DECODING".ALARMS_UNIT_01.ST4_CLEANING.ALARM )
      Not()
      Coil( "DB440_MACHINE_ALARM_DECODING".ALARMS_UNIT_01.GLOBAL.ALARM )
   END_RUNG
   RUNG wire#w1
      I_Contact( "DB440_MACHINE_ALARM_DECODING".ALARMS_UNIT_01.ST0_TRANSFER.WARNING_STOP )
      I_Contact( "DB440_MACHINE_ALARM_DECODING".ALARMS_UNIT_01.ST1_LOAD_UNLOAD.WARNING_STOP )
      I_Contact( "DB440_MACHINE_ALARM_DECODING".ALARMS_UNIT_01.ST2_SPARE.WARNING_STOP )
      I_Contact( "DB440_MACHINE_ALARM_DECODING".ALARMS_UNIT_01.ST3_CLADDING.WARNING_STOP )
      I_Contact( "DB440_MACHINE_ALARM_DECODING".ALARMS_UNIT_01.ST4_CLEANING.WARNING_STOP )
      Not()
      Coil( "DB440_MACHINE_ALARM_DECODING".ALARMS_UNIT_01.GLOBAL.WARNING_STOP )
   END_RUNG
   // the same network as SCL:
   "DB440_MACHINE_ALARM_DECODING".ALARMS_UNIT_01.GLOBAL.IS_ALARMS := NOT ("M_ONE" AND NOT "DB440_MACHINE_ALARM_DECODING".ALARMS_UNIT_01.ST0_TRANSFER.IS_ALARMS AND NOT "DB440_MACHINE_ALARM_DECODING".ALARMS_UNIT_01.ST1_LOAD_UNLOAD.IS_ALARMS AND NOT "DB440_MACHINE_ALARM_DECODING".ALARMS_UNIT_01.ST2_SPARE.IS_ALARMS AND NOT "DB440_MACHINE_ALARM_DECODING".ALARMS_UNIT_01.ST3_CLADDING.IS_ALARMS AND NOT "DB440_MACHINE_ALARM_DECODING".ALARMS_UNIT_01.ST4_CLEANING.IS_ALARMS);
   "DB440_MACHINE_ALARM_DECODING".ALARMS_UNIT_01.GLOBAL.IS_SEOC_ALARMS := NOT ("M_ONE" AND NOT "DB440_MACHINE_ALARM_DECODING".ALARMS_UNIT_01.ST0_TRANSFER.IS_SEOC_ALARMS AND NOT "DB440_MACHINE_ALARM_DECODING".ALARMS_UNIT_01.ST1_LOAD_UNLOAD.IS_SEOC_ALARMS AND NOT "DB440_MACHINE_ALARM_DECODING".ALARMS_UNIT_01.ST2_SPARE.IS_SEOC_ALARMS AND NOT "DB440_MACHINE_ALARM_DECODING".ALARMS_UNIT_01.ST3_CLADDING.IS_SEOC_ALARMS AND NOT "DB440_MACHINE_ALARM_DECODING".ALARMS_UNIT_01.ST4_CLEANING.IS_SEOC_ALARMS);
   "DB440_MACHINE_ALARM_DECODING".ALARMS_UNIT_01.GLOBAL.RHP_ALARMS := NOT ("M_ONE" AND NOT "DB440_MACHINE_ALARM_DECODING".ALARMS_UNIT_01.ST0_TRANSFER.RHP_ALARMS AND NOT "DB440_MACHINE_ALARM_DECODING".ALARMS_UNIT_01.ST1_LOAD_UNLOAD.RHP_ALARMS AND NOT "DB440_MACHINE_ALARM_DECODING".ALARMS_UNIT_01.ST2_SPARE.RHP_ALARMS AND NOT "DB440_MACHINE_ALARM_DECODING".ALARMS_UNIT_01.ST3_CLADDING.RHP_ALARMS AND NOT "DB440_MACHINE_ALARM_DECODING".ALARMS_UNIT_01.ST4_CLEANING.RHP_ALARMS);
   "DB440_MACHINE_ALARM_DECODING".ALARMS_UNIT_01.GLOBAL.RHP_SEOC_ALARMS := NOT ("M_ONE" AND NOT "DB440_MACHINE_ALARM_DECODING".ALARMS_UNIT_01.ST0_TRANSFER.RHP_SEOC_ALARMS AND NOT "DB440_MACHINE_ALARM_DECODING".ALARMS_UNIT_01.ST1_LOAD_UNLOAD.RHP_SEOC_ALARMS AND NOT "DB440_MACHINE_ALARM_DECODING".ALARMS_UNIT_01.ST2_SPARE.RHP_SEOC_ALARMS AND NOT "DB440_MACHINE_ALARM_DECODING".ALARMS_UNIT_01.ST3_CLADDING.RHP_SEOC_ALARMS AND NOT "DB440_MACHINE_ALARM_DECODING".ALARMS_UNIT_01.ST4_CLEANING.RHP_SEOC_ALARMS);
   "DB440_MACHINE_ALARM_DECODING".ALARMS_UNIT_01.GLOBAL.SEOC_ALARMS := NOT ("M_ONE" AND NOT "DB440_MACHINE_ALARM_DECODING".ALARMS_UNIT_01.ST0_TRANSFER.SEOC_ALARMS AND NOT "DB440_MACHINE_ALARM_DECODING".ALARMS_UNIT_01.ST1_LOAD_UNLOAD.SEOC_ALARMS AND NOT "DB440_MACHINE_ALARM_DECODING".ALARMS_UNIT_01.ST2_SPARE.SEOC_ALARMS AND NOT "DB440_MACHINE_ALARM_DECODING".ALARMS_UNIT_01.ST3_CLADDING.SEOC_ALARMS AND NOT "DB440_MACHINE_ALARM_DECODING".ALARMS_UNIT_01.ST4_CLEANING.SEOC_ALARMS);
   "DB440_MACHINE_ALARM_DECODING".ALARMS_UNIT_01.GLOBAL.IS_WARNING := NOT ("M_ONE" AND NOT "DB440_MACHINE_ALARM_DECODING".ALARMS_UNIT_01.ST0_TRANSFER.IS_WARNING AND NOT "DB440_MACHINE_ALARM_DECODING".ALARMS_UNIT_01.ST1_LOAD_UNLOAD.IS_WARNING AND NOT "DB440_MACHINE_ALARM_DECODING".ALARMS_UNIT_01.ST2_SPARE.IS_WARNING AND NOT "DB440_MACHINE_ALARM_DECODING".ALARMS_UNIT_01.ST3_CLADDING.IS_WARNING AND NOT "DB440_MACHINE_ALARM_DECODING".ALARMS_UNIT_01.ST4_CLEANING.IS_WARNING);
   "DB440_MACHINE_ALARM_DECODING".ALARMS_UNIT_01.GLOBAL.RHP_WARNING := NOT ("M_ONE" AND NOT "DB440_MACHINE_ALARM_DECODING".ALARMS_UNIT_01.ST0_TRANSFER.RHP_WARNING AND NOT "DB440_MACHINE_ALARM_DECODING".ALARMS_UNIT_01.ST1_LOAD_UNLOAD.RHP_WARNING AND NOT "DB440_MACHINE_ALARM_DECODING".ALARMS_UNIT_01.ST2_SPARE.RHP_WARNING AND NOT "DB440_MACHINE_ALARM_DECODING".ALARMS_UNIT_01.ST3_CLADDING.RHP_WARNING AND NOT "DB440_MACHINE_ALARM_DECODING".ALARMS_UNIT_01.ST4_CLEANING.RHP_WARNING);
   "DB440_MACHINE_ALARM_DECODING".ALARMS_UNIT_01.GLOBAL.SEOC_WARNING := NOT ("M_ONE" AND NOT "DB440_MACHINE_ALARM_DECODING".ALARMS_UNIT_01.ST0_TRANSFER.SEOC_WARNING AND NOT "DB440_MACHINE_ALARM_DECODING".ALARMS_UNIT_01.ST1_LOAD_UNLOAD.SEOC_WARNING AND NOT "DB440_MACHINE_ALARM_DECODING".ALARMS_UNIT_01.ST2_SPARE.SEOC_WARNING AND NOT "DB440_MACHINE_ALARM_DECODING".ALARMS_UNIT_01.ST3_CLADDING.SEOC_WARNING AND NOT "DB440_MACHINE_ALARM_DECODING".ALARMS_UNIT_01.ST4_CLEANING.SEOC_WARNING);
   "DB440_MACHINE_ALARM_DECODING".ALARMS_UNIT_01.GLOBAL.WARNING := NOT ("M_ONE" AND NOT "DB440_MACHINE_ALARM_DECODING".ALARMS_UNIT_01.ST0_TRANSFER.WARNING AND NOT "DB440_MACHINE_ALARM_DECODING".ALARMS_UNIT_01.ST1_LOAD_UNLOAD.WARNING AND NOT "DB440_MACHINE_ALARM_DECODING".ALARMS_UNIT_01.ST2_SPARE.WARNING AND NOT "DB440_MACHINE_ALARM_DECODING".ALARMS_UNIT_01.ST3_CLADDING.WARNING AND NOT "DB440_MACHINE_ALARM_DECODING".ALARMS_UNIT_01.ST4_CLEANING.WARNING);
   "DB440_MACHINE_ALARM_DECODING".ALARMS_UNIT_01.GLOBAL.ALARM := NOT ("M_ONE" AND NOT "DB440_MACHINE_ALARM_DECODING".ALARMS_UNIT_01.ST0_TRANSFER.ALARM AND NOT "DB440_MACHINE_ALARM_DECODING".ALARMS_UNIT_01.ST1_LOAD_UNLOAD.ALARM AND NOT "DB440_MACHINE_ALARM_DECODING".ALARMS_UNIT_01.ST2_SPARE.ALARM AND NOT "DB440_MACHINE_ALARM_DECODING".ALARMS_UNIT_01.ST3_CLADDING.ALARM AND NOT "DB440_MACHINE_ALARM_DECODING".ALARMS_UNIT_01.ST4_CLEANING.ALARM);
   "DB440_MACHINE_ALARM_DECODING".ALARMS_UNIT_01.GLOBAL.WARNING_STOP := NOT ("M_ONE" AND NOT "DB440_MACHINE_ALARM_DECODING".ALARMS_UNIT_01.ST0_TRANSFER.WARNING_STOP AND NOT "DB440_MACHINE_ALARM_DECODING".ALARMS_UNIT_01.ST1_LOAD_UNLOAD.WARNING_STOP AND NOT "DB440_MACHINE_ALARM_DECODING".ALARMS_UNIT_01.ST2_SPARE.WARNING_STOP AND NOT "DB440_MACHINE_ALARM_DECODING".ALARMS_UNIT_01.ST3_CLADDING.WARNING_STOP AND NOT "DB440_MACHINE_ALARM_DECODING".ALARMS_UNIT_01.ST4_CLEANING.WARNING_STOP);
END_REGION

REGION Network 26: UNIT 01 RESETS
   RUNG wire#powerrail
      Contact( "M_ONE" )
      wire#w1
      I_Contact( "DB440_MACHINE_ALARM_DECODING".ALARMS_UNIT_01.ST0_TRANSFER.RESET_ALL_SEQUENCES )
      I_Contact( "DB440_MACHINE_ALARM_DECODING".ALARMS_UNIT_01.ST1_LOAD_UNLOAD.RESET_ALL_SEQUENCES )
      I_Contact( "DB440_MACHINE_ALARM_DECODING".ALARMS_UNIT_01.ST2_SPARE.RESET_ALL_SEQUENCES )
      I_Contact( "DB440_MACHINE_ALARM_DECODING".ALARMS_UNIT_01.ST3_CLADDING.RESET_ALL_SEQUENCES )
      I_Contact( "DB440_MACHINE_ALARM_DECODING".ALARMS_UNIT_01.ST4_CLEANING.RESET_ALL_SEQUENCES )
      Not()
      Coil( "DB440_MACHINE_ALARM_DECODING".ALARMS_UNIT_01.GLOBAL.RESET_ALL_SEQUENCES )
   END_RUNG
   RUNG wire#w1
      I_Contact( "DB440_MACHINE_ALARM_DECODING".ALARMS_UNIT_01.ST0_TRANSFER.RESET_LOCAL_SEQUENCES )
      I_Contact( "DB440_MACHINE_ALARM_DECODING".ALARMS_UNIT_01.ST1_LOAD_UNLOAD.RESET_LOCAL_SEQUENCES )
      I_Contact( "DB440_MACHINE_ALARM_DECODING".ALARMS_UNIT_01.ST2_SPARE.RESET_LOCAL_SEQUENCES )
      I_Contact( "DB440_MACHINE_ALARM_DECODING".ALARMS_UNIT_01.ST3_CLADDING.RESET_LOCAL_SEQUENCES )
      I_Contact( "DB440_MACHINE_ALARM_DECODING".ALARMS_UNIT_01.ST4_CLEANING.RESET_LOCAL_SEQUENCES )
      Not()
      Coil( "DB440_MACHINE_ALARM_DECODING".ALARMS_UNIT_01.GLOBAL.RESET_LOCAL_SEQUENCES )
   END_RUNG
   // the same network as SCL:
   "DB440_MACHINE_ALARM_DECODING".ALARMS_UNIT_01.GLOBAL.RESET_ALL_SEQUENCES := NOT ("M_ONE" AND NOT "DB440_MACHINE_ALARM_DECODING".ALARMS_UNIT_01.ST0_TRANSFER.RESET_ALL_SEQUENCES AND NOT "DB440_MACHINE_ALARM_DECODING".ALARMS_UNIT_01.ST1_LOAD_UNLOAD.RESET_ALL_SEQUENCES AND NOT "DB440_MACHINE_ALARM_DECODING".ALARMS_UNIT_01.ST2_SPARE.RESET_ALL_SEQUENCES AND NOT "DB440_MACHINE_ALARM_DECODING".ALARMS_UNIT_01.ST3_CLADDING.RESET_ALL_SEQUENCES AND NOT "DB440_MACHINE_ALARM_DECODING".ALARMS_UNIT_01.ST4_CLEANING.RESET_ALL_SEQUENCES);
   "DB440_MACHINE_ALARM_DECODING".ALARMS_UNIT_01.GLOBAL.RESET_LOCAL_SEQUENCES := NOT ("M_ONE" AND NOT "DB440_MACHINE_ALARM_DECODING".ALARMS_UNIT_01.ST0_TRANSFER.RESET_LOCAL_SEQUENCES AND NOT "DB440_MACHINE_ALARM_DECODING".ALARMS_UNIT_01.ST1_LOAD_UNLOAD.RESET_LOCAL_SEQUENCES AND NOT "DB440_MACHINE_ALARM_DECODING".ALARMS_UNIT_01.ST2_SPARE.RESET_LOCAL_SEQUENCES AND NOT "DB440_MACHINE_ALARM_DECODING".ALARMS_UNIT_01.ST3_CLADDING.RESET_LOCAL_SEQUENCES AND NOT "DB440_MACHINE_ALARM_DECODING".ALARMS_UNIT_01.ST4_CLEANING.RESET_LOCAL_SEQUENCES);
END_REGION

REGION Network 27: <<<<<<<<<<<<<<<<<<<<<<<< UNIT 02 >>>>>>>>>>>>>>>>>>>>>>>>
END_REGION

